REGION Network 30: CLOSEED 1 ALARM
   RUNG wire#powerrail
      I_Contact( #CYL.CLOSE_COMMAND )
      I_Contact( #CLOSE )
      Not()
      Contact( #CLOSED_1_I )
      Contact( #OPENED_1_I )
      Contact( #CYL.SIMULTANEITY_ALARM )
      wire#w1
      Contact( #O_BYTE_0.OPENED_INPUT_1 )
      Contact( "DB1401_PNEUMATIC_SYSTEM".IN_SERVICE )
      Coil( #OPENED_1_ALARM )
   END_RUNG
   RUNG wire#powerrail
      I_Contact( #CYL.OPEN_COMMAND )
      I_Contact( #OPEN )
      Not()
      Contact( #CYL.TIME_EXCEEDED_ALARM )
      I_Contact( #OPENED_1_I )
   END_RUNG wire#w1
   RUNG wire#powerrail
      Contact( #OPENED_1_ALARM )
      I_Contact( "DB2120_MPP_ITC_IPC".RESET_FAULTS )
   END_RUNG wire#w1
   // the same network as SCL:
   #OPENED_1_ALARM := ((NOT (NOT #CYL.CLOSE_COMMAND AND NOT #CLOSE) AND #CLOSED_1_I AND #OPENED_1_I AND #CYL.SIMULTANEITY_ALARM) OR (NOT (NOT #CYL.OPEN_COMMAND AND NOT #OPEN) AND #CYL.TIME_EXCEEDED_ALARM AND NOT #OPENED_1_I) OR (#OPENED_1_ALARM AND NOT "DB2120_MPP_ITC_IPC".RESET_FAULTS)) AND #O_BYTE_0.OPENED_INPUT_1 AND "DB1401_PNEUMATIC_SYSTEM".IN_SERVICE;
END_REGION

REGION Network 31: CLOSEED 2 ALARM
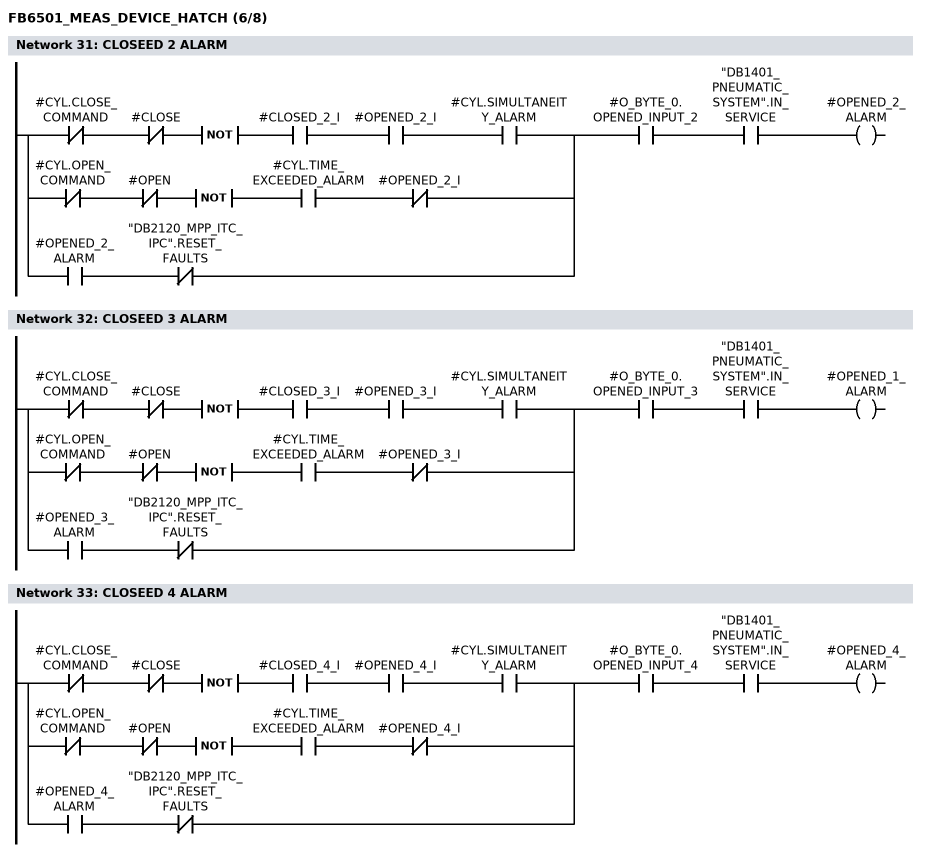
   RUNG wire#powerrail
      I_Contact( #CYL.CLOSE_COMMAND )
      I_Contact( #CLOSE )
      Not()
      Contact( #CLOSED_2_I )
      Contact( #OPENED_2_I )
      Contact( #CYL.SIMULTANEITY_ALARM )
      wire#w1
      Contact( #O_BYTE_0.OPENED_INPUT_2 )
      Contact( "DB1401_PNEUMATIC_SYSTEM".IN_SERVICE )
      Coil( #OPENED_2_ALARM )
   END_RUNG
   RUNG wire#powerrail
      I_Contact( #CYL.OPEN_COMMAND )
      I_Contact( #OPEN )
      Not()
      Contact( #CYL.TIME_EXCEEDED_ALARM )
      I_Contact( #OPENED_2_I )
   END_RUNG wire#w1
   RUNG wire#powerrail
      Contact( #OPENED_2_ALARM )
      I_Contact( "DB2120_MPP_ITC_IPC".RESET_FAULTS )
   END_RUNG wire#w1
   // the same network as SCL:
   #OPENED_2_ALARM := ((NOT (NOT #CYL.CLOSE_COMMAND AND NOT #CLOSE) AND #CLOSED_2_I AND #OPENED_2_I AND #CYL.SIMULTANEITY_ALARM) OR (NOT (NOT #CYL.OPEN_COMMAND AND NOT #OPEN) AND #CYL.TIME_EXCEEDED_ALARM AND NOT #OPENED_2_I) OR (#OPENED_2_ALARM AND NOT "DB2120_MPP_ITC_IPC".RESET_FAULTS)) AND #O_BYTE_0.OPENED_INPUT_2 AND "DB1401_PNEUMATIC_SYSTEM".IN_SERVICE;
END_REGION

REGION Network 32: CLOSEED 3 ALARM
   RUNG wire#powerrail
      I_Contact( #CYL.CLOSE_COMMAND )
      I_Contact( #CLOSE )
      Not()
      Contact( #CLOSED_3_I )
      Contact( #OPENED_3_I )
      Contact( #CYL.SIMULTANEITY_ALARM )
      wire#w1
      Contact( #O_BYTE_0.OPENED_INPUT_3 )
      Contact( "DB1401_PNEUMATIC_SYSTEM".IN_SERVICE )
      Coil( #OPENED_1_ALARM )
   END_RUNG
   RUNG wire#powerrail
      I_Contact( #CYL.OPEN_COMMAND )
      I_Contact( #OPEN )
      Not()
      Contact( #CYL.TIME_EXCEEDED_ALARM )
      I_Contact( #OPENED_3_I )
   END_RUNG wire#w1
   RUNG wire#powerrail
      Contact( #OPENED_3_ALARM )
      I_Contact( "DB2120_MPP_ITC_IPC".RESET_FAULTS )
   END_RUNG wire#w1
   // the same network as SCL:
   #OPENED_1_ALARM := ((NOT (NOT #CYL.CLOSE_COMMAND AND NOT #CLOSE) AND #CLOSED_3_I AND #OPENED_3_I AND #CYL.SIMULTANEITY_ALARM) OR (NOT (NOT #CYL.OPEN_COMMAND AND NOT #OPEN) AND #CYL.TIME_EXCEEDED_ALARM AND NOT #OPENED_3_I) OR (#OPENED_3_ALARM AND NOT "DB2120_MPP_ITC_IPC".RESET_FAULTS)) AND #O_BYTE_0.OPENED_INPUT_3 AND "DB1401_PNEUMATIC_SYSTEM".IN_SERVICE;
END_REGION

REGION Network 33: CLOSEED 4 ALARM
   RUNG wire#powerrail
      I_Contact( #CYL.CLOSE_COMMAND )
      I_Contact( #CLOSE )
      Not()
      Contact( #CLOSED_4_I )
      Contact( #OPENED_4_I )
      Contact( #CYL.SIMULTANEITY_ALARM )
      wire#w1
      Contact( #O_BYTE_0.OPENED_INPUT_4 )
      Contact( "DB1401_PNEUMATIC_SYSTEM".IN_SERVICE )
      Coil( #OPENED_4_ALARM )
   END_RUNG
   RUNG wire#powerrail
      I_Contact( #CYL.OPEN_COMMAND )
      I_Contact( #OPEN )
      Not()
      Contact( #CYL.TIME_EXCEEDED_ALARM )
      I_Contact( #OPENED_4_I )
   END_RUNG wire#w1
   RUNG wire#powerrail
      Contact( #OPENED_4_ALARM )
      I_Contact( "DB2120_MPP_ITC_IPC".RESET_FAULTS )
   END_RUNG wire#w1
   // the same network as SCL:
   #OPENED_4_ALARM := ((NOT (NOT #CYL.CLOSE_COMMAND AND NOT #CLOSE) AND #CLOSED_4_I AND #OPENED_4_I AND #CYL.SIMULTANEITY_ALARM) OR (NOT (NOT #CYL.OPEN_COMMAND AND NOT #OPEN) AND #CYL.TIME_EXCEEDED_ALARM AND NOT #OPENED_4_I) OR (#OPENED_4_ALARM AND NOT "DB2120_MPP_ITC_IPC".RESET_FAULTS)) AND #O_BYTE_0.OPENED_INPUT_4 AND "DB1401_PNEUMATIC_SYSTEM".IN_SERVICE;
END_REGION

REGION Network 34: IMMEDIATE STOP AND STOP END OF CYCLE ALARMS
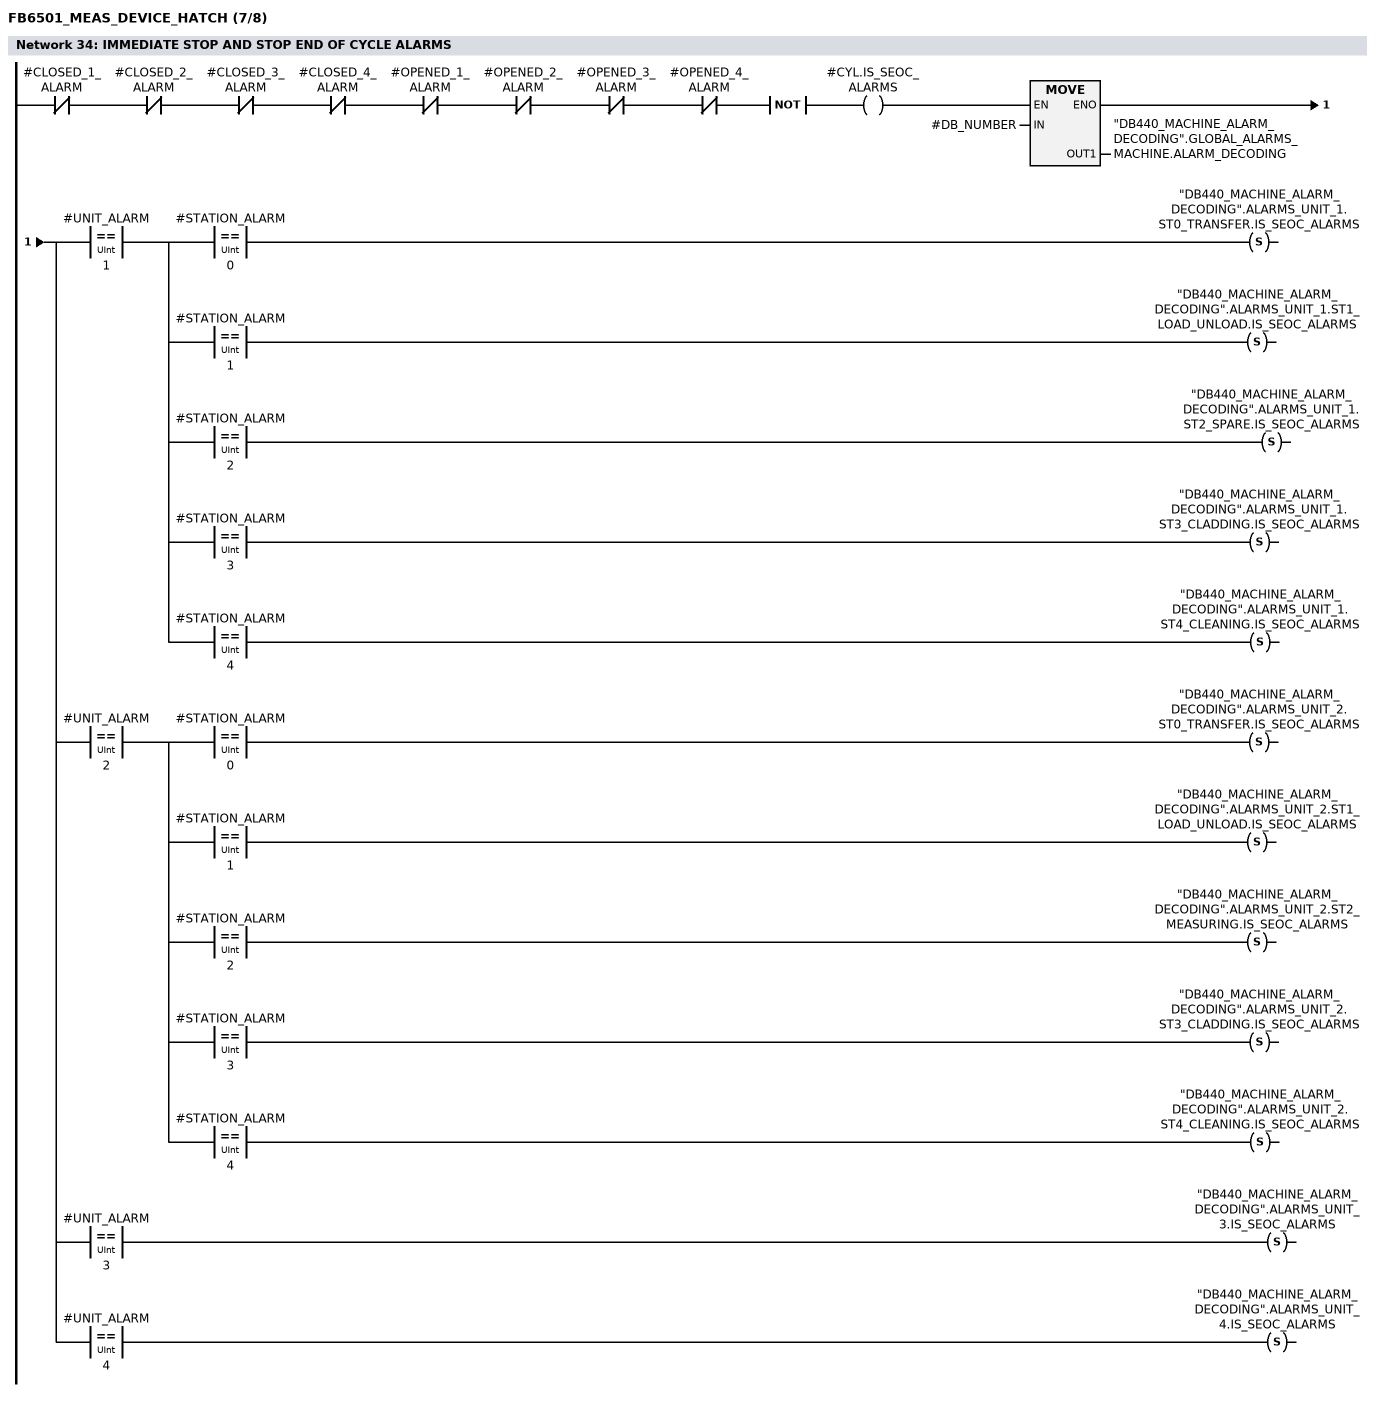
   RUNG wire#powerrail
      I_Contact( #CLOSED_1_ALARM )
      I_Contact( #CLOSED_2_ALARM )
      I_Contact( #CLOSED_3_ALARM )
      I_Contact( #CLOSED_4_ALARM )
      I_Contact( #OPENED_1_ALARM )
      I_Contact( #OPENED_2_ALARM )
      I_Contact( #OPENED_3_ALARM )
      I_Contact( #OPENED_4_ALARM )
      Not()
      Coil( #CYL.IS_SEOC_ALARMS )
      { S7_GenerateENO := "TRUE" } Move(in := #DB_NUMBER, out1 => "DB440_MACHINE_ALARM_DECODING".GLOBAL_ALARMS_MACHINE.ALARM_DECODING)
      wire#w1
      { S7_Templates := "SrcType := UInt" } EQ_Contact(in1 := #UNIT_ALARM, in2 := 1)
      wire#w2
      { S7_Templates := "SrcType := UInt" } EQ_Contact(in1 := #STATION_ALARM, in2 := 0)
      S_Coil( "DB440_MACHINE_ALARM_DECODING".ALARMS_UNIT_1.ST0_TRANSFER.IS_SEOC_ALARMS )
   END_RUNG
   RUNG wire#w2
      { S7_Templates := "SrcType := UInt" } EQ_Contact(in1 := #STATION_ALARM, in2 := 1)
      S_Coil( "DB440_MACHINE_ALARM_DECODING".ALARMS_UNIT_1.ST1_LOAD_UNLOAD.IS_SEOC_ALARMS )
   END_RUNG
   RUNG wire#w2
      { S7_Templates := "SrcType := UInt" } EQ_Contact(in1 := #STATION_ALARM, in2 := 2)
      S_Coil( "DB440_MACHINE_ALARM_DECODING".ALARMS_UNIT_1.ST2_SPARE.IS_SEOC_ALARMS )
   END_RUNG
   RUNG wire#w2
      { S7_Templates := "SrcType := UInt" } EQ_Contact(in1 := #STATION_ALARM, in2 := 3)
      S_Coil( "DB440_MACHINE_ALARM_DECODING".ALARMS_UNIT_1.ST3_CLADDING.IS_SEOC_ALARMS )
   END_RUNG
   RUNG wire#w2
      { S7_Templates := "SrcType := UInt" } EQ_Contact(in1 := #STATION_ALARM, in2 := 4)
      S_Coil( "DB440_MACHINE_ALARM_DECODING".ALARMS_UNIT_1.ST4_CLEANING.IS_SEOC_ALARMS )
   END_RUNG
   RUNG wire#w1
      { S7_Templates := "SrcType := UInt" } EQ_Contact(in1 := #UNIT_ALARM, in2 := 2)
      wire#w3
      { S7_Templates := "SrcType := UInt" } EQ_Contact(in1 := #STATION_ALARM, in2 := 0)
      S_Coil( "DB440_MACHINE_ALARM_DECODING".ALARMS_UNIT_2.ST0_TRANSFER.IS_SEOC_ALARMS )
   END_RUNG
   RUNG wire#w3
      { S7_Templates := "SrcType := UInt" } EQ_Contact(in1 := #STATION_ALARM, in2 := 1)
      S_Coil( "DB440_MACHINE_ALARM_DECODING".ALARMS_UNIT_2.ST1_LOAD_UNLOAD.IS_SEOC_ALARMS )
   END_RUNG
   RUNG wire#w3
      { S7_Templates := "SrcType := UInt" } EQ_Contact(in1 := #STATION_ALARM, in2 := 2)
      S_Coil( "DB440_MACHINE_ALARM_DECODING".ALARMS_UNIT_2.ST2_MEASURING.IS_SEOC_ALARMS )
   END_RUNG
   RUNG wire#w3
      { S7_Templates := "SrcType := UInt" } EQ_Contact(in1 := #STATION_ALARM, in2 := 3)
      S_Coil( "DB440_MACHINE_ALARM_DECODING".ALARMS_UNIT_2.ST3_CLADDING.IS_SEOC_ALARMS )
   END_RUNG
   RUNG wire#w3
      { S7_Templates := "SrcType := UInt" } EQ_Contact(in1 := #STATION_ALARM, in2 := 4)
      S_Coil( "DB440_MACHINE_ALARM_DECODING".ALARMS_UNIT_2.ST4_CLEANING.IS_SEOC_ALARMS )
   END_RUNG
   RUNG wire#w1
      { S7_Templates := "SrcType := UInt" } EQ_Contact(in1 := #UNIT_ALARM, in2 := 3)
      S_Coil( "DB440_MACHINE_ALARM_DECODING".ALARMS_UNIT_3.IS_SEOC_ALARMS )
   END_RUNG
   RUNG wire#w1
      { S7_Templates := "SrcType := UInt" } EQ_Contact(in1 := #UNIT_ALARM, in2 := 4)
      S_Coil( "DB440_MACHINE_ALARM_DECODING".ALARMS_UNIT_4.IS_SEOC_ALARMS )
   END_RUNG
   // the same network as SCL:
   // ENO of a box is taken as its EN; it also drops when the box reports an error
   #CYL.IS_SEOC_ALARMS := NOT (NOT #CLOSED_1_ALARM AND NOT #CLOSED_2_ALARM AND NOT #CLOSED_3_ALARM AND NOT #CLOSED_4_ALARM AND NOT #OPENED_1_ALARM AND NOT #OPENED_2_ALARM AND NOT #OPENED_3_ALARM AND NOT #OPENED_4_ALARM);
   IF #CYL.IS_SEOC_ALARMS THEN
       "DB440_MACHINE_ALARM_DECODING".GLOBAL_ALARMS_MACHINE.ALARM_DECODING := #DB_NUMBER;
   END_IF;
   #_w1 := #CYL.IS_SEOC_ALARMS AND (#UNIT_ALARM = 1);
   IF #_w1 AND (#STATION_ALARM = 0) THEN
       "DB440_MACHINE_ALARM_DECODING".ALARMS_UNIT_1.ST0_TRANSFER.IS_SEOC_ALARMS := TRUE;
   END_IF;
   IF #_w1 AND (#STATION_ALARM = 1) THEN
       "DB440_MACHINE_ALARM_DECODING".ALARMS_UNIT_1.ST1_LOAD_UNLOAD.IS_SEOC_ALARMS := TRUE;
   END_IF;
   IF #_w1 AND (#STATION_ALARM = 2) THEN
       "DB440_MACHINE_ALARM_DECODING".ALARMS_UNIT_1.ST2_SPARE.IS_SEOC_ALARMS := TRUE;
   END_IF;
   IF #_w1 AND (#STATION_ALARM = 3) THEN
       "DB440_MACHINE_ALARM_DECODING".ALARMS_UNIT_1.ST3_CLADDING.IS_SEOC_ALARMS := TRUE;
   END_IF;
   IF #_w1 AND (#STATION_ALARM = 4) THEN
       "DB440_MACHINE_ALARM_DECODING".ALARMS_UNIT_1.ST4_CLEANING.IS_SEOC_ALARMS := TRUE;
   END_IF;
   #_w2 := #CYL.IS_SEOC_ALARMS AND (#UNIT_ALARM = 2);
   IF #_w2 AND (#STATION_ALARM = 0) THEN
       "DB440_MACHINE_ALARM_DECODING".ALARMS_UNIT_2.ST0_TRANSFER.IS_SEOC_ALARMS := TRUE;
   END_IF;
   IF #_w2 AND (#STATION_ALARM = 1) THEN
       "DB440_MACHINE_ALARM_DECODING".ALARMS_UNIT_2.ST1_LOAD_UNLOAD.IS_SEOC_ALARMS := TRUE;
   END_IF;
   IF #_w2 AND (#STATION_ALARM = 2) THEN
       "DB440_MACHINE_ALARM_DECODING".ALARMS_UNIT_2.ST2_MEASURING.IS_SEOC_ALARMS := TRUE;
   END_IF;
   IF #_w2 AND (#STATION_ALARM = 3) THEN
       "DB440_MACHINE_ALARM_DECODING".ALARMS_UNIT_2.ST3_CLADDING.IS_SEOC_ALARMS := TRUE;
   END_IF;
   IF #_w2 AND (#STATION_ALARM = 4) THEN
       "DB440_MACHINE_ALARM_DECODING".ALARMS_UNIT_2.ST4_CLEANING.IS_SEOC_ALARMS := TRUE;
   END_IF;
   IF #CYL.IS_SEOC_ALARMS AND (#UNIT_ALARM = 3) THEN
       "DB440_MACHINE_ALARM_DECODING".ALARMS_UNIT_3.IS_SEOC_ALARMS := TRUE;
   END_IF;
   IF #CYL.IS_SEOC_ALARMS AND (#UNIT_ALARM = 4) THEN
       "DB440_MACHINE_ALARM_DECODING".ALARMS_UNIT_4.IS_SEOC_ALARMS := TRUE;
   END_IF;
END_REGION

REGION Network 35: ANY ACTIVE ALARM
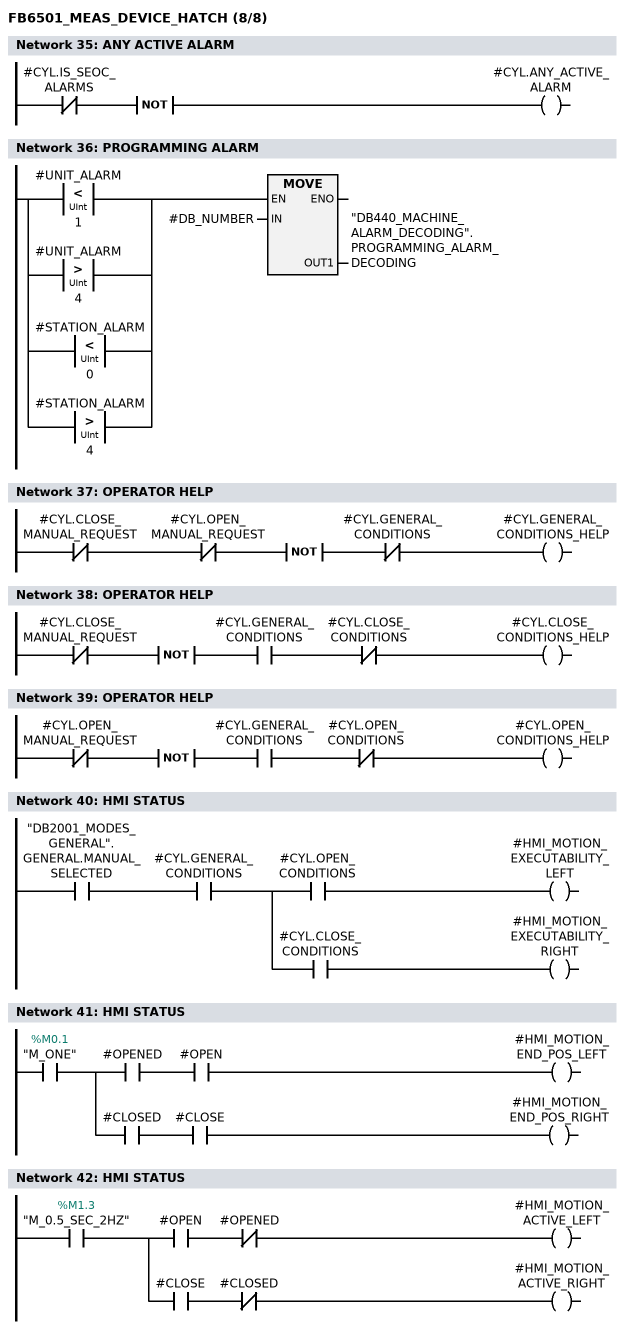
   RUNG wire#powerrail
      I_Contact( #CYL.IS_SEOC_ALARMS )
      Not()
      Coil( #CYL.ANY_ACTIVE_ALARM )
   END_RUNG
   // the same network as SCL:
   #CYL.ANY_ACTIVE_ALARM := NOT (NOT #CYL.IS_SEOC_ALARMS);
END_REGION

REGION Network 36: PROGRAMMING ALARM
   RUNG wire#powerrail
      { S7_Templates := "SrcType := UInt" } LT_Contact(in1 := #UNIT_ALARM, in2 := 1)
      wire#w1
      Move(in := #DB_NUMBER, out1 => "DB440_MACHINE_ALARM_DECODING".PROGRAMMING_ALARM_DECODING)
   END_RUNG
   RUNG wire#powerrail
      { S7_Templates := "SrcType := UInt" } GT_Contact(in1 := #UNIT_ALARM, in2 := 4)
   END_RUNG wire#w1
   RUNG wire#powerrail
      { S7_Templates := "SrcType := UInt" } LT_Contact(in1 := #STATION_ALARM, in2 := 0)
   END_RUNG wire#w1
   RUNG wire#powerrail
      { S7_Templates := "SrcType := UInt" } GT_Contact(in1 := #STATION_ALARM, in2 := 4)
   END_RUNG wire#w1
   // the same network as SCL:
   IF (#UNIT_ALARM < 1) OR (#UNIT_ALARM > 4) OR (#STATION_ALARM < 0) OR (#STATION_ALARM > 4) THEN
       "DB440_MACHINE_ALARM_DECODING".PROGRAMMING_ALARM_DECODING := #DB_NUMBER;
   END_IF;
END_REGION

REGION Network 37: OPERATOR HELP
   RUNG wire#powerrail
      I_Contact( #CYL.CLOSE_MANUAL_REQUEST )
      I_Contact( #CYL.OPEN_MANUAL_REQUEST )
      Not()
      I_Contact( #CYL.GENERAL_CONDITIONS )
      Coil( #CYL.GENERAL_CONDITIONS_HELP )
   END_RUNG
   // the same network as SCL:
   #CYL.GENERAL_CONDITIONS_HELP := NOT (NOT #CYL.CLOSE_MANUAL_REQUEST AND NOT #CYL.OPEN_MANUAL_REQUEST) AND NOT #CYL.GENERAL_CONDITIONS;
END_REGION

REGION Network 38: OPERATOR HELP
   RUNG wire#powerrail
      I_Contact( #CYL.CLOSE_MANUAL_REQUEST )
      Not()
      Contact( #CYL.GENERAL_CONDITIONS )
      I_Contact( #CYL.CLOSE_CONDITIONS )
      Coil( #CYL.CLOSE_CONDITIONS_HELP )
   END_RUNG
   // the same network as SCL:
   #CYL.CLOSE_CONDITIONS_HELP := NOT (NOT #CYL.CLOSE_MANUAL_REQUEST) AND #CYL.GENERAL_CONDITIONS AND NOT #CYL.CLOSE_CONDITIONS;
END_REGION

REGION Network 39: OPERATOR HELP
   RUNG wire#powerrail
      I_Contact( #CYL.OPEN_MANUAL_REQUEST )
      Not()
      Contact( #CYL.GENERAL_CONDITIONS )
      I_Contact( #CYL.OPEN_CONDITIONS )
      Coil( #CYL.OPEN_CONDITIONS_HELP )
   END_RUNG
   // the same network as SCL:
   #CYL.OPEN_CONDITIONS_HELP := NOT (NOT #CYL.OPEN_MANUAL_REQUEST) AND #CYL.GENERAL_CONDITIONS AND NOT #CYL.OPEN_CONDITIONS;
END_REGION

REGION Network 40: HMI STATUS
   RUNG wire#powerrail
      Contact( "DB2001_MODES_GENERAL".GENERAL.MANUAL_SELECTED )
      Contact( #CYL.GENERAL_CONDITIONS )
      wire#w1
      Contact( #CYL.OPEN_CONDITIONS )
      Coil( #HMI_MOTION_EXECUTABILITY_LEFT )
   END_RUNG
   RUNG wire#w1
      Contact( #CYL.CLOSE_CONDITIONS )
      Coil( #HMI_MOTION_EXECUTABILITY_RIGHT )
   END_RUNG
   // the same network as SCL:
   #_w1 := "DB2001_MODES_GENERAL".GENERAL.MANUAL_SELECTED AND #CYL.GENERAL_CONDITIONS;
   #HMI_MOTION_EXECUTABILITY_LEFT := #_w1 AND #CYL.OPEN_CONDITIONS;
   #HMI_MOTION_EXECUTABILITY_RIGHT := #_w1 AND #CYL.CLOSE_CONDITIONS;
END_REGION

REGION Network 41: HMI STATUS
   RUNG wire#powerrail
      Contact( "M_ONE" )
      wire#w1
      Contact( #OPENED )
      Contact( #OPEN )
      Coil( #HMI_MOTION_END_POS_LEFT )
   END_RUNG
   RUNG wire#w1
      Contact( #CLOSED )
      Contact( #CLOSE )
      Coil( #HMI_MOTION_END_POS_RIGHT )
   END_RUNG
   // the same network as SCL:
   #HMI_MOTION_END_POS_LEFT := "M_ONE" AND #OPENED AND #OPEN;
   #HMI_MOTION_END_POS_RIGHT := "M_ONE" AND #CLOSED AND #CLOSE;
END_REGION

REGION Network 42: HMI STATUS
   RUNG wire#powerrail
      Contact( "M_0.5_SEC_2HZ" )
      wire#w1
      Contact( #OPEN )
      I_Contact( #OPENED )
      Coil( #HMI_MOTION_ACTIVE_LEFT )
   END_RUNG
   RUNG wire#w1
      Contact( #CLOSE )
      I_Contact( #CLOSED )
      Coil( #HMI_MOTION_ACTIVE_RIGHT )
   END_RUNG
   // the same network as SCL:
   #HMI_MOTION_ACTIVE_LEFT := "M_0.5_SEC_2HZ" AND #OPEN AND NOT #OPENED;
   #HMI_MOTION_ACTIVE_RIGHT := "M_0.5_SEC_2HZ" AND #CLOSE AND NOT #CLOSED;
END_REGION
END_FUNCTION_BLOCK

FUNCTION_BLOCK "FB6502_SEALING_STRUCTURES"   // FB6502, LAD
{ S7_Optimized_Access := 'FALSE' }
AUTHOR : ETXETAR
VERSION : 1.0
// stored: AutoNumber false, IsIECCheckEnabled false, SetENOAutomatically false, UDAEnableTagReadback false
   VAR_INPUT
      OPTIONS_0 : Byte := 2#0000_0000;   // OPTIONS 0
      CLOSED_1_I : Bool;   // CLOSED 1 INPUT
      CLOSED_2_I : Bool;   // CLOSED 2 INPUT
      CLOSED_3_I : Bool;   // CLOSED 3 INPUT
      CLOSED_4_I : Bool;   // CLOSED 4 INPUT
      OPENED_1_I : Bool;   // OPENED 1 INPUT
      OPENED_2_I : Bool;   // OPENED 2 INPUT
      OPENED_3_I : Bool;   // OPENED 3 INPUT
      OPENED_4_I : Bool;   // OPENED 4 INPUT
      CLOSE_CONDITIONS : Bool;   // CLOSE CONDITIONS
      OPEN_CONDITIONS : Bool;   // OPEN CONDITIONS
      HMI_LINE_REQUEST : Bool;   // HMI LINE REQUEST
      CLOSE_AUTO_REQUEST : Bool;   // AUTO CLOSE REQUEST
      OPEN_AUTO_REQUEST_1 : Bool;   // AUTO OPEN REQUEST
      UNIT_ALARM : UInt;   // UNIT NUMBER MIN. NUMBER=1 MAX. NUMBER=4
      STATION_ALARM : UInt;   // STATION NUMBER MIN. NUMBER=0 MAX. NUMBER=4
   END_VAR
   VAR_OUTPUT
      CLOSED : Bool;   // CLOSED STATUS
      OPENED : Bool;   // OPENED STATUS
      CLOSED_1_ALARM : Bool;   // CLOSED 1 ALARM
      CLOSED_2_ALARM : Bool;   // CLOSED 2 ALARM
      CLOSED_3_ALARM : Bool;   // CLOSED 3 ALARM
      CLOSED_4_ALARM : Bool;   // CLOSED 4 ALARM
      OPENED_1_ALARM : Bool;   // OPENED 1 ALARM
      OPENED_2_ALARM : Bool;   // OPENED 2 ALARM
      OPENED_3_ALARM : Bool;   // OPENED 3 ALARM
      OPENED_4_ALARM : Bool;   // OPENED 4 ALARM
      HMI_MOTION_EXECUTABILITY_LEFT : Bool;   // HMI MOTION EXECUTABILITY LEFT
      HMI_MOTION_EXECUTABILITY_RIGHT : Bool;   // HMI MOTION EXECUTABILITY RIGHT
      HMI_MOTION_END_POS_LEFT : Bool;   // HMI MOTION END POSITION LEFT
      HMI_MOTION_END_POS_RIGHT : Bool;   // HMI MOTION END POSITION RIGHT
      HMI_MOTION_ACTIVE_LEFT : Bool;   // HMI MOTION ACTIVE LEFT
      HMI_MOTION_ACTIVE_RIGHT : Bool;   // HMI MOTION ACTIVE RIGHT
      CLOSE : Bool;   // CLOSE OUTPUT
      OPEN : Bool;   // OPEN OUTPUT
   END_VAR
   VAR DB_SPECIFIC
      CYL { S7_SetPoint := 'True'} : "OPEN_CLOSE_HATCH_CLADDING";
      TIMER_CLOSED { S7_SetPoint := 'True'} : TON_TIME;   // CLOSED TIMER
      TIMER_OPENED { S7_SetPoint := 'True'} : TON_TIME;   // OPENED TIMER
      TIMER_SIMULTANEITY { S7_SetPoint := 'True'} : TON_TIME;   // SIMULTANEITY TIMER
      TIMER_TIME_EXCEEDED { S7_SetPoint := 'True'} : TON_TIME;   // TIME EXCEEDED TIMER
   END_VAR
   VAR_TEMP
      INPUTS_MASK : Byte;   // INPUTS_MASK
      O_BYTE_0 : Struct   // OPTIONS BYTE 0
         CLOSED_INPUT_1 : Bool;   // CLOSED INPUT 1 OPTION
         CLOSED_INPUT_2 : Bool;   // CLOSED INPUT 2 OPTION
         CLOSED_INPUT_3 : Bool;   // CLOSED
         CLOSED_INPUT_4 : Bool;   // CLOSED INPUT 4 OPTION
         OPENED_INPUT_1 : Bool;   // OPENED INPUT 1 OPTION
         OPENED_INPUT_2 : Bool;   // OPENED INPUT 2 OPTION
         OPENED_INPUT_3 : Bool;   // OPENED INPUT 3 OPTION
         OPENED_INPUT_4 : Bool;   // OPENED INPUT 4 OPTION
      END_STRUCT;
      DB_NUMBER : DInt;   // DB NUMBER FOR ALARM AND HELP DECODING
   END_VAR
   // TIMER_CLOSED.PT := T#100MS;
   // TIMER_OPENED.PT := T#300MS;
   // TIMER_SIMULTANEITY.PT := T#100MS;
   // TIMER_TIME_EXCEEDED.PT := T#8S;
   VAR_TEMP   // added for the SCL form of the ladder/FBD networks
      _w1 : Bool;
      _w2 : Bool;
   END_VAR
BEGIN

NETWORK
TITLE = READ INSTANCE DB
      L     DINO;
      +     10#800000;
      T     #DB_NUMBER;


REGION Network 2: OPTIONS
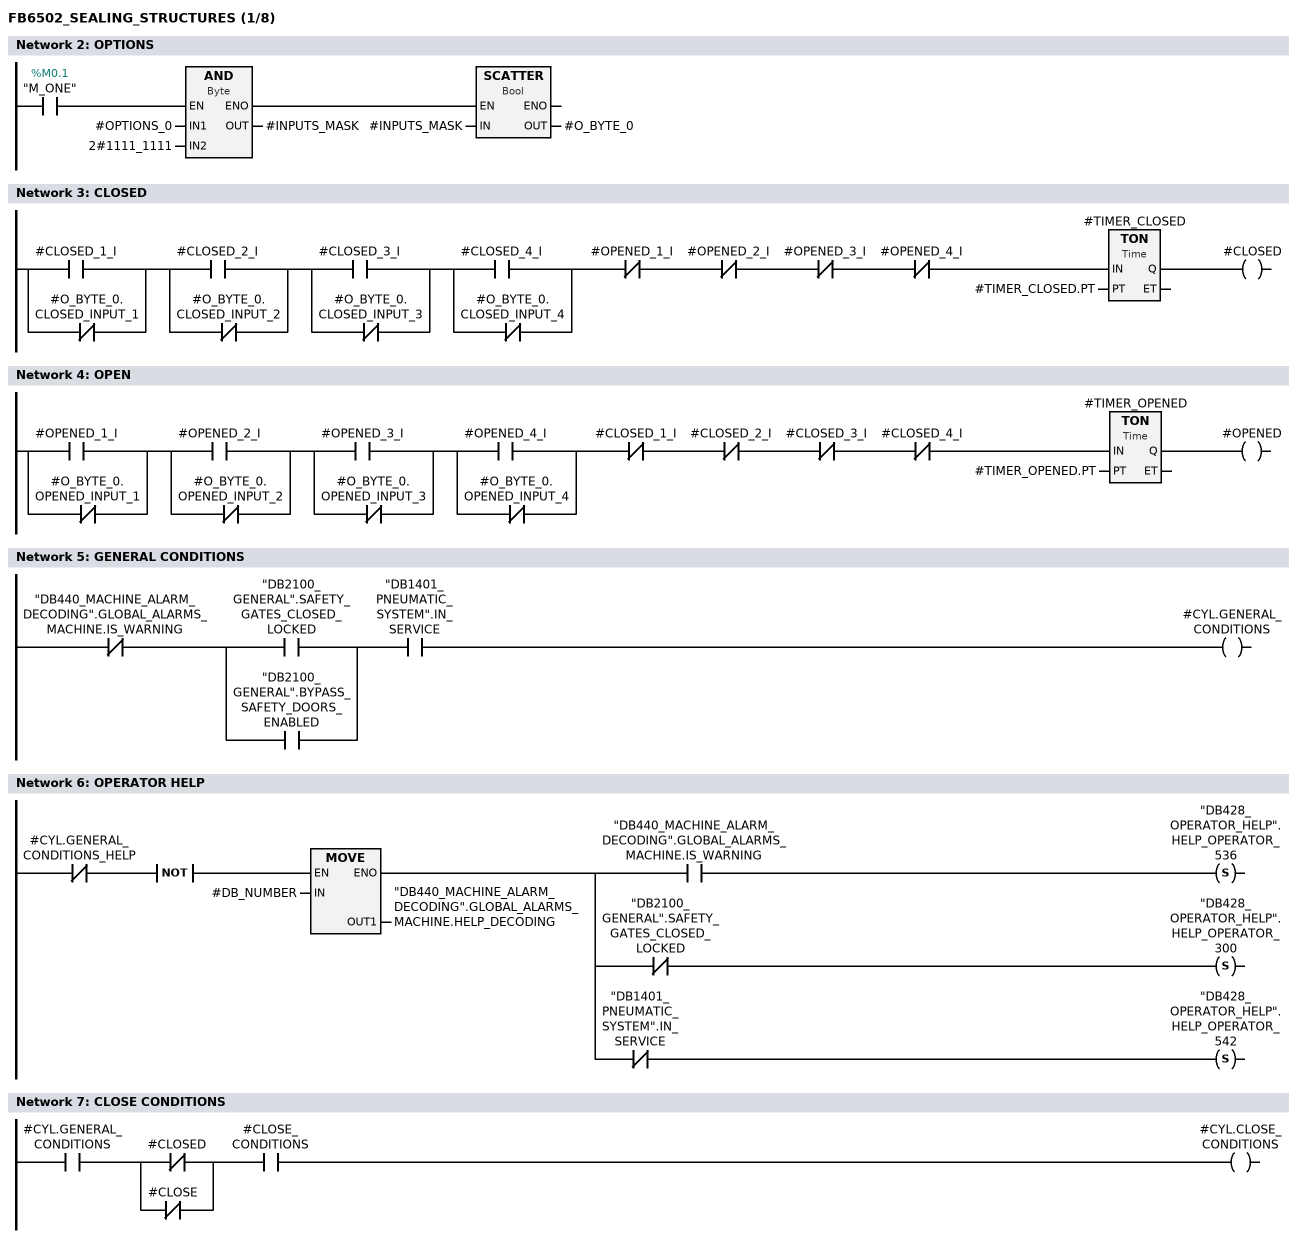
   RUNG wire#powerrail
      Contact( "M_ONE" )
      { S7_Templates := "SrcType := Byte"; S7_GenerateENO := "TRUE" } And(in1 := #OPTIONS_0, in2 := 2#1111_1111, out => #INPUTS_MASK)
      { S7_Templates := "[dest_type := Bool, src_type := Byte]" } SCATTER(IN := #INPUTS_MASK, OUT => #O_BYTE_0)
   END_RUNG
   // the same network as SCL:
   IF "M_ONE" THEN
       #INPUTS_MASK := #OPTIONS_0 AND 2#1111_1111;
       SCATTER(IN := #INPUTS_MASK, OUT => #O_BYTE_0);
   END_IF;
END_REGION

REGION Network 3: CLOSED
   RUNG wire#powerrail
      Contact( #CLOSED_1_I )
      wire#w1
      Contact( #CLOSED_2_I )
      wire#w2
      Contact( #CLOSED_3_I )
      wire#w3
      Contact( #CLOSED_4_I )
      wire#w4
      I_Contact( #OPENED_1_I )
      I_Contact( #OPENED_2_I )
      I_Contact( #OPENED_3_I )
      I_Contact( #OPENED_4_I )
      { S7_Templates := "time_type := Time" } #TIMER_CLOSED.TON(pt := #TIMER_CLOSED.PT, et =>)
      Coil( #CLOSED )
   END_RUNG
   RUNG wire#powerrail
      I_Contact( #O_BYTE_0.CLOSED_INPUT_1 )
   END_RUNG wire#w1
   RUNG wire#w1
      I_Contact( #O_BYTE_0.CLOSED_INPUT_2 )
   END_RUNG wire#w2
   RUNG wire#w2
      I_Contact( #O_BYTE_0.CLOSED_INPUT_3 )
   END_RUNG wire#w3
   RUNG wire#w3
      I_Contact( #O_BYTE_0.CLOSED_INPUT_4 )
   END_RUNG wire#w4
   // the same network as SCL:
   #TIMER_CLOSED(IN := (#CLOSED_1_I OR NOT #O_BYTE_0.CLOSED_INPUT_1) AND (#CLOSED_2_I OR NOT #O_BYTE_0.CLOSED_INPUT_2) AND (#CLOSED_3_I OR NOT #O_BYTE_0.CLOSED_INPUT_3) AND (#CLOSED_4_I OR NOT #O_BYTE_0.CLOSED_INPUT_4) AND NOT #OPENED_1_I AND NOT #OPENED_2_I AND NOT #OPENED_3_I AND NOT #OPENED_4_I,   // TON
                 PT := #TIMER_CLOSED.PT);
   #CLOSED := #TIMER_CLOSED.Q;
END_REGION

REGION Network 4: OPEN
   RUNG wire#powerrail
      Contact( #OPENED_1_I )
      wire#w1
      Contact( #OPENED_2_I )
      wire#w2
      Contact( #OPENED_3_I )
      wire#w3
      Contact( #OPENED_4_I )
      wire#w4
      I_Contact( #CLOSED_1_I )
      I_Contact( #CLOSED_2_I )
      I_Contact( #CLOSED_3_I )
      I_Contact( #CLOSED_4_I )
      { S7_Templates := "time_type := Time" } #TIMER_OPENED.TON(pt := #TIMER_OPENED.PT, et =>)
      Coil( #OPENED )
   END_RUNG
   RUNG wire#powerrail
      I_Contact( #O_BYTE_0.OPENED_INPUT_1 )
   END_RUNG wire#w1
   RUNG wire#w1
      I_Contact( #O_BYTE_0.OPENED_INPUT_2 )
   END_RUNG wire#w2
   RUNG wire#w2
      I_Contact( #O_BYTE_0.OPENED_INPUT_3 )
   END_RUNG wire#w3
   RUNG wire#w3
      I_Contact( #O_BYTE_0.OPENED_INPUT_4 )
   END_RUNG wire#w4
   // the same network as SCL:
   #TIMER_OPENED(IN := (#OPENED_1_I OR NOT #O_BYTE_0.OPENED_INPUT_1) AND (#OPENED_2_I OR NOT #O_BYTE_0.OPENED_INPUT_2) AND (#OPENED_3_I OR NOT #O_BYTE_0.OPENED_INPUT_3) AND (#OPENED_4_I OR NOT #O_BYTE_0.OPENED_INPUT_4) AND NOT #CLOSED_1_I AND NOT #CLOSED_2_I AND NOT #CLOSED_3_I AND NOT #CLOSED_4_I,   // TON
                 PT := #TIMER_OPENED.PT);
   #OPENED := #TIMER_OPENED.Q;
END_REGION

REGION Network 5: GENERAL CONDITIONS
   RUNG wire#powerrail
      I_Contact( "DB440_MACHINE_ALARM_DECODING".GLOBAL_ALARMS_MACHINE.IS_WARNING )
      wire#w1
      Contact( "DB2100_GENERAL".SAFETY_GATES_CLOSED_LOCKED )
      wire#w2
      Contact( "DB1401_PNEUMATIC_SYSTEM".IN_SERVICE )
      Coil( #CYL.GENERAL_CONDITIONS )
   END_RUNG
   RUNG wire#w1
      Contact( "DB2100_GENERAL".BYPASS_SAFETY_DOORS_ENABLED )
   END_RUNG wire#w2
   // the same network as SCL:
   #CYL.GENERAL_CONDITIONS := NOT "DB440_MACHINE_ALARM_DECODING".GLOBAL_ALARMS_MACHINE.IS_WARNING AND ("DB2100_GENERAL".SAFETY_GATES_CLOSED_LOCKED OR "DB2100_GENERAL".BYPASS_SAFETY_DOORS_ENABLED) AND "DB1401_PNEUMATIC_SYSTEM".IN_SERVICE;
END_REGION

REGION Network 6: OPERATOR HELP
   RUNG wire#powerrail
      I_Contact( #CYL.GENERAL_CONDITIONS_HELP )
      Not()
      { S7_GenerateENO := "TRUE" } Move(in := #DB_NUMBER, out1 => "DB440_MACHINE_ALARM_DECODING".GLOBAL_ALARMS_MACHINE.HELP_DECODING)
      wire#w1
      Contact( "DB440_MACHINE_ALARM_DECODING".GLOBAL_ALARMS_MACHINE.IS_WARNING )
      S_Coil( "DB428_OPERATOR_HELP".HELP_OPERATOR_536 )
   END_RUNG
   RUNG wire#w1
      I_Contact( "DB2100_GENERAL".SAFETY_GATES_CLOSED_LOCKED )
      S_Coil( "DB428_OPERATOR_HELP".HELP_OPERATOR_300 )
   END_RUNG
   RUNG wire#w1
      I_Contact( "DB1401_PNEUMATIC_SYSTEM".IN_SERVICE )
      S_Coil( "DB428_OPERATOR_HELP".HELP_OPERATOR_542 )
   END_RUNG
   // the same network as SCL:
   // ENO of a box is taken as its EN; it also drops when the box reports an error
   #_w1 := NOT (NOT #CYL.GENERAL_CONDITIONS_HELP);
   IF #_w1 THEN "DB440_MACHINE_ALARM_DECODING".GLOBAL_ALARMS_MACHINE.HELP_DECODING := #DB_NUMBER; END_IF;
   IF #_w1 AND "DB440_MACHINE_ALARM_DECODING".GLOBAL_ALARMS_MACHINE.IS_WARNING THEN
       "DB428_OPERATOR_HELP".HELP_OPERATOR_536 := TRUE;
   END_IF;
   IF #_w1 AND NOT "DB2100_GENERAL".SAFETY_GATES_CLOSED_LOCKED THEN
       "DB428_OPERATOR_HELP".HELP_OPERATOR_300 := TRUE;
   END_IF;
   IF #_w1 AND NOT "DB1401_PNEUMATIC_SYSTEM".IN_SERVICE THEN
       "DB428_OPERATOR_HELP".HELP_OPERATOR_542 := TRUE;
   END_IF;
END_REGION

REGION Network 7: CLOSE CONDITIONS
   RUNG wire#powerrail
      Contact( #CYL.GENERAL_CONDITIONS )
      wire#w1
      I_Contact( #CLOSED )
      wire#w2
      Contact( #CLOSE_CONDITIONS )
      Coil( #CYL.CLOSE_CONDITIONS )
   END_RUNG
   RUNG wire#w1
      I_Contact( #CLOSE )
   END_RUNG wire#w2
   // the same network as SCL:
   #CYL.CLOSE_CONDITIONS := #CYL.GENERAL_CONDITIONS AND (NOT #CLOSED OR NOT #CLOSE) AND #CLOSE_CONDITIONS;
END_REGION

REGION Network 8: OPERATOR HELP
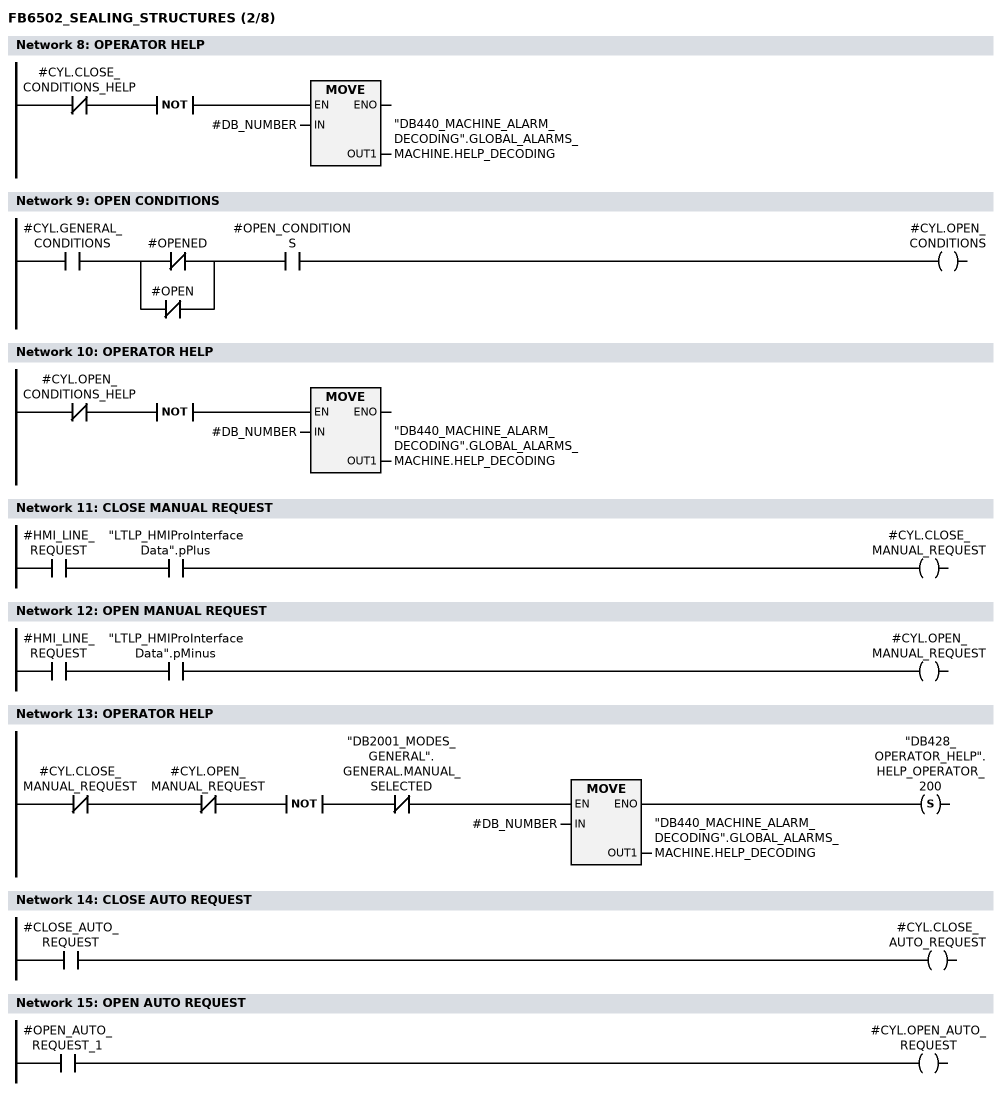
   RUNG wire#powerrail
      I_Contact( #CYL.CLOSE_CONDITIONS_HELP )
      Not()
      { S7_GenerateENO := "TRUE" } Move(in := #DB_NUMBER, out1 => "DB440_MACHINE_ALARM_DECODING".GLOBAL_ALARMS_MACHINE.HELP_DECODING)
   END_RUNG
   // the same network as SCL:
   IF NOT (NOT #CYL.CLOSE_CONDITIONS_HELP) THEN
       "DB440_MACHINE_ALARM_DECODING".GLOBAL_ALARMS_MACHINE.HELP_DECODING := #DB_NUMBER;
   END_IF;
END_REGION

REGION Network 9: OPEN CONDITIONS
   RUNG wire#powerrail
      Contact( #CYL.GENERAL_CONDITIONS )
      wire#w1
      I_Contact( #OPENED )
      wire#w2
      Contact( #OPEN_CONDITIONS )
      Coil( #CYL.OPEN_CONDITIONS )
   END_RUNG
   RUNG wire#w1
      I_Contact( #OPEN )
   END_RUNG wire#w2
   // the same network as SCL:
   #CYL.OPEN_CONDITIONS := #CYL.GENERAL_CONDITIONS AND (NOT #OPENED OR NOT #OPEN) AND #OPEN_CONDITIONS;
END_REGION

REGION Network 10: OPERATOR HELP
   RUNG wire#powerrail
      I_Contact( #CYL.OPEN_CONDITIONS_HELP )
      Not()
      { S7_GenerateENO := "TRUE" } Move(in := #DB_NUMBER, out1 => "DB440_MACHINE_ALARM_DECODING".GLOBAL_ALARMS_MACHINE.HELP_DECODING)
   END_RUNG
   // the same network as SCL:
   IF NOT (NOT #CYL.OPEN_CONDITIONS_HELP) THEN
       "DB440_MACHINE_ALARM_DECODING".GLOBAL_ALARMS_MACHINE.HELP_DECODING := #DB_NUMBER;
   END_IF;
END_REGION

REGION Network 11: CLOSE MANUAL REQUEST
   RUNG wire#powerrail
      Contact( #HMI_LINE_REQUEST )
      Contact( "LTLP_HMIProInterfaceData".pPlus )
      Coil( #CYL.CLOSE_MANUAL_REQUEST )
   END_RUNG
   // the same network as SCL:
   #CYL.CLOSE_MANUAL_REQUEST := #HMI_LINE_REQUEST AND "LTLP_HMIProInterfaceData".pPlus;
END_REGION

REGION Network 12: OPEN MANUAL REQUEST
   RUNG wire#powerrail
      Contact( #HMI_LINE_REQUEST )
      Contact( "LTLP_HMIProInterfaceData".pMinus )
      Coil( #CYL.OPEN_MANUAL_REQUEST )
   END_RUNG
   // the same network as SCL:
   #CYL.OPEN_MANUAL_REQUEST := #HMI_LINE_REQUEST AND "LTLP_HMIProInterfaceData".pMinus;
END_REGION

REGION Network 13: OPERATOR HELP
   RUNG wire#powerrail
      I_Contact( #CYL.CLOSE_MANUAL_REQUEST )
      I_Contact( #CYL.OPEN_MANUAL_REQUEST )
      Not()
      I_Contact( "DB2001_MODES_GENERAL".GENERAL.MANUAL_SELECTED )
      { S7_GenerateENO := "TRUE" } Move(in := #DB_NUMBER, out1 => "DB440_MACHINE_ALARM_DECODING".GLOBAL_ALARMS_MACHINE.HELP_DECODING)
      S_Coil( "DB428_OPERATOR_HELP".HELP_OPERATOR_200 )
   END_RUNG
   // the same network as SCL:
   // ENO of a box is taken as its EN; it also drops when the box reports an error
   IF NOT (NOT #CYL.CLOSE_MANUAL_REQUEST AND NOT #CYL.OPEN_MANUAL_REQUEST) AND NOT "DB2001_MODES_GENERAL".GENERAL.MANUAL_SELECTED THEN
       "DB440_MACHINE_ALARM_DECODING".GLOBAL_ALARMS_MACHINE.HELP_DECODING := #DB_NUMBER;
       "DB428_OPERATOR_HELP".HELP_OPERATOR_200 := TRUE;
   END_IF;
END_REGION

REGION Network 14: CLOSE AUTO REQUEST
   RUNG wire#powerrail
      Contact( #CLOSE_AUTO_REQUEST )
      Coil( #CYL.CLOSE_AUTO_REQUEST )
   END_RUNG
   // the same network as SCL:
   #CYL.CLOSE_AUTO_REQUEST := #CLOSE_AUTO_REQUEST;
END_REGION

REGION Network 15: OPEN AUTO REQUEST
   RUNG wire#powerrail
      Contact( #OPEN_AUTO_REQUEST_1 )
      Coil( #CYL.OPEN_AUTO_REQUEST )
   END_RUNG
   // the same network as SCL:
   #CYL.OPEN_AUTO_REQUEST := #OPEN_AUTO_REQUEST_1;
END_REGION

REGION Network 16: CLOSE GLOBAL REQUEST
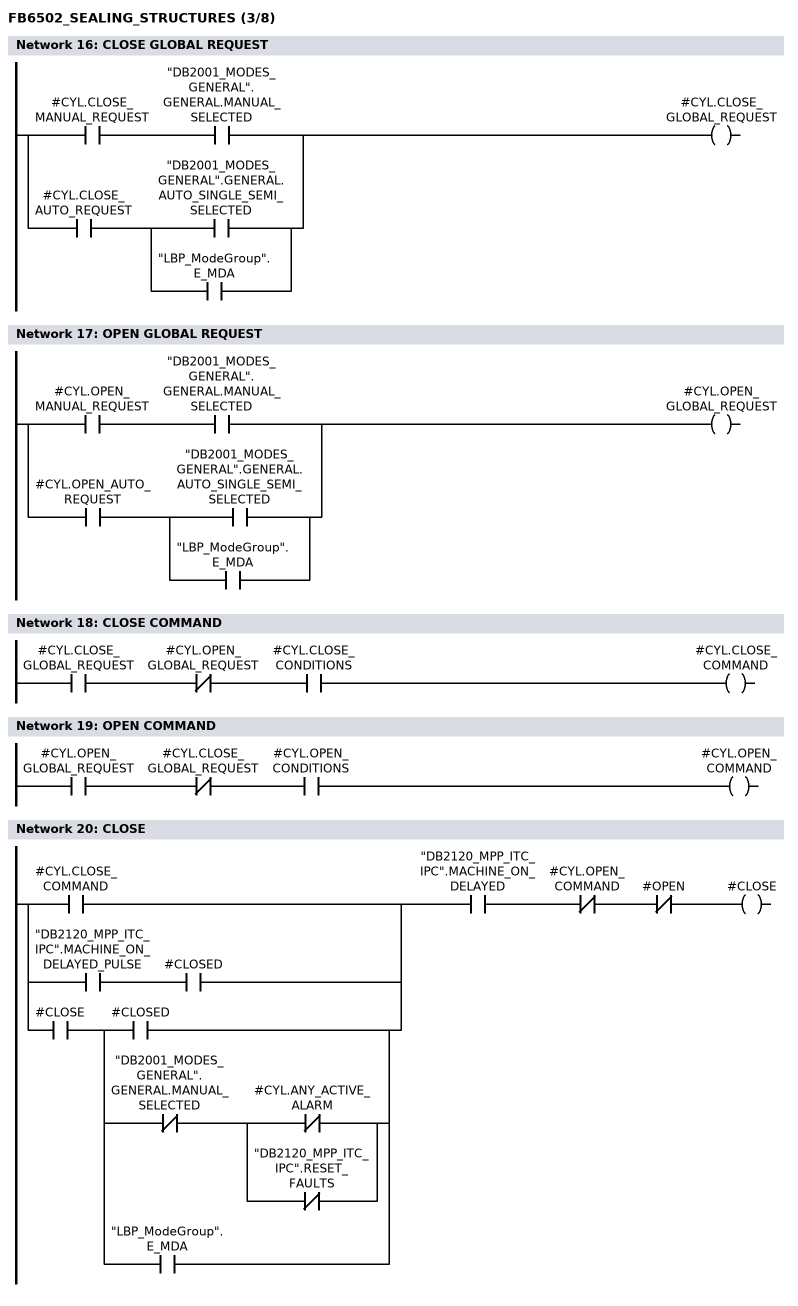
   RUNG wire#powerrail
      Contact( #CYL.CLOSE_MANUAL_REQUEST )
      Contact( "DB2001_MODES_GENERAL".GENERAL.MANUAL_SELECTED )
      wire#w1
      Coil( #CYL.CLOSE_GLOBAL_REQUEST )
   END_RUNG
   RUNG wire#powerrail
      Contact( #CYL.CLOSE_AUTO_REQUEST )
      wire#w2
      Contact( "DB2001_MODES_GENERAL".GENERAL.AUTO_SINGLE_SEMI_SELECTED )
   END_RUNG wire#w1
   RUNG wire#w2
      Contact( "LBP_ModeGroup".E_MDA )
   END_RUNG wire#w1
   // the same network as SCL:
   #CYL.CLOSE_GLOBAL_REQUEST := (#CYL.CLOSE_MANUAL_REQUEST AND "DB2001_MODES_GENERAL".GENERAL.MANUAL_SELECTED) OR (#CYL.CLOSE_AUTO_REQUEST AND ("DB2001_MODES_GENERAL".GENERAL.AUTO_SINGLE_SEMI_SELECTED OR "LBP_ModeGroup".E_MDA));
END_REGION

REGION Network 17: OPEN GLOBAL REQUEST
   RUNG wire#powerrail
      Contact( #CYL.OPEN_MANUAL_REQUEST )
      Contact( "DB2001_MODES_GENERAL".GENERAL.MANUAL_SELECTED )
      wire#w1
      Coil( #CYL.OPEN_GLOBAL_REQUEST )
   END_RUNG
   RUNG wire#powerrail
      Contact( #CYL.OPEN_AUTO_REQUEST )
      wire#w2
      Contact( "DB2001_MODES_GENERAL".GENERAL.AUTO_SINGLE_SEMI_SELECTED )
   END_RUNG wire#w1
   RUNG wire#w2
      Contact( "LBP_ModeGroup".E_MDA )
   END_RUNG wire#w1
   // the same network as SCL:
   #CYL.OPEN_GLOBAL_REQUEST := (#CYL.OPEN_MANUAL_REQUEST AND "DB2001_MODES_GENERAL".GENERAL.MANUAL_SELECTED) OR (#CYL.OPEN_AUTO_REQUEST AND ("DB2001_MODES_GENERAL".GENERAL.AUTO_SINGLE_SEMI_SELECTED OR "LBP_ModeGroup".E_MDA));
END_REGION

REGION Network 18: CLOSE COMMAND
   RUNG wire#powerrail
      Contact( #CYL.CLOSE_GLOBAL_REQUEST )
      I_Contact( #CYL.OPEN_GLOBAL_REQUEST )
      Contact( #CYL.CLOSE_CONDITIONS )
      Coil( #CYL.CLOSE_COMMAND )
   END_RUNG
   // the same network as SCL:
   #CYL.CLOSE_COMMAND := #CYL.CLOSE_GLOBAL_REQUEST AND NOT #CYL.OPEN_GLOBAL_REQUEST AND #CYL.CLOSE_CONDITIONS;
END_REGION

REGION Network 19: OPEN COMMAND
   RUNG wire#powerrail
      Contact( #CYL.OPEN_GLOBAL_REQUEST )
      I_Contact( #CYL.CLOSE_GLOBAL_REQUEST )
      Contact( #CYL.OPEN_CONDITIONS )
      Coil( #CYL.OPEN_COMMAND )
   END_RUNG
   // the same network as SCL:
   #CYL.OPEN_COMMAND := #CYL.OPEN_GLOBAL_REQUEST AND NOT #CYL.CLOSE_GLOBAL_REQUEST AND #CYL.OPEN_CONDITIONS;
END_REGION

REGION Network 20: CLOSE
   RUNG wire#powerrail
      Contact( #CYL.CLOSE_COMMAND )
      wire#w1
      Contact( "DB2120_MPP_ITC_IPC".MACHINE_ON_DELAYED )
      I_Contact( #CYL.OPEN_COMMAND )
      I_Contact( #OPEN )
      Coil( #CLOSE )
   END_RUNG
   RUNG wire#powerrail
      Contact( "DB2120_MPP_ITC_IPC".MACHINE_ON_DELAYED_PULSE )
      Contact( #CLOSED )
   END_RUNG wire#w1
   RUNG wire#powerrail
      Contact( #CLOSE )
      wire#w2
      Contact( #CLOSED )
   END_RUNG wire#w1
   RUNG wire#w2
      I_Contact( "DB2001_MODES_GENERAL".GENERAL.MANUAL_SELECTED )
      wire#w3
      I_Contact( #CYL.ANY_ACTIVE_ALARM )
   END_RUNG wire#w1
   RUNG wire#w3
      I_Contact( "DB2120_MPP_ITC_IPC".RESET_FAULTS )
   END_RUNG wire#w1
   RUNG wire#w2
      Contact( "LBP_ModeGroup".E_MDA )
   END_RUNG wire#w1
   // the same network as SCL:
   #CLOSE := (#CYL.CLOSE_COMMAND OR ("DB2120_MPP_ITC_IPC".MACHINE_ON_DELAYED_PULSE AND #CLOSED) OR (#CLOSE AND (#CLOSED OR (NOT "DB2001_MODES_GENERAL".GENERAL.MANUAL_SELECTED AND (NOT #CYL.ANY_ACTIVE_ALARM OR NOT "DB2120_MPP_ITC_IPC".RESET_FAULTS)) OR "LBP_ModeGroup".E_MDA))) AND "DB2120_MPP_ITC_IPC".MACHINE_ON_DELAYED AND NOT #CYL.OPEN_COMMAND AND NOT #OPEN;
END_REGION

REGION Network 21: OPEN
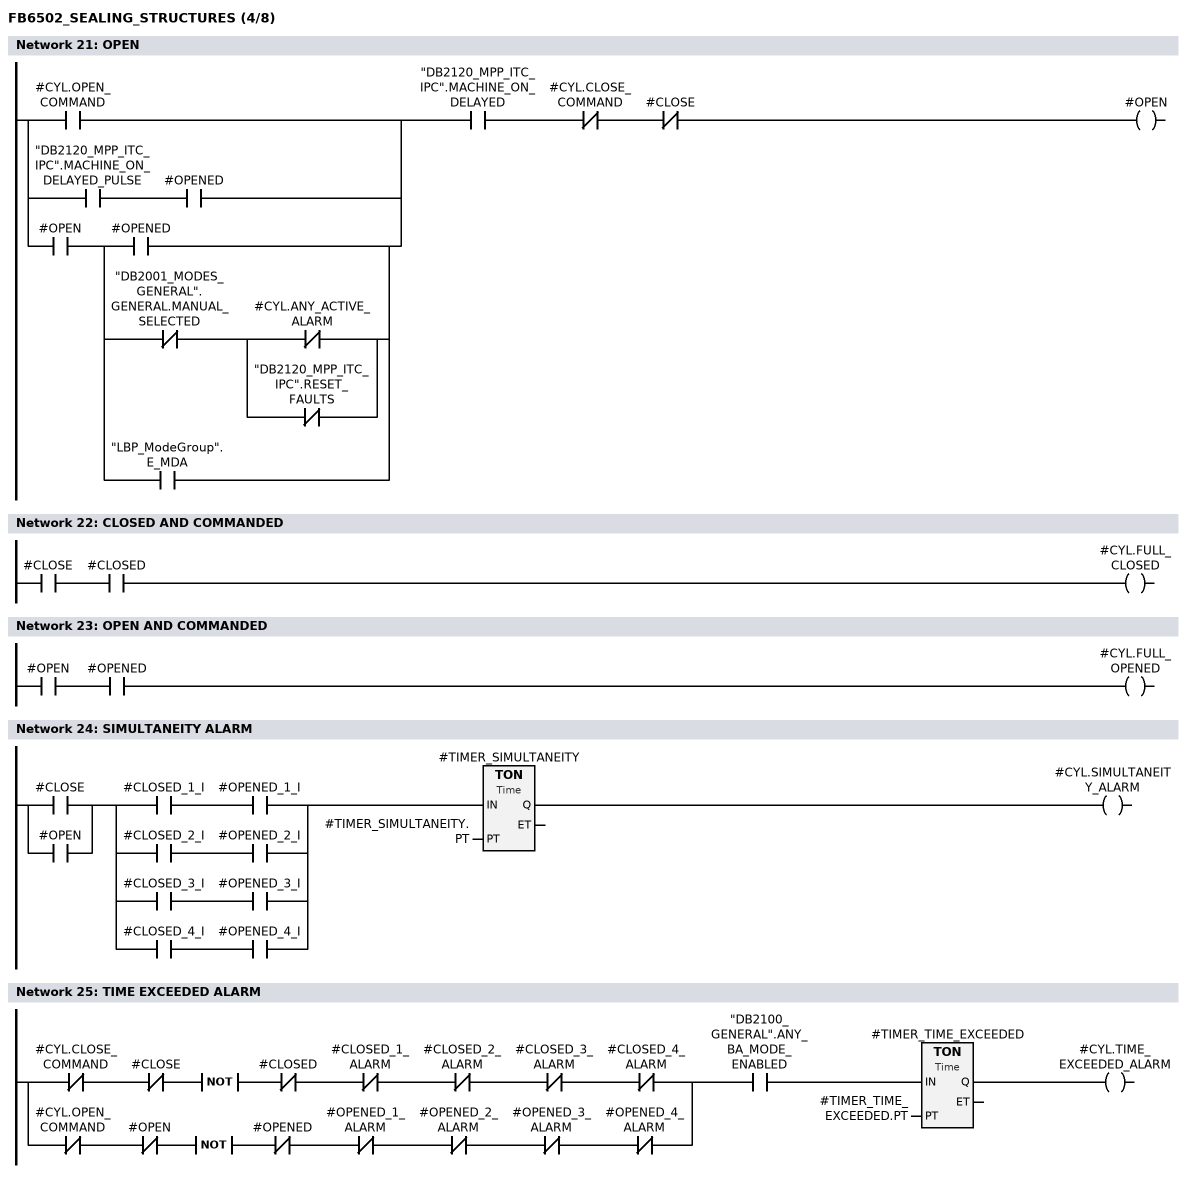
   RUNG wire#powerrail
      Contact( #CYL.OPEN_COMMAND )
      wire#w1
      Contact( "DB2120_MPP_ITC_IPC".MACHINE_ON_DELAYED )
      I_Contact( #CYL.CLOSE_COMMAND )
      I_Contact( #CLOSE )
      Coil( #OPEN )
   END_RUNG
   RUNG wire#powerrail
      Contact( "DB2120_MPP_ITC_IPC".MACHINE_ON_DELAYED_PULSE )
      Contact( #OPENED )
   END_RUNG wire#w1
   RUNG wire#powerrail
      Contact( #OPEN )
      wire#w2
      Contact( #OPENED )
   END_RUNG wire#w1
   RUNG wire#w2
      I_Contact( "DB2001_MODES_GENERAL".GENERAL.MANUAL_SELECTED )
      wire#w3
      I_Contact( #CYL.ANY_ACTIVE_ALARM )
   END_RUNG wire#w1
   RUNG wire#w3
      I_Contact( "DB2120_MPP_ITC_IPC".RESET_FAULTS )
   END_RUNG wire#w1
   RUNG wire#w2
      Contact( "LBP_ModeGroup".E_MDA )
   END_RUNG wire#w1
   // the same network as SCL:
   #OPEN := (#CYL.OPEN_COMMAND OR ("DB2120_MPP_ITC_IPC".MACHINE_ON_DELAYED_PULSE AND #OPENED) OR (#OPEN AND (#OPENED OR (NOT "DB2001_MODES_GENERAL".GENERAL.MANUAL_SELECTED AND (NOT #CYL.ANY_ACTIVE_ALARM OR NOT "DB2120_MPP_ITC_IPC".RESET_FAULTS)) OR "LBP_ModeGroup".E_MDA))) AND "DB2120_MPP_ITC_IPC".MACHINE_ON_DELAYED AND NOT #CYL.CLOSE_COMMAND AND NOT #CLOSE;
END_REGION

REGION Network 22: CLOSED AND COMMANDED
   RUNG wire#powerrail
      Contact( #CLOSE )
      Contact( #CLOSED )
      Coil( #CYL.FULL_CLOSED )
   END_RUNG
   // the same network as SCL:
   #CYL.FULL_CLOSED := #CLOSE AND #CLOSED;
END_REGION

REGION Network 23: OPEN AND COMMANDED
   RUNG wire#powerrail
      Contact( #OPEN )
      Contact( #OPENED )
      Coil( #CYL.FULL_OPENED )
   END_RUNG
   // the same network as SCL:
   #CYL.FULL_OPENED := #OPEN AND #OPENED;
END_REGION

REGION Network 24: SIMULTANEITY ALARM
   RUNG wire#powerrail
      Contact( #CLOSE )
      wire#w1
      Contact( #CLOSED_1_I )
      Contact( #OPENED_1_I )
      wire#w2
      { S7_Templates := "time_type := Time" } #TIMER_SIMULTANEITY.TON(pt := #TIMER_SIMULTANEITY.PT, et =>)
      Coil( #CYL.SIMULTANEITY_ALARM )
   END_RUNG
   RUNG wire#powerrail
      Contact( #OPEN )
   END_RUNG wire#w1
   RUNG wire#w1
      Contact( #CLOSED_2_I )
      Contact( #OPENED_2_I )
   END_RUNG wire#w2
   RUNG wire#w1
      Contact( #CLOSED_3_I )
      Contact( #OPENED_3_I )
   END_RUNG wire#w2
   RUNG wire#w1
      Contact( #CLOSED_4_I )
      Contact( #OPENED_4_I )
   END_RUNG wire#w2
   // the same network as SCL:
   #TIMER_SIMULTANEITY(IN := (#CLOSE OR #OPEN) AND ((#CLOSED_1_I AND #OPENED_1_I) OR (#CLOSED_2_I AND #OPENED_2_I) OR (#CLOSED_3_I AND #OPENED_3_I) OR (#CLOSED_4_I AND #OPENED_4_I)),   // TON
                       PT := #TIMER_SIMULTANEITY.PT);
   #CYL.SIMULTANEITY_ALARM := #TIMER_SIMULTANEITY.Q;
END_REGION

REGION Network 25: TIME EXCEEDED ALARM
   RUNG wire#powerrail
      I_Contact( #CYL.CLOSE_COMMAND )
      I_Contact( #CLOSE )
      Not()
      I_Contact( #CLOSED )
      I_Contact( #CLOSED_1_ALARM )
      I_Contact( #CLOSED_2_ALARM )
      I_Contact( #CLOSED_3_ALARM )
      I_Contact( #CLOSED_4_ALARM )
      wire#w1
      Contact( "DB2100_GENERAL".ANY_BA_MODE_ENABLED )
      { S7_Templates := "time_type := Time" } #TIMER_TIME_EXCEEDED.TON(pt := #TIMER_TIME_EXCEEDED.PT, et =>)
      Coil( #CYL.TIME_EXCEEDED_ALARM )
   END_RUNG
   RUNG wire#powerrail
      I_Contact( #CYL.OPEN_COMMAND )
      I_Contact( #OPEN )
      Not()
      I_Contact( #OPENED )
      I_Contact( #OPENED_1_ALARM )
      I_Contact( #OPENED_2_ALARM )
      I_Contact( #OPENED_3_ALARM )
      I_Contact( #OPENED_4_ALARM )
   END_RUNG wire#w1
   // the same network as SCL:
   #TIMER_TIME_EXCEEDED(IN := ((NOT (NOT #CYL.CLOSE_COMMAND AND NOT #CLOSE) AND NOT #CLOSED AND NOT #CLOSED_1_ALARM AND NOT #CLOSED_2_ALARM AND NOT #CLOSED_3_ALARM AND NOT #CLOSED_4_ALARM) OR (NOT (NOT #CYL.OPEN_COMMAND AND NOT #OPEN) AND NOT #OPENED AND NOT #OPENED_1_ALARM AND NOT #OPENED_2_ALARM AND NOT #OPENED_3_ALARM AND NOT #OPENED_4_ALARM)) AND "DB2100_GENERAL".ANY_BA_MODE_ENABLED,   // TON
                        PT := #TIMER_TIME_EXCEEDED.PT);
   #CYL.TIME_EXCEEDED_ALARM := #TIMER_TIME_EXCEEDED.Q;
END_REGION

REGION Network 26: CLOSED 1 ALARM
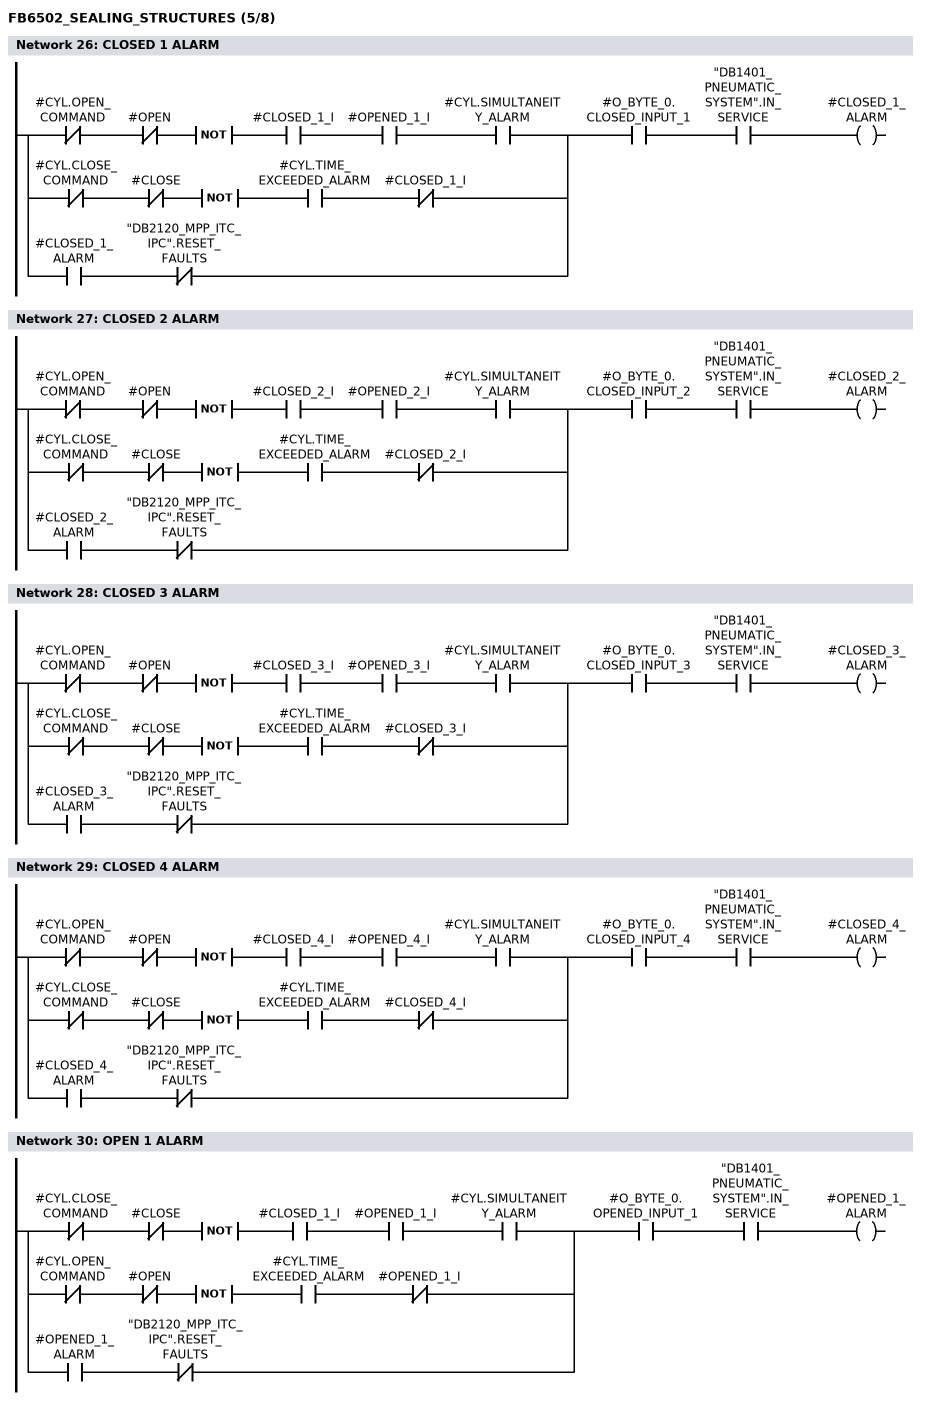
   RUNG wire#powerrail
      I_Contact( #CYL.OPEN_COMMAND )
      I_Contact( #OPEN )
      Not()
      Contact( #CLOSED_1_I )
      Contact( #OPENED_1_I )
      Contact( #CYL.SIMULTANEITY_ALARM )
      wire#w1
      Contact( #O_BYTE_0.CLOSED_INPUT_1 )
      Contact( "DB1401_PNEUMATIC_SYSTEM".IN_SERVICE )
      Coil( #CLOSED_1_ALARM )
   END_RUNG
   RUNG wire#powerrail
      I_Contact( #CYL.CLOSE_COMMAND )
      I_Contact( #CLOSE )
      Not()
      Contact( #CYL.TIME_EXCEEDED_ALARM )
      I_Contact( #CLOSED_1_I )
   END_RUNG wire#w1
   RUNG wire#powerrail
      Contact( #CLOSED_1_ALARM )
      I_Contact( "DB2120_MPP_ITC_IPC".RESET_FAULTS )
   END_RUNG wire#w1
   // the same network as SCL:
   #CLOSED_1_ALARM := ((NOT (NOT #CYL.OPEN_COMMAND AND NOT #OPEN) AND #CLOSED_1_I AND #OPENED_1_I AND #CYL.SIMULTANEITY_ALARM) OR (NOT (NOT #CYL.CLOSE_COMMAND AND NOT #CLOSE) AND #CYL.TIME_EXCEEDED_ALARM AND NOT #CLOSED_1_I) OR (#CLOSED_1_ALARM AND NOT "DB2120_MPP_ITC_IPC".RESET_FAULTS)) AND #O_BYTE_0.CLOSED_INPUT_1 AND "DB1401_PNEUMATIC_SYSTEM".IN_SERVICE;
END_REGION

REGION Network 27: CLOSED 2 ALARM
   RUNG wire#powerrail
      I_Contact( #CYL.OPEN_COMMAND )
      I_Contact( #OPEN )
      Not()
      Contact( #CLOSED_2_I )
      Contact( #OPENED_2_I )
      Contact( #CYL.SIMULTANEITY_ALARM )
      wire#w1
      Contact( #O_BYTE_0.CLOSED_INPUT_2 )
      Contact( "DB1401_PNEUMATIC_SYSTEM".IN_SERVICE )
      Coil( #CLOSED_2_ALARM )
   END_RUNG
   RUNG wire#powerrail
      I_Contact( #CYL.CLOSE_COMMAND )
      I_Contact( #CLOSE )
      Not()
      Contact( #CYL.TIME_EXCEEDED_ALARM )
      I_Contact( #CLOSED_2_I )
   END_RUNG wire#w1
   RUNG wire#powerrail
      Contact( #CLOSED_2_ALARM )
      I_Contact( "DB2120_MPP_ITC_IPC".RESET_FAULTS )
   END_RUNG wire#w1
   // the same network as SCL:
   #CLOSED_2_ALARM := ((NOT (NOT #CYL.OPEN_COMMAND AND NOT #OPEN) AND #CLOSED_2_I AND #OPENED_2_I AND #CYL.SIMULTANEITY_ALARM) OR (NOT (NOT #CYL.CLOSE_COMMAND AND NOT #CLOSE) AND #CYL.TIME_EXCEEDED_ALARM AND NOT #CLOSED_2_I) OR (#CLOSED_2_ALARM AND NOT "DB2120_MPP_ITC_IPC".RESET_FAULTS)) AND #O_BYTE_0.CLOSED_INPUT_2 AND "DB1401_PNEUMATIC_SYSTEM".IN_SERVICE;
END_REGION

REGION Network 28: CLOSED 3 ALARM
   RUNG wire#powerrail
      I_Contact( #CYL.OPEN_COMMAND )
      I_Contact( #OPEN )
      Not()
      Contact( #CLOSED_3_I )
      Contact( #OPENED_3_I )
      Contact( #CYL.SIMULTANEITY_ALARM )
      wire#w1
      Contact( #O_BYTE_0.CLOSED_INPUT_3 )
      Contact( "DB1401_PNEUMATIC_SYSTEM".IN_SERVICE )
      Coil( #CLOSED_3_ALARM )
   END_RUNG
   RUNG wire#powerrail
      I_Contact( #CYL.CLOSE_COMMAND )
      I_Contact( #CLOSE )
      Not()
      Contact( #CYL.TIME_EXCEEDED_ALARM )
      I_Contact( #CLOSED_3_I )
   END_RUNG wire#w1
   RUNG wire#powerrail
      Contact( #CLOSED_3_ALARM )
      I_Contact( "DB2120_MPP_ITC_IPC".RESET_FAULTS )
   END_RUNG wire#w1
   // the same network as SCL:
   #CLOSED_3_ALARM := ((NOT (NOT #CYL.OPEN_COMMAND AND NOT #OPEN) AND #CLOSED_3_I AND #OPENED_3_I AND #CYL.SIMULTANEITY_ALARM) OR (NOT (NOT #CYL.CLOSE_COMMAND AND NOT #CLOSE) AND #CYL.TIME_EXCEEDED_ALARM AND NOT #CLOSED_3_I) OR (#CLOSED_3_ALARM AND NOT "DB2120_MPP_ITC_IPC".RESET_FAULTS)) AND #O_BYTE_0.CLOSED_INPUT_3 AND "DB1401_PNEUMATIC_SYSTEM".IN_SERVICE;
END_REGION

REGION Network 29: CLOSED 4 ALARM
   RUNG wire#powerrail
      I_Contact( #CYL.OPEN_COMMAND )
      I_Contact( #OPEN )
      Not()
      Contact( #CLOSED_4_I )
      Contact( #OPENED_4_I )
      Contact( #CYL.SIMULTANEITY_ALARM )
      wire#w1
      Contact( #O_BYTE_0.CLOSED_INPUT_4 )
      Contact( "DB1401_PNEUMATIC_SYSTEM".IN_SERVICE )
      Coil( #CLOSED_4_ALARM )
   END_RUNG
   RUNG wire#powerrail
      I_Contact( #CYL.CLOSE_COMMAND )
      I_Contact( #CLOSE )
      Not()
      Contact( #CYL.TIME_EXCEEDED_ALARM )
      I_Contact( #CLOSED_4_I )
   END_RUNG wire#w1
   RUNG wire#powerrail
      Contact( #CLOSED_4_ALARM )
      I_Contact( "DB2120_MPP_ITC_IPC".RESET_FAULTS )
   END_RUNG wire#w1
   // the same network as SCL:
   #CLOSED_4_ALARM := ((NOT (NOT #CYL.OPEN_COMMAND AND NOT #OPEN) AND #CLOSED_4_I AND #OPENED_4_I AND #CYL.SIMULTANEITY_ALARM) OR (NOT (NOT #CYL.CLOSE_COMMAND AND NOT #CLOSE) AND #CYL.TIME_EXCEEDED_ALARM AND NOT #CLOSED_4_I) OR (#CLOSED_4_ALARM AND NOT "DB2120_MPP_ITC_IPC".RESET_FAULTS)) AND #O_BYTE_0.CLOSED_INPUT_4 AND "DB1401_PNEUMATIC_SYSTEM".IN_SERVICE;
END_REGION

REGION Network 30: OPEN 1 ALARM
   RUNG wire#powerrail
      I_Contact( #CYL.CLOSE_COMMAND )
      I_Contact( #CLOSE )
      Not()
      Contact( #CLOSED_1_I )
      Contact( #OPENED_1_I )
      Contact( #CYL.SIMULTANEITY_ALARM )
      wire#w1
      Contact( #O_BYTE_0.OPENED_INPUT_1 )
      Contact( "DB1401_PNEUMATIC_SYSTEM".IN_SERVICE )
      Coil( #OPENED_1_ALARM )
   END_RUNG
   RUNG wire#powerrail
      I_Contact( #CYL.OPEN_COMMAND )
      I_Contact( #OPEN )
      Not()
      Contact( #CYL.TIME_EXCEEDED_ALARM )
      I_Contact( #OPENED_1_I )
   END_RUNG wire#w1
   RUNG wire#powerrail
      Contact( #OPENED_1_ALARM )
      I_Contact( "DB2120_MPP_ITC_IPC".RESET_FAULTS )
   END_RUNG wire#w1
   // the same network as SCL:
   #OPENED_1_ALARM := ((NOT (NOT #CYL.CLOSE_COMMAND AND NOT #CLOSE) AND #CLOSED_1_I AND #OPENED_1_I AND #CYL.SIMULTANEITY_ALARM) OR (NOT (NOT #CYL.OPEN_COMMAND AND NOT #OPEN) AND #CYL.TIME_EXCEEDED_ALARM AND NOT #OPENED_1_I) OR (#OPENED_1_ALARM AND NOT "DB2120_MPP_ITC_IPC".RESET_FAULTS)) AND #O_BYTE_0.OPENED_INPUT_1 AND "DB1401_PNEUMATIC_SYSTEM".IN_SERVICE;
END_REGION

REGION Network 31: OPEN 2 ALARM
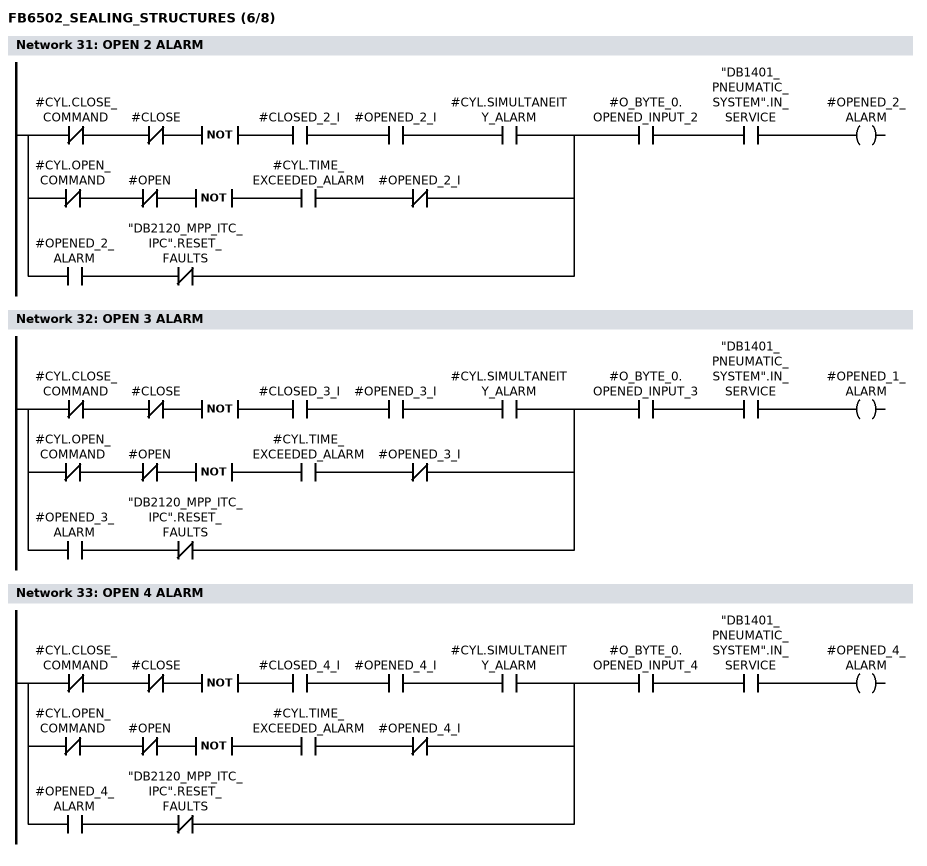
   RUNG wire#powerrail
      I_Contact( #CYL.CLOSE_COMMAND )
      I_Contact( #CLOSE )
      Not()
      Contact( #CLOSED_2_I )
      Contact( #OPENED_2_I )
      Contact( #CYL.SIMULTANEITY_ALARM )
      wire#w1
      Contact( #O_BYTE_0.OPENED_INPUT_2 )
      Contact( "DB1401_PNEUMATIC_SYSTEM".IN_SERVICE )
      Coil( #OPENED_2_ALARM )
   END_RUNG
   RUNG wire#powerrail
      I_Contact( #CYL.OPEN_COMMAND )
      I_Contact( #OPEN )
      Not()
      Contact( #CYL.TIME_EXCEEDED_ALARM )
      I_Contact( #OPENED_2_I )
   END_RUNG wire#w1
   RUNG wire#powerrail
      Contact( #OPENED_2_ALARM )
      I_Contact( "DB2120_MPP_ITC_IPC".RESET_FAULTS )
   END_RUNG wire#w1
   // the same network as SCL:
   #OPENED_2_ALARM := ((NOT (NOT #CYL.CLOSE_COMMAND AND NOT #CLOSE) AND #CLOSED_2_I AND #OPENED_2_I AND #CYL.SIMULTANEITY_ALARM) OR (NOT (NOT #CYL.OPEN_COMMAND AND NOT #OPEN) AND #CYL.TIME_EXCEEDED_ALARM AND NOT #OPENED_2_I) OR (#OPENED_2_ALARM AND NOT "DB2120_MPP_ITC_IPC".RESET_FAULTS)) AND #O_BYTE_0.OPENED_INPUT_2 AND "DB1401_PNEUMATIC_SYSTEM".IN_SERVICE;
END_REGION

REGION Network 32: OPEN 3 ALARM
   RUNG wire#powerrail
      I_Contact( #CYL.CLOSE_COMMAND )
      I_Contact( #CLOSE )
      Not()
      Contact( #CLOSED_3_I )
      Contact( #OPENED_3_I )
      Contact( #CYL.SIMULTANEITY_ALARM )
      wire#w1
      Contact( #O_BYTE_0.OPENED_INPUT_3 )
      Contact( "DB1401_PNEUMATIC_SYSTEM".IN_SERVICE )
      Coil( #OPENED_1_ALARM )
   END_RUNG
   RUNG wire#powerrail
      I_Contact( #CYL.OPEN_COMMAND )
      I_Contact( #OPEN )
      Not()
      Contact( #CYL.TIME_EXCEEDED_ALARM )
      I_Contact( #OPENED_3_I )
   END_RUNG wire#w1
   RUNG wire#powerrail
      Contact( #OPENED_3_ALARM )
      I_Contact( "DB2120_MPP_ITC_IPC".RESET_FAULTS )
   END_RUNG wire#w1
   // the same network as SCL:
   #OPENED_1_ALARM := ((NOT (NOT #CYL.CLOSE_COMMAND AND NOT #CLOSE) AND #CLOSED_3_I AND #OPENED_3_I AND #CYL.SIMULTANEITY_ALARM) OR (NOT (NOT #CYL.OPEN_COMMAND AND NOT #OPEN) AND #CYL.TIME_EXCEEDED_ALARM AND NOT #OPENED_3_I) OR (#OPENED_3_ALARM AND NOT "DB2120_MPP_ITC_IPC".RESET_FAULTS)) AND #O_BYTE_0.OPENED_INPUT_3 AND "DB1401_PNEUMATIC_SYSTEM".IN_SERVICE;
END_REGION

REGION Network 33: OPEN 4 ALARM
   RUNG wire#powerrail
      I_Contact( #CYL.CLOSE_COMMAND )
      I_Contact( #CLOSE )
      Not()
      Contact( #CLOSED_4_I )
      Contact( #OPENED_4_I )
      Contact( #CYL.SIMULTANEITY_ALARM )
      wire#w1
      Contact( #O_BYTE_0.OPENED_INPUT_4 )
      Contact( "DB1401_PNEUMATIC_SYSTEM".IN_SERVICE )
      Coil( #OPENED_4_ALARM )
   END_RUNG
   RUNG wire#powerrail
      I_Contact( #CYL.OPEN_COMMAND )
      I_Contact( #OPEN )
      Not()
      Contact( #CYL.TIME_EXCEEDED_ALARM )
      I_Contact( #OPENED_4_I )
   END_RUNG wire#w1
   RUNG wire#powerrail
      Contact( #OPENED_4_ALARM )
      I_Contact( "DB2120_MPP_ITC_IPC".RESET_FAULTS )
   END_RUNG wire#w1
   // the same network as SCL:
   #OPENED_4_ALARM := ((NOT (NOT #CYL.CLOSE_COMMAND AND NOT #CLOSE) AND #CLOSED_4_I AND #OPENED_4_I AND #CYL.SIMULTANEITY_ALARM) OR (NOT (NOT #CYL.OPEN_COMMAND AND NOT #OPEN) AND #CYL.TIME_EXCEEDED_ALARM AND NOT #OPENED_4_I) OR (#OPENED_4_ALARM AND NOT "DB2120_MPP_ITC_IPC".RESET_FAULTS)) AND #O_BYTE_0.OPENED_INPUT_4 AND "DB1401_PNEUMATIC_SYSTEM".IN_SERVICE;
END_REGION

REGION Network 34: IMMEDIATE STOP AND STOP END OF CYCLE ALARMS
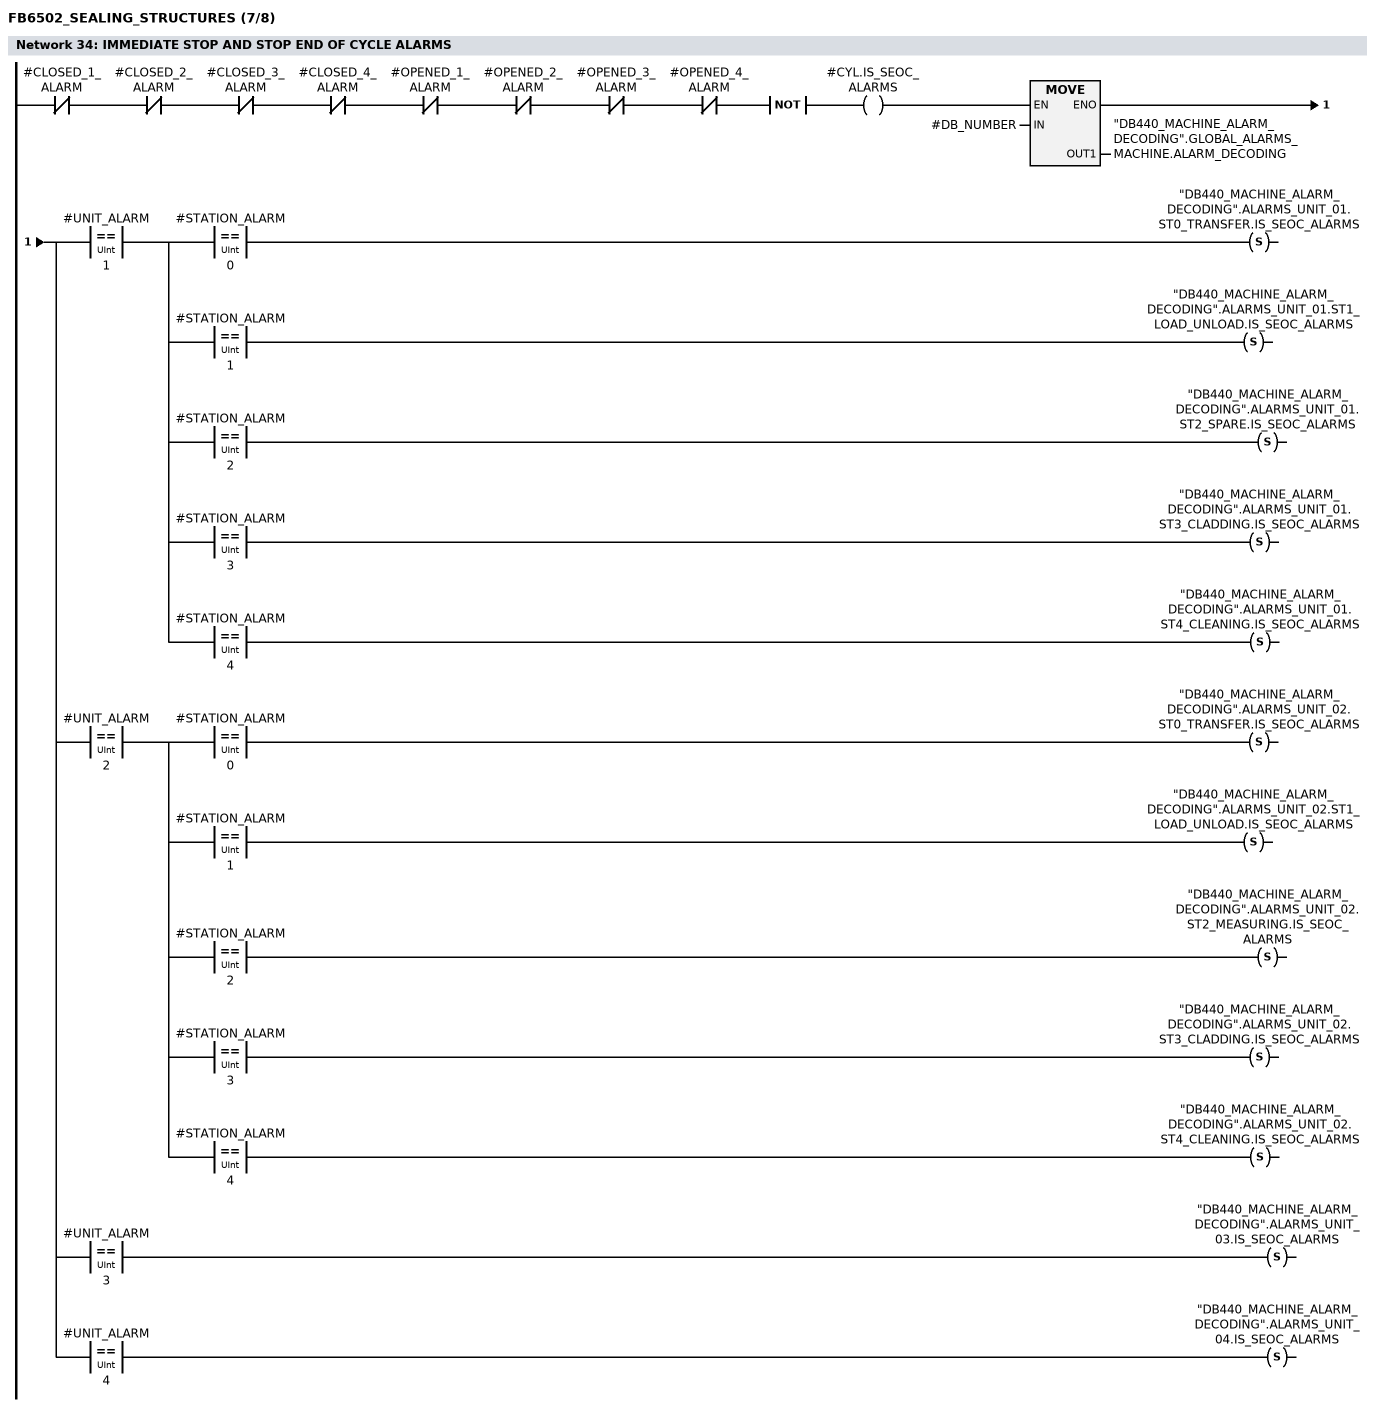
   RUNG wire#powerrail
      I_Contact( #CLOSED_1_ALARM )
      I_Contact( #CLOSED_2_ALARM )
      I_Contact( #CLOSED_3_ALARM )
      I_Contact( #CLOSED_4_ALARM )
      I_Contact( #OPENED_1_ALARM )
      I_Contact( #OPENED_2_ALARM )
      I_Contact( #OPENED_3_ALARM )
      I_Contact( #OPENED_4_ALARM )
      Not()
      Coil( #CYL.IS_SEOC_ALARMS )
      { S7_GenerateENO := "TRUE" } Move(in := #DB_NUMBER, out1 => "DB440_MACHINE_ALARM_DECODING".GLOBAL_ALARMS_MACHINE.ALARM_DECODING)
      wire#w1
      { S7_Templates := "SrcType := UInt" } EQ_Contact(in1 := #UNIT_ALARM, in2 := 1)
      wire#w2
      { S7_Templates := "SrcType := UInt" } EQ_Contact(in1 := #STATION_ALARM, in2 := 0)
      S_Coil( "DB440_MACHINE_ALARM_DECODING".ALARMS_UNIT_01.ST0_TRANSFER.IS_SEOC_ALARMS )
   END_RUNG
   RUNG wire#w2
      { S7_Templates := "SrcType := UInt" } EQ_Contact(in1 := #STATION_ALARM, in2 := 1)
      S_Coil( "DB440_MACHINE_ALARM_DECODING".ALARMS_UNIT_01.ST1_LOAD_UNLOAD.IS_SEOC_ALARMS )
   END_RUNG
   RUNG wire#w2
      { S7_Templates := "SrcType := UInt" } EQ_Contact(in1 := #STATION_ALARM, in2 := 2)
      S_Coil( "DB440_MACHINE_ALARM_DECODING".ALARMS_UNIT_01.ST2_SPARE.IS_SEOC_ALARMS )
   END_RUNG
   RUNG wire#w2
      { S7_Templates := "SrcType := UInt" } EQ_Contact(in1 := #STATION_ALARM, in2 := 3)
      S_Coil( "DB440_MACHINE_ALARM_DECODING".ALARMS_UNIT_01.ST3_CLADDING.IS_SEOC_ALARMS )
   END_RUNG
   RUNG wire#w2
      { S7_Templates := "SrcType := UInt" } EQ_Contact(in1 := #STATION_ALARM, in2 := 4)
      S_Coil( "DB440_MACHINE_ALARM_DECODING".ALARMS_UNIT_01.ST4_CLEANING.IS_SEOC_ALARMS )
   END_RUNG
   RUNG wire#w1
      { S7_Templates := "SrcType := UInt" } EQ_Contact(in1 := #UNIT_ALARM, in2 := 2)
      wire#w3
      { S7_Templates := "SrcType := UInt" } EQ_Contact(in1 := #STATION_ALARM, in2 := 0)
      S_Coil( "DB440_MACHINE_ALARM_DECODING".ALARMS_UNIT_02.ST0_TRANSFER.IS_SEOC_ALARMS )
   END_RUNG
   RUNG wire#w3
      { S7_Templates := "SrcType := UInt" } EQ_Contact(in1 := #STATION_ALARM, in2 := 1)
      S_Coil( "DB440_MACHINE_ALARM_DECODING".ALARMS_UNIT_02.ST1_LOAD_UNLOAD.IS_SEOC_ALARMS )
   END_RUNG
   RUNG wire#w3
      { S7_Templates := "SrcType := UInt" } EQ_Contact(in1 := #STATION_ALARM, in2 := 2)
      S_Coil( "DB440_MACHINE_ALARM_DECODING".ALARMS_UNIT_02.ST2_MEASURING.IS_SEOC_ALARMS )
   END_RUNG
   RUNG wire#w3
      { S7_Templates := "SrcType := UInt" } EQ_Contact(in1 := #STATION_ALARM, in2 := 3)
      S_Coil( "DB440_MACHINE_ALARM_DECODING".ALARMS_UNIT_02.ST3_CLADDING.IS_SEOC_ALARMS )
   END_RUNG
   RUNG wire#w3
      { S7_Templates := "SrcType := UInt" } EQ_Contact(in1 := #STATION_ALARM, in2 := 4)
      S_Coil( "DB440_MACHINE_ALARM_DECODING".ALARMS_UNIT_02.ST4_CLEANING.IS_SEOC_ALARMS )
   END_RUNG
   RUNG wire#w1
      { S7_Templates := "SrcType := UInt" } EQ_Contact(in1 := #UNIT_ALARM, in2 := 3)
      S_Coil( "DB440_MACHINE_ALARM_DECODING".ALARMS_UNIT_03.IS_SEOC_ALARMS )
   END_RUNG
   RUNG wire#w1
      { S7_Templates := "SrcType := UInt" } EQ_Contact(in1 := #UNIT_ALARM, in2 := 4)
      S_Coil( "DB440_MACHINE_ALARM_DECODING".ALARMS_UNIT_04.IS_SEOC_ALARMS )
   END_RUNG
   // the same network as SCL:
   // ENO of a box is taken as its EN; it also drops when the box reports an error
   #CYL.IS_SEOC_ALARMS := NOT (NOT #CLOSED_1_ALARM AND NOT #CLOSED_2_ALARM AND NOT #CLOSED_3_ALARM AND NOT #CLOSED_4_ALARM AND NOT #OPENED_1_ALARM AND NOT #OPENED_2_ALARM AND NOT #OPENED_3_ALARM AND NOT #OPENED_4_ALARM);
   IF #CYL.IS_SEOC_ALARMS THEN
       "DB440_MACHINE_ALARM_DECODING".GLOBAL_ALARMS_MACHINE.ALARM_DECODING := #DB_NUMBER;
   END_IF;
   #_w1 := #CYL.IS_SEOC_ALARMS AND (#UNIT_ALARM = 1);
   IF #_w1 AND (#STATION_ALARM = 0) THEN
       "DB440_MACHINE_ALARM_DECODING".ALARMS_UNIT_01.ST0_TRANSFER.IS_SEOC_ALARMS := TRUE;
   END_IF;
   IF #_w1 AND (#STATION_ALARM = 1) THEN
       "DB440_MACHINE_ALARM_DECODING".ALARMS_UNIT_01.ST1_LOAD_UNLOAD.IS_SEOC_ALARMS := TRUE;
   END_IF;
   IF #_w1 AND (#STATION_ALARM = 2) THEN
       "DB440_MACHINE_ALARM_DECODING".ALARMS_UNIT_01.ST2_SPARE.IS_SEOC_ALARMS := TRUE;
   END_IF;
   IF #_w1 AND (#STATION_ALARM = 3) THEN
       "DB440_MACHINE_ALARM_DECODING".ALARMS_UNIT_01.ST3_CLADDING.IS_SEOC_ALARMS := TRUE;
   END_IF;
   IF #_w1 AND (#STATION_ALARM = 4) THEN
       "DB440_MACHINE_ALARM_DECODING".ALARMS_UNIT_01.ST4_CLEANING.IS_SEOC_ALARMS := TRUE;
   END_IF;
   #_w2 := #CYL.IS_SEOC_ALARMS AND (#UNIT_ALARM = 2);
   IF #_w2 AND (#STATION_ALARM = 0) THEN
       "DB440_MACHINE_ALARM_DECODING".ALARMS_UNIT_02.ST0_TRANSFER.IS_SEOC_ALARMS := TRUE;
   END_IF;
   IF #_w2 AND (#STATION_ALARM = 1) THEN
       "DB440_MACHINE_ALARM_DECODING".ALARMS_UNIT_02.ST1_LOAD_UNLOAD.IS_SEOC_ALARMS := TRUE;
   END_IF;
   IF #_w2 AND (#STATION_ALARM = 2) THEN
       "DB440_MACHINE_ALARM_DECODING".ALARMS_UNIT_02.ST2_MEASURING.IS_SEOC_ALARMS := TRUE;
   END_IF;
   IF #_w2 AND (#STATION_ALARM = 3) THEN
       "DB440_MACHINE_ALARM_DECODING".ALARMS_UNIT_02.ST3_CLADDING.IS_SEOC_ALARMS := TRUE;
   END_IF;
   IF #_w2 AND (#STATION_ALARM = 4) THEN
       "DB440_MACHINE_ALARM_DECODING".ALARMS_UNIT_02.ST4_CLEANING.IS_SEOC_ALARMS := TRUE;
   END_IF;
   IF #CYL.IS_SEOC_ALARMS AND (#UNIT_ALARM = 3) THEN
       "DB440_MACHINE_ALARM_DECODING".ALARMS_UNIT_03.IS_SEOC_ALARMS := TRUE;
   END_IF;
   IF #CYL.IS_SEOC_ALARMS AND (#UNIT_ALARM = 4) THEN
       "DB440_MACHINE_ALARM_DECODING".ALARMS_UNIT_04.IS_SEOC_ALARMS := TRUE;
   END_IF;
END_REGION

REGION Network 35: ANY ACTIVE ALARM
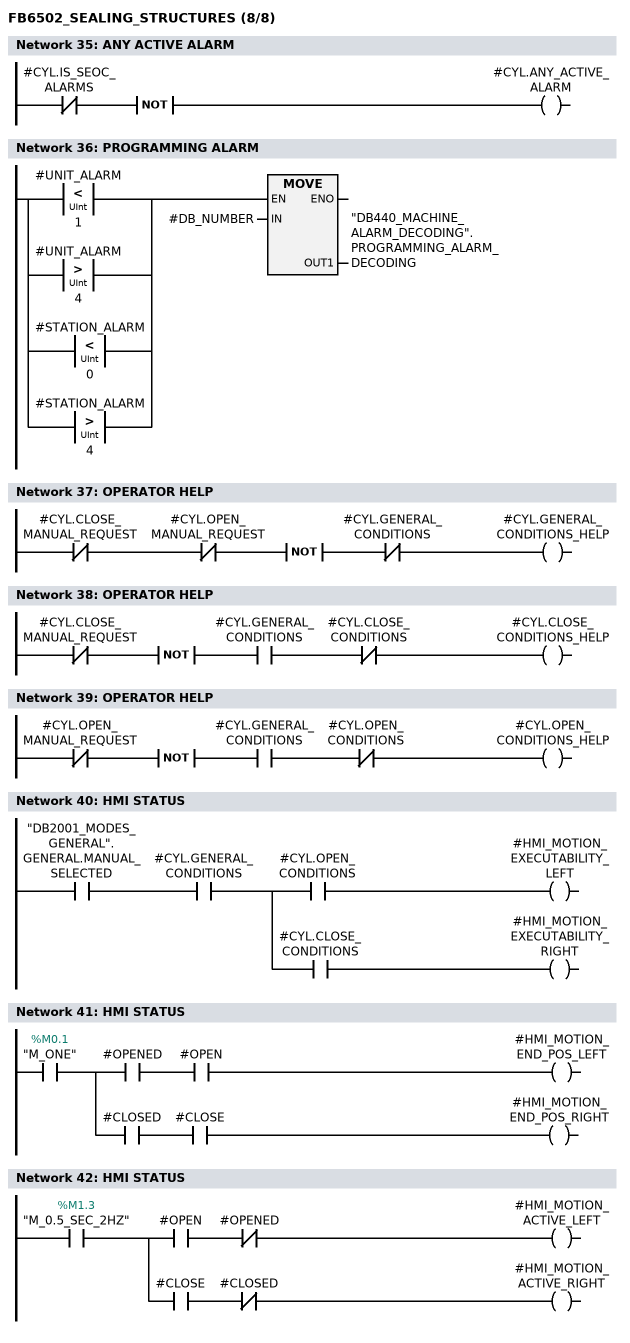
   RUNG wire#powerrail
      I_Contact( #CYL.IS_SEOC_ALARMS )
      Not()
      Coil( #CYL.ANY_ACTIVE_ALARM )
   END_RUNG
   // the same network as SCL:
   #CYL.ANY_ACTIVE_ALARM := NOT (NOT #CYL.IS_SEOC_ALARMS);
END_REGION

REGION Network 36: PROGRAMMING ALARM
   RUNG wire#powerrail
      { S7_Templates := "SrcType := UInt" } LT_Contact(in1 := #UNIT_ALARM, in2 := 1)
      wire#w1
      Move(in := #DB_NUMBER, out1 => "DB440_MACHINE_ALARM_DECODING".PROGRAMMING_ALARM_DECODING)
   END_RUNG
   RUNG wire#powerrail
      { S7_Templates := "SrcType := UInt" } GT_Contact(in1 := #UNIT_ALARM, in2 := 4)
   END_RUNG wire#w1
   RUNG wire#powerrail
      { S7_Templates := "SrcType := UInt" } LT_Contact(in1 := #STATION_ALARM, in2 := 0)
   END_RUNG wire#w1
   RUNG wire#powerrail
      { S7_Templates := "SrcType := UInt" } GT_Contact(in1 := #STATION_ALARM, in2 := 4)
   END_RUNG wire#w1
   // the same network as SCL:
   IF (#UNIT_ALARM < 1) OR (#UNIT_ALARM > 4) OR (#STATION_ALARM < 0) OR (#STATION_ALARM > 4) THEN
       "DB440_MACHINE_ALARM_DECODING".PROGRAMMING_ALARM_DECODING := #DB_NUMBER;
   END_IF;
END_REGION

REGION Network 37: OPERATOR HELP
   RUNG wire#powerrail
      I_Contact( #CYL.CLOSE_MANUAL_REQUEST )
      I_Contact( #CYL.OPEN_MANUAL_REQUEST )
      Not()
      I_Contact( #CYL.GENERAL_CONDITIONS )
      Coil( #CYL.GENERAL_CONDITIONS_HELP )
   END_RUNG
   // the same network as SCL:
   #CYL.GENERAL_CONDITIONS_HELP := NOT (NOT #CYL.CLOSE_MANUAL_REQUEST AND NOT #CYL.OPEN_MANUAL_REQUEST) AND NOT #CYL.GENERAL_CONDITIONS;
END_REGION

REGION Network 38: OPERATOR HELP
   RUNG wire#powerrail
      I_Contact( #CYL.CLOSE_MANUAL_REQUEST )
      Not()
      Contact( #CYL.GENERAL_CONDITIONS )
      I_Contact( #CYL.CLOSE_CONDITIONS )
      Coil( #CYL.CLOSE_CONDITIONS_HELP )
   END_RUNG
   // the same network as SCL:
   #CYL.CLOSE_CONDITIONS_HELP := NOT (NOT #CYL.CLOSE_MANUAL_REQUEST) AND #CYL.GENERAL_CONDITIONS AND NOT #CYL.CLOSE_CONDITIONS;
END_REGION

REGION Network 39: OPERATOR HELP
   RUNG wire#powerrail
      I_Contact( #CYL.OPEN_MANUAL_REQUEST )
      Not()
      Contact( #CYL.GENERAL_CONDITIONS )
      I_Contact( #CYL.OPEN_CONDITIONS )
      Coil( #CYL.OPEN_CONDITIONS_HELP )
   END_RUNG
   // the same network as SCL:
   #CYL.OPEN_CONDITIONS_HELP := NOT (NOT #CYL.OPEN_MANUAL_REQUEST) AND #CYL.GENERAL_CONDITIONS AND NOT #CYL.OPEN_CONDITIONS;
END_REGION

REGION Network 40: HMI STATUS
   RUNG wire#powerrail
      Contact( "DB2001_MODES_GENERAL".GENERAL.MANUAL_SELECTED )
      Contact( #CYL.GENERAL_CONDITIONS )
      wire#w1
      Contact( #CYL.OPEN_CONDITIONS )
      Coil( #HMI_MOTION_EXECUTABILITY_LEFT )
   END_RUNG
   RUNG wire#w1
      Contact( #CYL.CLOSE_CONDITIONS )
      Coil( #HMI_MOTION_EXECUTABILITY_RIGHT )
   END_RUNG
   // the same network as SCL:
   #_w1 := "DB2001_MODES_GENERAL".GENERAL.MANUAL_SELECTED AND #CYL.GENERAL_CONDITIONS;
   #HMI_MOTION_EXECUTABILITY_LEFT := #_w1 AND #CYL.OPEN_CONDITIONS;
   #HMI_MOTION_EXECUTABILITY_RIGHT := #_w1 AND #CYL.CLOSE_CONDITIONS;
END_REGION

REGION Network 41: HMI STATUS
   RUNG wire#powerrail
      Contact( "M_ONE" )
      wire#w1
      Contact( #OPENED )
      Contact( #OPEN )
      Coil( #HMI_MOTION_END_POS_LEFT )
   END_RUNG
   RUNG wire#w1
      Contact( #CLOSED )
      Contact( #CLOSE )
      Coil( #HMI_MOTION_END_POS_RIGHT )
   END_RUNG
   // the same network as SCL:
   #HMI_MOTION_END_POS_LEFT := "M_ONE" AND #OPENED AND #OPEN;
   #HMI_MOTION_END_POS_RIGHT := "M_ONE" AND #CLOSED AND #CLOSE;
END_REGION

REGION Network 42: HMI STATUS
   RUNG wire#powerrail
      Contact( "M_0.5_SEC_2HZ" )
      wire#w1
      Contact( #OPEN )
      I_Contact( #OPENED )
      Coil( #HMI_MOTION_ACTIVE_LEFT )
   END_RUNG
   RUNG wire#w1
      Contact( #CLOSE )
      I_Contact( #CLOSED )
      Coil( #HMI_MOTION_ACTIVE_RIGHT )
   END_RUNG
   // the same network as SCL:
   #HMI_MOTION_ACTIVE_LEFT := "M_0.5_SEC_2HZ" AND #OPEN AND NOT #OPENED;
   #HMI_MOTION_ACTIVE_RIGHT := "M_0.5_SEC_2HZ" AND #CLOSE AND NOT #CLOSED;
END_REGION
END_FUNCTION_BLOCK

FUNCTION_BLOCK "FB6600_SAFETY_BRAKE_Z_AXIS"   // FB6600, LAD
{ S7_Optimized_Access := 'FALSE' }
AUTHOR : ETXETAR
VERSION : 1.0
// stored: AutoNumber false, IsIECCheckEnabled false, SetENOAutomatically false, UDAEnableTagReadback false
   VAR_INPUT
      OPTIONS_0 : Byte := 2#0000_0000;   // OPTION
      BLOCKED_1 : Bool;   // BLOCKED INPUT
      UNBLOCKED_1 : Bool;   // UNBLOCKED INPUT
      MAINT_BLOCKED : Bool;   // MAINTENANCE BLOCKED INPUT
      MAINT_UNBLOCKED : Bool;   // MAINTENANCE UNBLOCKED INPUT
      BLOCK_CONDITIONS : Bool;   // BLOCK CONDITIONS INPUT
      UNBLOCK_CONDITIONS : Bool;   // UNBLOCK CONDITIONS INPUT
      AXIS_SELECTED : Bool;   // AXES SCREEN AXIS SELECTED
      TRAVERSE_COMMAND : Bool;   // TRAVERSE COMMAND FOR THE AXIS
      UNBLOCK_MAN_REQUEST : Bool;   // UNBLOCK MANUAL REQUEST
      BLOCK_AUTO_REQUEST : Bool;   // BLOCK AUTO REQUEST
      UNBLOCK_AUTO_REQUEST : Bool;   // UNBLOCK AUTO REQUEST
      BRAKE_TEST : Bool;   // BRAKE TEST SIGNAL OF THE AXIS
      UNIT_ALARM : UInt;   // UNIT NUMBER MAX. NUMBER=10
      STATION_ALARM : UInt;   // UNIT NUMBER MAX. NUMBER=10
   END_VAR
   VAR_OUTPUT
      BLOCKED : Bool;   // BLOCKED
      UNBLOCKED : Bool;   // UNBLOCKED
      BLOCKED_ALARM : Bool;   // BLOCKED ALARM
      UNBLOCKED_ALARM : Bool;   // UNBLOCKED ALARM
      MAINTENANCE_UNBLOCKED_ALARM : Bool;   // MAINTENANCE UNBLOCKED ALARM
      BLOCK : Bool;   // BLOCK
      UNBLOCK : Bool;   // UNBLOCK
   END_VAR
   VAR DB_SPECIFIC
      BRAKE { S7_SetPoint := 'True'} : "SAFETY_BRAKE";
      TIMER_BLOCKED { S7_SetPoint := 'True'} : TON_TIME;   // BLOCKED TIMER
      TIMER_UNBLOCKED { S7_SetPoint := 'True'} : TON_TIME;   // UNBLOCKED TIMER
      TIMER_SIMULTANEITY { S7_SetPoint := 'True'} : TON_TIME;   // SIMULTANEITY TIMER
      TIMER_TIME_EXCEEDED { S7_SetPoint := 'True'} : TON_TIME;   // TIME EXCEEDED TIMER
   END_VAR
   VAR_TEMP
      INPUTS_MASK : Byte;   // INPUT MASK
      O_BYTE_0 : Struct   // OPTIONS BYTE 0
         MAINTENANCE_SENSORS : Bool;   // MAINTENANCE SENSORS OPTION
         SPARE_1 : Bool;   // SPARE OPTION
         SPARE_2 : Bool;   // SPARE OPTION
         SPARE_3 : Bool;   // SPARE OPTION
         SPARE_4 : Bool;   // SPARE OPTION
         SPARE_5 : Bool;   // SPARE OPTION
         SPARE_6 : Bool;   // SPARE OPTION
         SPARE_7 : Bool;   // SPARE OPTION
      END_STRUCT;
      DB_NUMBER : DInt;   // DB NUMBER FOR ALARM AND HELP DECODING
   END_VAR
   // TIMER_BLOCKED.PT := T#200ms;
   // TIMER_UNBLOCKED.PT := T#150ms;
   // TIMER_SIMULTANEITY.PT := T#20ms;
   // TIMER_TIME_EXCEEDED.PT := T#2S;
   VAR_TEMP   // added for the SCL form of the ladder/FBD networks
      _w1 : Bool;
      _w2 : Bool;
   END_VAR
BEGIN

NETWORK
TITLE = READ INSTANCE DB
      L     DINO;
      +     10#800000;
      T     #DB_NUMBER;


REGION Network 2: OPTIONS
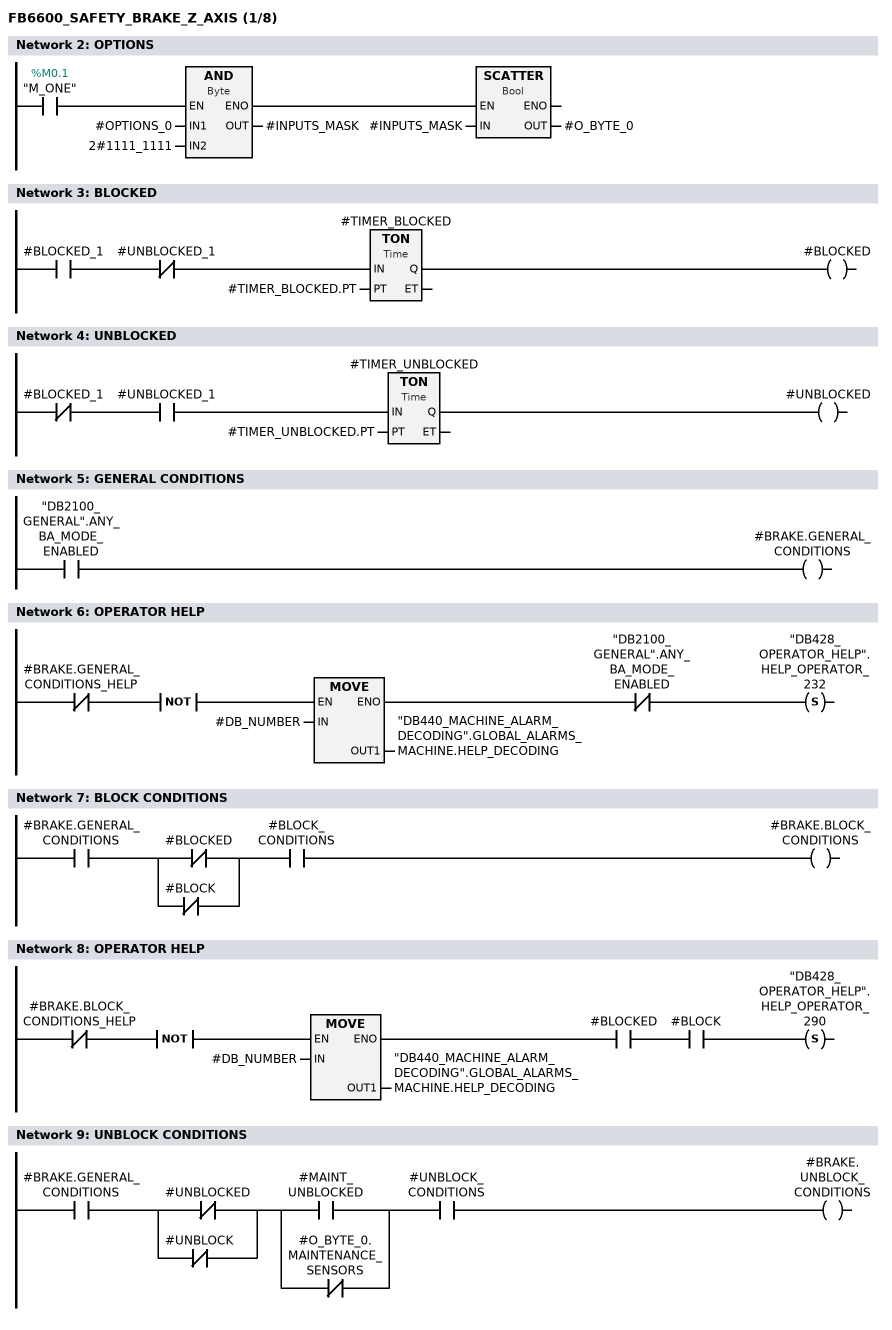
   RUNG wire#powerrail
      Contact( "M_ONE" )
      { S7_Templates := "SrcType := Byte"; S7_GenerateENO := "TRUE" } And(in1 := #OPTIONS_0, in2 := 2#1111_1111, out => #INPUTS_MASK)
      { S7_Templates := "[dest_type := Bool, src_type := Byte]" } SCATTER(IN := #INPUTS_MASK, OUT => #O_BYTE_0)
   END_RUNG
   // the same network as SCL:
   IF "M_ONE" THEN
       #INPUTS_MASK := #OPTIONS_0 AND 2#1111_1111;
       SCATTER(IN := #INPUTS_MASK, OUT => #O_BYTE_0);
   END_IF;
END_REGION

REGION Network 3: BLOCKED
   RUNG wire#powerrail
      Contact( #BLOCKED_1 )
      I_Contact( #UNBLOCKED_1 )
      { S7_Templates := "time_type := Time" } #TIMER_BLOCKED.TON(pt := #TIMER_BLOCKED.PT, et =>)
      Coil( #BLOCKED )
   END_RUNG
   // the same network as SCL:
   #TIMER_BLOCKED(IN := #BLOCKED_1 AND NOT #UNBLOCKED_1, PT := #TIMER_BLOCKED.PT);   // TON
   #BLOCKED := #TIMER_BLOCKED.Q;
END_REGION

REGION Network 4: UNBLOCKED
   RUNG wire#powerrail
      I_Contact( #BLOCKED_1 )
      Contact( #UNBLOCKED_1 )
      { S7_Templates := "time_type := Time" } #TIMER_UNBLOCKED.TON(pt := #TIMER_UNBLOCKED.PT, et =>)
      Coil( #UNBLOCKED )
   END_RUNG
   // the same network as SCL:
   #TIMER_UNBLOCKED(IN := NOT #BLOCKED_1 AND #UNBLOCKED_1, PT := #TIMER_UNBLOCKED.PT);   // TON
   #UNBLOCKED := #TIMER_UNBLOCKED.Q;
END_REGION

REGION Network 5: GENERAL CONDITIONS
   RUNG wire#powerrail
      Contact( "DB2100_GENERAL".ANY_BA_MODE_ENABLED )
      Coil( #BRAKE.GENERAL_CONDITIONS )
   END_RUNG
   // the same network as SCL:
   #BRAKE.GENERAL_CONDITIONS := "DB2100_GENERAL".ANY_BA_MODE_ENABLED;
END_REGION

REGION Network 6: OPERATOR HELP
   RUNG wire#powerrail
      I_Contact( #BRAKE.GENERAL_CONDITIONS_HELP )
      Not()
      { S7_GenerateENO := "TRUE" } Move(in := #DB_NUMBER, out1 => "DB440_MACHINE_ALARM_DECODING".GLOBAL_ALARMS_MACHINE.HELP_DECODING)
      I_Contact( "DB2100_GENERAL".ANY_BA_MODE_ENABLED )
      S_Coil( "DB428_OPERATOR_HELP".HELP_OPERATOR_232 )
   END_RUNG
   // the same network as SCL:
   // ENO of a box is taken as its EN; it also drops when the box reports an error
   #_w1 := NOT (NOT #BRAKE.GENERAL_CONDITIONS_HELP);
   IF #_w1 THEN "DB440_MACHINE_ALARM_DECODING".GLOBAL_ALARMS_MACHINE.HELP_DECODING := #DB_NUMBER; END_IF;
   IF #_w1 AND NOT "DB2100_GENERAL".ANY_BA_MODE_ENABLED THEN
       "DB428_OPERATOR_HELP".HELP_OPERATOR_232 := TRUE;
   END_IF;
END_REGION

REGION Network 7: BLOCK CONDITIONS
   RUNG wire#powerrail
      Contact( #BRAKE.GENERAL_CONDITIONS )
      wire#w1
      I_Contact( #BLOCKED )
      wire#w2
      Contact( #BLOCK_CONDITIONS )
      Coil( #BRAKE.BLOCK_CONDITIONS )
   END_RUNG
   RUNG wire#w1
      I_Contact( #BLOCK )
   END_RUNG wire#w2
   // the same network as SCL:
   #BRAKE.BLOCK_CONDITIONS := #BRAKE.GENERAL_CONDITIONS AND (NOT #BLOCKED OR NOT #BLOCK) AND #BLOCK_CONDITIONS;
END_REGION

REGION Network 8: OPERATOR HELP
   RUNG wire#powerrail
      I_Contact( #BRAKE.BLOCK_CONDITIONS_HELP )
      Not()
      { S7_GenerateENO := "TRUE" } Move(in := #DB_NUMBER, out1 => "DB440_MACHINE_ALARM_DECODING".GLOBAL_ALARMS_MACHINE.HELP_DECODING)
      Contact( #BLOCKED )
      Contact( #BLOCK )
      S_Coil( "DB428_OPERATOR_HELP".HELP_OPERATOR_290 )
   END_RUNG
   // the same network as SCL:
   // ENO of a box is taken as its EN; it also drops when the box reports an error
   #_w1 := NOT (NOT #BRAKE.BLOCK_CONDITIONS_HELP);
   IF #_w1 THEN "DB440_MACHINE_ALARM_DECODING".GLOBAL_ALARMS_MACHINE.HELP_DECODING := #DB_NUMBER; END_IF;
   IF #_w1 AND #BLOCKED AND #BLOCK THEN "DB428_OPERATOR_HELP".HELP_OPERATOR_290 := TRUE; END_IF;
END_REGION

REGION Network 9: UNBLOCK CONDITIONS
   RUNG wire#powerrail
      Contact( #BRAKE.GENERAL_CONDITIONS )
      wire#w1
      I_Contact( #UNBLOCKED )
      wire#w2
      Contact( #MAINT_UNBLOCKED )
      wire#w3
      Contact( #UNBLOCK_CONDITIONS )
      Coil( #BRAKE.UNBLOCK_CONDITIONS )
   END_RUNG
   RUNG wire#w1
      I_Contact( #UNBLOCK )
   END_RUNG wire#w2
   RUNG wire#w2
      I_Contact( #O_BYTE_0.MAINTENANCE_SENSORS )
   END_RUNG wire#w3
   // the same network as SCL:
   #BRAKE.UNBLOCK_CONDITIONS := #BRAKE.GENERAL_CONDITIONS AND (NOT #UNBLOCKED OR NOT #UNBLOCK) AND (#MAINT_UNBLOCKED OR NOT #O_BYTE_0.MAINTENANCE_SENSORS) AND #UNBLOCK_CONDITIONS;
END_REGION

REGION Network 10: OPERATOR HELP
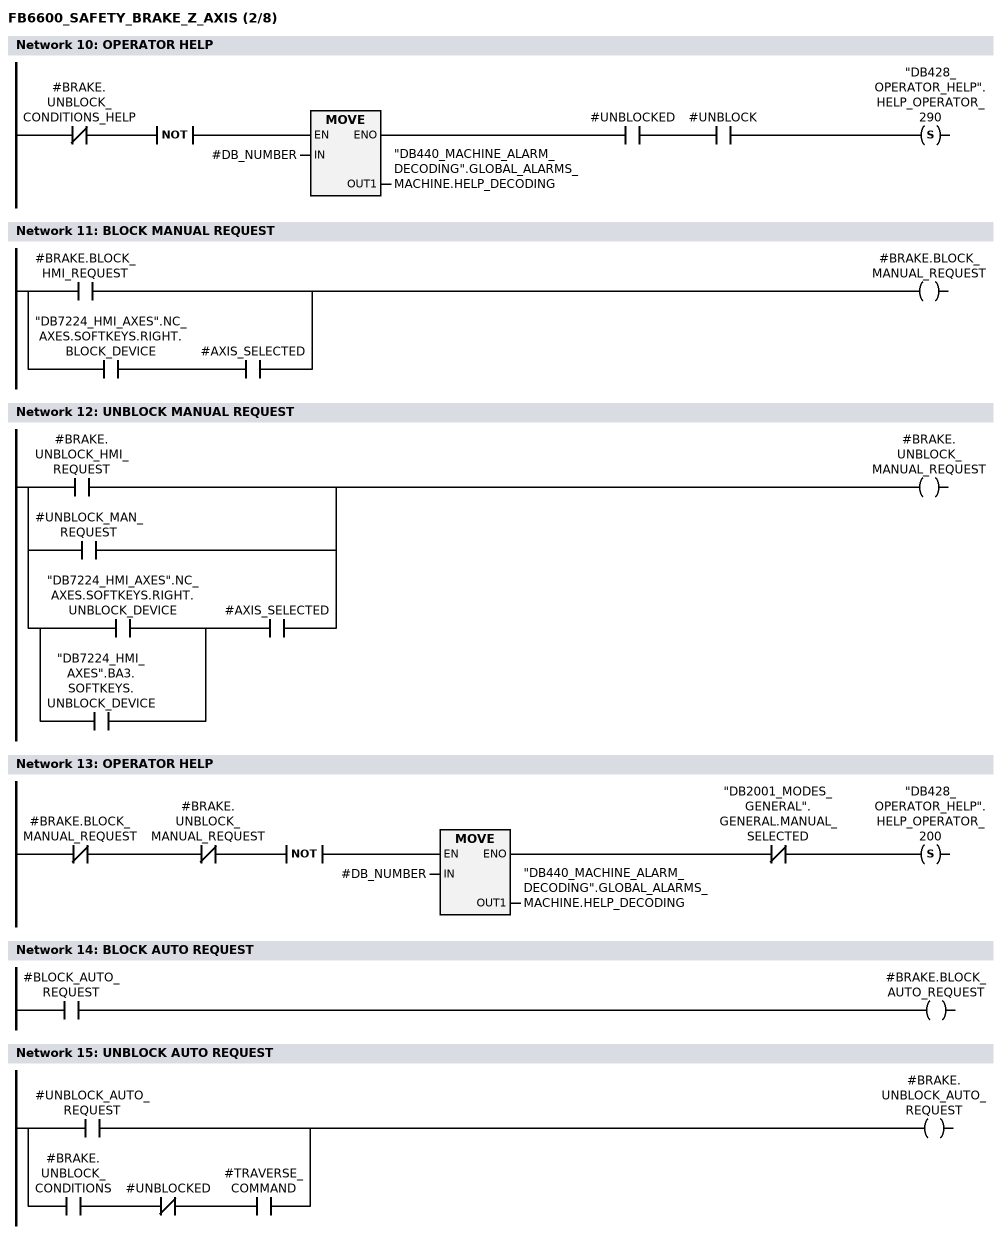
   RUNG wire#powerrail
      I_Contact( #BRAKE.UNBLOCK_CONDITIONS_HELP )
      Not()
      { S7_GenerateENO := "TRUE" } Move(in := #DB_NUMBER, out1 => "DB440_MACHINE_ALARM_DECODING".GLOBAL_ALARMS_MACHINE.HELP_DECODING)
      Contact( #UNBLOCKED )
      Contact( #UNBLOCK )
      S_Coil( "DB428_OPERATOR_HELP".HELP_OPERATOR_290 )
   END_RUNG
   // the same network as SCL:
   // ENO of a box is taken as its EN; it also drops when the box reports an error
   #_w1 := NOT (NOT #BRAKE.UNBLOCK_CONDITIONS_HELP);
   IF #_w1 THEN "DB440_MACHINE_ALARM_DECODING".GLOBAL_ALARMS_MACHINE.HELP_DECODING := #DB_NUMBER; END_IF;
   IF #_w1 AND #UNBLOCKED AND #UNBLOCK THEN "DB428_OPERATOR_HELP".HELP_OPERATOR_290 := TRUE; END_IF;
END_REGION

REGION Network 11: BLOCK MANUAL REQUEST
   RUNG wire#powerrail
      Contact( #BRAKE.BLOCK_HMI_REQUEST )
      wire#w1
      Coil( #BRAKE.BLOCK_MANUAL_REQUEST )
   END_RUNG
   RUNG wire#powerrail
      Contact( "DB7224_HMI_AXES".NC_AXES.SOFTKEYS.RIGHT.BLOCK_DEVICE )
      Contact( #AXIS_SELECTED )
   END_RUNG wire#w1
   // the same network as SCL:
   #BRAKE.BLOCK_MANUAL_REQUEST := #BRAKE.BLOCK_HMI_REQUEST OR ("DB7224_HMI_AXES".NC_AXES.SOFTKEYS.RIGHT.BLOCK_DEVICE AND #AXIS_SELECTED);
END_REGION

REGION Network 12: UNBLOCK MANUAL REQUEST
   RUNG wire#powerrail
      Contact( #BRAKE.UNBLOCK_HMI_REQUEST )
      wire#w1
      Coil( #BRAKE.UNBLOCK_MANUAL_REQUEST )
   END_RUNG
   RUNG wire#powerrail
      Contact( #UNBLOCK_MAN_REQUEST )
   END_RUNG wire#w1
   RUNG wire#powerrail
      Contact( "DB7224_HMI_AXES".NC_AXES.SOFTKEYS.RIGHT.UNBLOCK_DEVICE )
      wire#w2
      Contact( #AXIS_SELECTED )
   END_RUNG wire#w1
   RUNG wire#powerrail
      Contact( "DB7224_HMI_AXES".BA3.SOFTKEYS.UNBLOCK_DEVICE )
   END_RUNG wire#w2
   // the same network as SCL:
   #BRAKE.UNBLOCK_MANUAL_REQUEST := #BRAKE.UNBLOCK_HMI_REQUEST OR #UNBLOCK_MAN_REQUEST OR (("DB7224_HMI_AXES".NC_AXES.SOFTKEYS.RIGHT.UNBLOCK_DEVICE OR "DB7224_HMI_AXES".BA3.SOFTKEYS.UNBLOCK_DEVICE) AND #AXIS_SELECTED);
END_REGION

REGION Network 13: OPERATOR HELP
   RUNG wire#powerrail
      I_Contact( #BRAKE.BLOCK_MANUAL_REQUEST )
      I_Contact( #BRAKE.UNBLOCK_MANUAL_REQUEST )
      Not()
      { S7_GenerateENO := "TRUE" } Move(in := #DB_NUMBER, out1 => "DB440_MACHINE_ALARM_DECODING".GLOBAL_ALARMS_MACHINE.HELP_DECODING)
      I_Contact( "DB2001_MODES_GENERAL".GENERAL.MANUAL_SELECTED )
      S_Coil( "DB428_OPERATOR_HELP".HELP_OPERATOR_200 )
   END_RUNG
   // the same network as SCL:
   // ENO of a box is taken as its EN; it also drops when the box reports an error
   #_w1 := NOT (NOT #BRAKE.BLOCK_MANUAL_REQUEST AND NOT #BRAKE.UNBLOCK_MANUAL_REQUEST);
   IF #_w1 THEN "DB440_MACHINE_ALARM_DECODING".GLOBAL_ALARMS_MACHINE.HELP_DECODING := #DB_NUMBER; END_IF;
   IF #_w1 AND NOT "DB2001_MODES_GENERAL".GENERAL.MANUAL_SELECTED THEN
       "DB428_OPERATOR_HELP".HELP_OPERATOR_200 := TRUE;
   END_IF;
END_REGION

REGION Network 14: BLOCK AUTO REQUEST
   RUNG wire#powerrail
      Contact( #BLOCK_AUTO_REQUEST )
      Coil( #BRAKE.BLOCK_AUTO_REQUEST )
   END_RUNG
   // the same network as SCL:
   #BRAKE.BLOCK_AUTO_REQUEST := #BLOCK_AUTO_REQUEST;
END_REGION

REGION Network 15: UNBLOCK AUTO REQUEST
   RUNG wire#powerrail
      Contact( #UNBLOCK_AUTO_REQUEST )
      wire#w1
      Coil( #BRAKE.UNBLOCK_AUTO_REQUEST )
   END_RUNG
   RUNG wire#powerrail
      Contact( #BRAKE.UNBLOCK_CONDITIONS )
      I_Contact( #UNBLOCKED )
      Contact( #TRAVERSE_COMMAND )
   END_RUNG wire#w1
   // the same network as SCL:
   #BRAKE.UNBLOCK_AUTO_REQUEST := #UNBLOCK_AUTO_REQUEST OR (#BRAKE.UNBLOCK_CONDITIONS AND NOT #UNBLOCKED AND #TRAVERSE_COMMAND);
END_REGION

REGION Network 16: BLOCK GLOBAL REQUEST
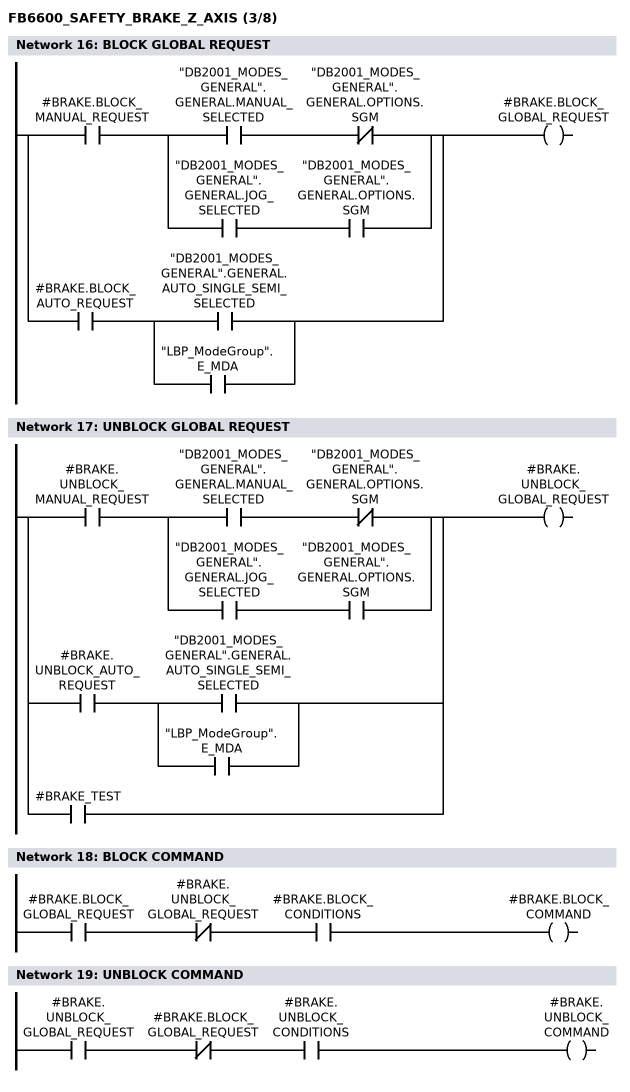
   RUNG wire#powerrail
      Contact( #BRAKE.BLOCK_MANUAL_REQUEST )
      wire#w1
      Contact( "DB2001_MODES_GENERAL".GENERAL.MANUAL_SELECTED )
      I_Contact( "DB2001_MODES_GENERAL".GENERAL.OPTIONS.SGM )
      wire#w2
      Coil( #BRAKE.BLOCK_GLOBAL_REQUEST )
   END_RUNG
   RUNG wire#w1
      Contact( "DB2001_MODES_GENERAL".GENERAL.JOG_SELECTED )
      Contact( "DB2001_MODES_GENERAL".GENERAL.OPTIONS.SGM )
   END_RUNG wire#w2
   RUNG wire#powerrail
      Contact( #BRAKE.BLOCK_AUTO_REQUEST )
      wire#w3
      Contact( "DB2001_MODES_GENERAL".GENERAL.AUTO_SINGLE_SEMI_SELECTED )
   END_RUNG wire#w2
   RUNG wire#w3
      Contact( "LBP_ModeGroup".E_MDA )
   END_RUNG wire#w2
   // the same network as SCL:
   #BRAKE.BLOCK_GLOBAL_REQUEST := (#BRAKE.BLOCK_MANUAL_REQUEST AND (("DB2001_MODES_GENERAL".GENERAL.MANUAL_SELECTED AND NOT "DB2001_MODES_GENERAL".GENERAL.OPTIONS.SGM) OR ("DB2001_MODES_GENERAL".GENERAL.JOG_SELECTED AND "DB2001_MODES_GENERAL".GENERAL.OPTIONS.SGM))) OR (#BRAKE.BLOCK_AUTO_REQUEST AND ("DB2001_MODES_GENERAL".GENERAL.AUTO_SINGLE_SEMI_SELECTED OR "LBP_ModeGroup".E_MDA));
END_REGION

REGION Network 17: UNBLOCK GLOBAL REQUEST
   RUNG wire#powerrail
      Contact( #BRAKE.UNBLOCK_MANUAL_REQUEST )
      wire#w1
      Contact( "DB2001_MODES_GENERAL".GENERAL.MANUAL_SELECTED )
      I_Contact( "DB2001_MODES_GENERAL".GENERAL.OPTIONS.SGM )
      wire#w2
      Coil( #BRAKE.UNBLOCK_GLOBAL_REQUEST )
   END_RUNG
   RUNG wire#w1
      Contact( "DB2001_MODES_GENERAL".GENERAL.JOG_SELECTED )
      Contact( "DB2001_MODES_GENERAL".GENERAL.OPTIONS.SGM )
   END_RUNG wire#w2
   RUNG wire#powerrail
      Contact( #BRAKE.UNBLOCK_AUTO_REQUEST )
      wire#w3
      Contact( "DB2001_MODES_GENERAL".GENERAL.AUTO_SINGLE_SEMI_SELECTED )
   END_RUNG wire#w2
   RUNG wire#w3
      Contact( "LBP_ModeGroup".E_MDA )
   END_RUNG wire#w2
   RUNG wire#powerrail
      Contact( #BRAKE_TEST )
   END_RUNG wire#w2
   // the same network as SCL:
   #BRAKE.UNBLOCK_GLOBAL_REQUEST := (#BRAKE.UNBLOCK_MANUAL_REQUEST AND (("DB2001_MODES_GENERAL".GENERAL.MANUAL_SELECTED AND NOT "DB2001_MODES_GENERAL".GENERAL.OPTIONS.SGM) OR ("DB2001_MODES_GENERAL".GENERAL.JOG_SELECTED AND "DB2001_MODES_GENERAL".GENERAL.OPTIONS.SGM))) OR (#BRAKE.UNBLOCK_AUTO_REQUEST AND ("DB2001_MODES_GENERAL".GENERAL.AUTO_SINGLE_SEMI_SELECTED OR "LBP_ModeGroup".E_MDA)) OR #BRAKE_TEST;
END_REGION

REGION Network 18: BLOCK COMMAND
   RUNG wire#powerrail
      Contact( #BRAKE.BLOCK_GLOBAL_REQUEST )
      I_Contact( #BRAKE.UNBLOCK_GLOBAL_REQUEST )
      Contact( #BRAKE.BLOCK_CONDITIONS )
      Coil( #BRAKE.BLOCK_COMMAND )
   END_RUNG
   // the same network as SCL:
   #BRAKE.BLOCK_COMMAND := #BRAKE.BLOCK_GLOBAL_REQUEST AND NOT #BRAKE.UNBLOCK_GLOBAL_REQUEST AND #BRAKE.BLOCK_CONDITIONS;
END_REGION

REGION Network 19: UNBLOCK COMMAND
   RUNG wire#powerrail
      Contact( #BRAKE.UNBLOCK_GLOBAL_REQUEST )
      I_Contact( #BRAKE.BLOCK_GLOBAL_REQUEST )
      Contact( #BRAKE.UNBLOCK_CONDITIONS )
      Coil( #BRAKE.UNBLOCK_COMMAND )
   END_RUNG
   // the same network as SCL:
   #BRAKE.UNBLOCK_COMMAND := #BRAKE.UNBLOCK_GLOBAL_REQUEST AND NOT #BRAKE.BLOCK_GLOBAL_REQUEST AND #BRAKE.UNBLOCK_CONDITIONS;
END_REGION

REGION Network 20: BLOCK
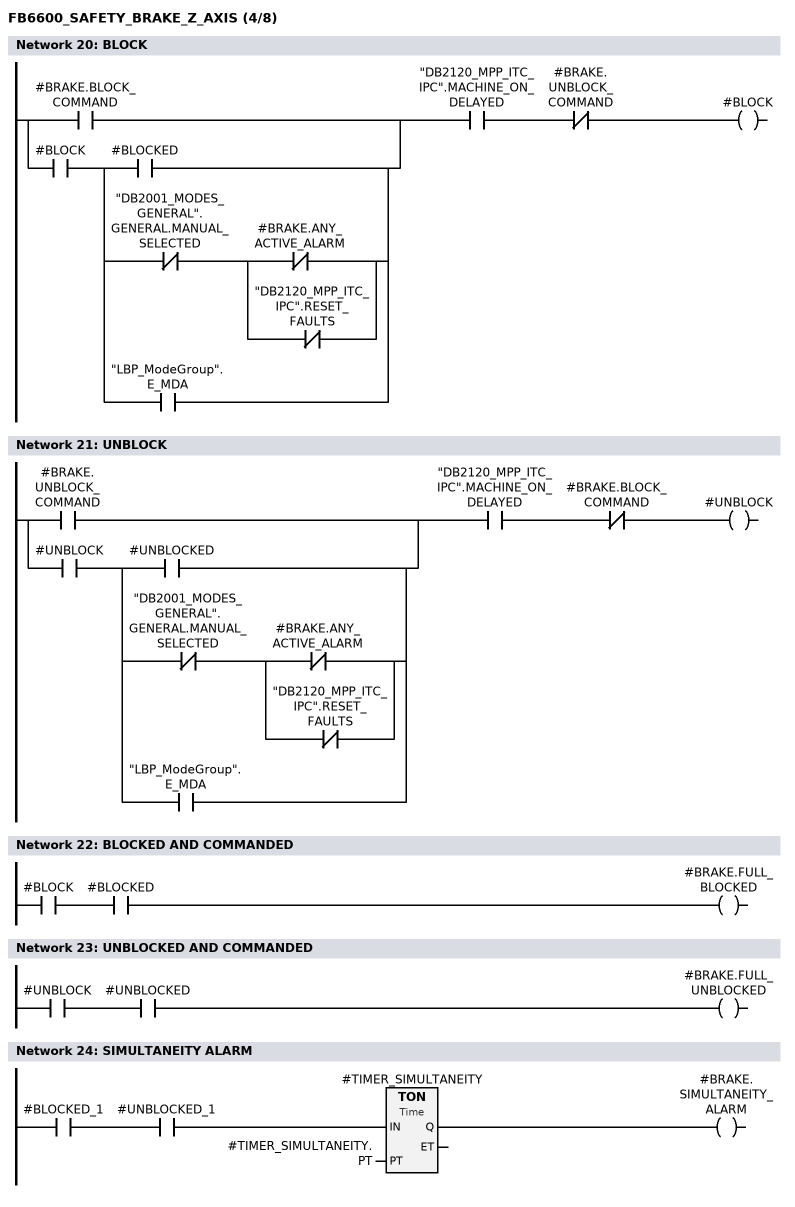
   RUNG wire#powerrail
      Contact( #BRAKE.BLOCK_COMMAND )
      wire#w1
      Contact( "DB2120_MPP_ITC_IPC".MACHINE_ON_DELAYED )
      I_Contact( #BRAKE.UNBLOCK_COMMAND )
      Coil( #BLOCK )
   END_RUNG
   RUNG wire#powerrail
      Contact( #BLOCK )
      wire#w2
      Contact( #BLOCKED )
   END_RUNG wire#w1
   RUNG wire#w2
      I_Contact( "DB2001_MODES_GENERAL".GENERAL.MANUAL_SELECTED )
      wire#w3
      I_Contact( #BRAKE.ANY_ACTIVE_ALARM )
   END_RUNG wire#w1
   RUNG wire#w3
      I_Contact( "DB2120_MPP_ITC_IPC".RESET_FAULTS )
   END_RUNG wire#w1
   RUNG wire#w2
      Contact( "LBP_ModeGroup".E_MDA )
   END_RUNG wire#w1
   // the same network as SCL:
   #BLOCK := (#BRAKE.BLOCK_COMMAND OR (#BLOCK AND (#BLOCKED OR (NOT "DB2001_MODES_GENERAL".GENERAL.MANUAL_SELECTED AND (NOT #BRAKE.ANY_ACTIVE_ALARM OR NOT "DB2120_MPP_ITC_IPC".RESET_FAULTS)) OR "LBP_ModeGroup".E_MDA))) AND "DB2120_MPP_ITC_IPC".MACHINE_ON_DELAYED AND NOT #BRAKE.UNBLOCK_COMMAND;
END_REGION

REGION Network 21: UNBLOCK
   RUNG wire#powerrail
      Contact( #BRAKE.UNBLOCK_COMMAND )
      wire#w1
      Contact( "DB2120_MPP_ITC_IPC".MACHINE_ON_DELAYED )
      I_Contact( #BRAKE.BLOCK_COMMAND )
      Coil( #UNBLOCK )
   END_RUNG
   RUNG wire#powerrail
      Contact( #UNBLOCK )
      wire#w2
      Contact( #UNBLOCKED )
   END_RUNG wire#w1
   RUNG wire#w2
      I_Contact( "DB2001_MODES_GENERAL".GENERAL.MANUAL_SELECTED )
      wire#w3
      I_Contact( #BRAKE.ANY_ACTIVE_ALARM )
   END_RUNG wire#w1
   RUNG wire#w3
      I_Contact( "DB2120_MPP_ITC_IPC".RESET_FAULTS )
   END_RUNG wire#w1
   RUNG wire#w2
      Contact( "LBP_ModeGroup".E_MDA )
   END_RUNG wire#w1
   // the same network as SCL:
   #UNBLOCK := (#BRAKE.UNBLOCK_COMMAND OR (#UNBLOCK AND (#UNBLOCKED OR (NOT "DB2001_MODES_GENERAL".GENERAL.MANUAL_SELECTED AND (NOT #BRAKE.ANY_ACTIVE_ALARM OR NOT "DB2120_MPP_ITC_IPC".RESET_FAULTS)) OR "LBP_ModeGroup".E_MDA))) AND "DB2120_MPP_ITC_IPC".MACHINE_ON_DELAYED AND NOT #BRAKE.BLOCK_COMMAND;
END_REGION

REGION Network 22: BLOCKED AND COMMANDED
   RUNG wire#powerrail
      Contact( #BLOCK )
      Contact( #BLOCKED )
      Coil( #BRAKE.FULL_BLOCKED )
   END_RUNG
   // the same network as SCL:
   #BRAKE.FULL_BLOCKED := #BLOCK AND #BLOCKED;
END_REGION

REGION Network 23: UNBLOCKED AND COMMANDED
   RUNG wire#powerrail
      Contact( #UNBLOCK )
      Contact( #UNBLOCKED )
      Coil( #BRAKE.FULL_UNBLOCKED )
   END_RUNG
   // the same network as SCL:
   #BRAKE.FULL_UNBLOCKED := #UNBLOCK AND #UNBLOCKED;
END_REGION

REGION Network 24: SIMULTANEITY ALARM
   RUNG wire#powerrail
      Contact( #BLOCKED_1 )
      Contact( #UNBLOCKED_1 )
      { S7_Templates := "time_type := Time" } #TIMER_SIMULTANEITY.TON(pt := #TIMER_SIMULTANEITY.PT, et =>)
      Coil( #BRAKE.SIMULTANEITY_ALARM )
   END_RUNG
   // the same network as SCL:
   #TIMER_SIMULTANEITY(IN := #BLOCKED_1 AND #UNBLOCKED_1, PT := #TIMER_SIMULTANEITY.PT);   // TON
   #BRAKE.SIMULTANEITY_ALARM := #TIMER_SIMULTANEITY.Q;
END_REGION

REGION Network 25: TIME EXCEEDED ALARM
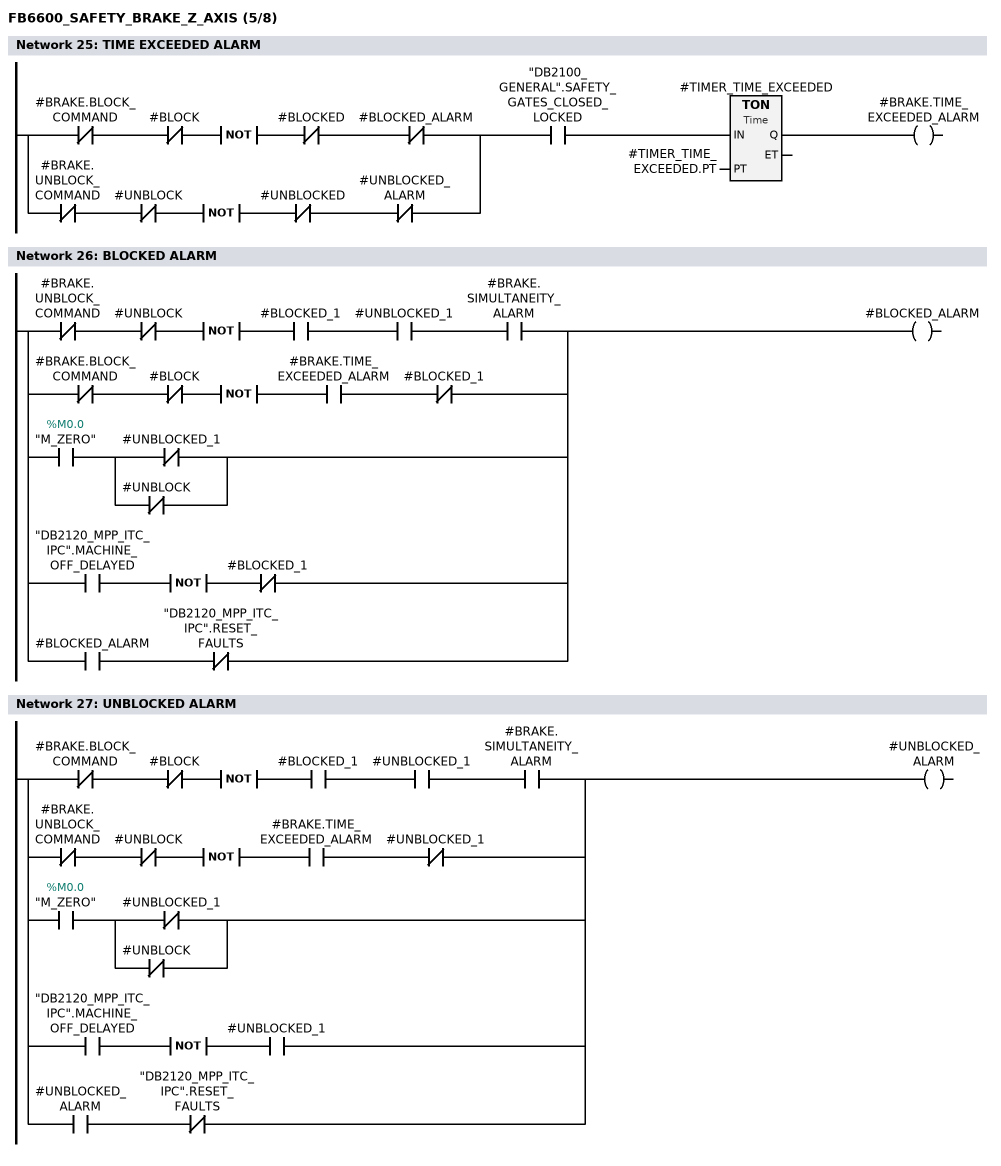
   RUNG wire#powerrail
      I_Contact( #BRAKE.BLOCK_COMMAND )
      I_Contact( #BLOCK )
      Not()
      I_Contact( #BLOCKED )
      I_Contact( #BLOCKED_ALARM )
      wire#w1
      Contact( "DB2100_GENERAL".SAFETY_GATES_CLOSED_LOCKED )
      { S7_Templates := "time_type := Time" } #TIMER_TIME_EXCEEDED.TON(pt := #TIMER_TIME_EXCEEDED.PT, et =>)
      Coil( #BRAKE.TIME_EXCEEDED_ALARM )
   END_RUNG
   RUNG wire#powerrail
      I_Contact( #BRAKE.UNBLOCK_COMMAND )
      I_Contact( #UNBLOCK )
      Not()
      I_Contact( #UNBLOCKED )
      I_Contact( #UNBLOCKED_ALARM )
   END_RUNG wire#w1
   // the same network as SCL:
   #TIMER_TIME_EXCEEDED(IN := ((NOT (NOT #BRAKE.BLOCK_COMMAND AND NOT #BLOCK) AND NOT #BLOCKED AND NOT #BLOCKED_ALARM) OR (NOT (NOT #BRAKE.UNBLOCK_COMMAND AND NOT #UNBLOCK) AND NOT #UNBLOCKED AND NOT #UNBLOCKED_ALARM)) AND "DB2100_GENERAL".SAFETY_GATES_CLOSED_LOCKED,   // TON
                        PT := #TIMER_TIME_EXCEEDED.PT);
   #BRAKE.TIME_EXCEEDED_ALARM := #TIMER_TIME_EXCEEDED.Q;
END_REGION

REGION Network 26: BLOCKED ALARM
   RUNG wire#powerrail
      I_Contact( #BRAKE.UNBLOCK_COMMAND )
      I_Contact( #UNBLOCK )
      Not()
      Contact( #BLOCKED_1 )
      Contact( #UNBLOCKED_1 )
      Contact( #BRAKE.SIMULTANEITY_ALARM )
      wire#w1
      Coil( #BLOCKED_ALARM )
   END_RUNG
   RUNG wire#powerrail
      I_Contact( #BRAKE.BLOCK_COMMAND )
      I_Contact( #BLOCK )
      Not()
      Contact( #BRAKE.TIME_EXCEEDED_ALARM )
      I_Contact( #BLOCKED_1 )
   END_RUNG wire#w1
   RUNG wire#powerrail
      Contact( "M_ZERO" )
      wire#w2
      I_Contact( #UNBLOCKED_1 )
   END_RUNG wire#w1
   RUNG wire#w2
      I_Contact( #UNBLOCK )
   END_RUNG wire#w1
   RUNG wire#powerrail
      Contact( "DB2120_MPP_ITC_IPC".MACHINE_OFF_DELAYED )
      Not()
      I_Contact( #BLOCKED_1 )
   END_RUNG wire#w1
   RUNG wire#powerrail
      Contact( #BLOCKED_ALARM )
      I_Contact( "DB2120_MPP_ITC_IPC".RESET_FAULTS )
   END_RUNG wire#w1
   // the same network as SCL:
   #BLOCKED_ALARM := (NOT (NOT #BRAKE.UNBLOCK_COMMAND AND NOT #UNBLOCK) AND #BLOCKED_1 AND #UNBLOCKED_1 AND #BRAKE.SIMULTANEITY_ALARM) OR (NOT (NOT #BRAKE.BLOCK_COMMAND AND NOT #BLOCK) AND #BRAKE.TIME_EXCEEDED_ALARM AND NOT #BLOCKED_1) OR ("M_ZERO" AND (NOT #UNBLOCKED_1 OR NOT #UNBLOCK)) OR (NOT "DB2120_MPP_ITC_IPC".MACHINE_OFF_DELAYED AND NOT #BLOCKED_1) OR (#BLOCKED_ALARM AND NOT "DB2120_MPP_ITC_IPC".RESET_FAULTS);
END_REGION

REGION Network 27: UNBLOCKED ALARM
   RUNG wire#powerrail
      I_Contact( #BRAKE.BLOCK_COMMAND )
      I_Contact( #BLOCK )
      Not()
      Contact( #BLOCKED_1 )
      Contact( #UNBLOCKED_1 )
      Contact( #BRAKE.SIMULTANEITY_ALARM )
      wire#w1
      Coil( #UNBLOCKED_ALARM )
   END_RUNG
   RUNG wire#powerrail
      I_Contact( #BRAKE.UNBLOCK_COMMAND )
      I_Contact( #UNBLOCK )
      Not()
      Contact( #BRAKE.TIME_EXCEEDED_ALARM )
      I_Contact( #UNBLOCKED_1 )
   END_RUNG wire#w1
   RUNG wire#powerrail
      Contact( "M_ZERO" )
      wire#w2
      I_Contact( #UNBLOCKED_1 )
   END_RUNG wire#w1
   RUNG wire#w2
      I_Contact( #UNBLOCK )
   END_RUNG wire#w1
   RUNG wire#powerrail
      Contact( "DB2120_MPP_ITC_IPC".MACHINE_OFF_DELAYED )
      Not()
      Contact( #UNBLOCKED_1 )
   END_RUNG wire#w1
   RUNG wire#powerrail
      Contact( #UNBLOCKED_ALARM )
      I_Contact( "DB2120_MPP_ITC_IPC".RESET_FAULTS )
   END_RUNG wire#w1
   // the same network as SCL:
   #UNBLOCKED_ALARM := (NOT (NOT #BRAKE.BLOCK_COMMAND AND NOT #BLOCK) AND #BLOCKED_1 AND #UNBLOCKED_1 AND #BRAKE.SIMULTANEITY_ALARM) OR (NOT (NOT #BRAKE.UNBLOCK_COMMAND AND NOT #UNBLOCK) AND #BRAKE.TIME_EXCEEDED_ALARM AND NOT #UNBLOCKED_1) OR ("M_ZERO" AND (NOT #UNBLOCKED_1 OR NOT #UNBLOCK)) OR (NOT "DB2120_MPP_ITC_IPC".MACHINE_OFF_DELAYED AND #UNBLOCKED_1) OR (#UNBLOCKED_ALARM AND NOT "DB2120_MPP_ITC_IPC".RESET_FAULTS);
END_REGION

REGION Network 28: MAINTENANCE UNBLOCKED ALARM
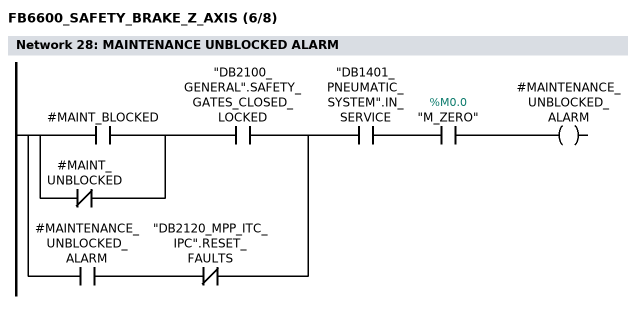
   RUNG wire#powerrail
      Contact( #MAINT_BLOCKED )
      wire#w1
      Contact( "DB2100_GENERAL".SAFETY_GATES_CLOSED_LOCKED )
      wire#w2
      Contact( "DB1401_PNEUMATIC_SYSTEM".IN_SERVICE )
      Contact( "M_ZERO" )
      Coil( #MAINTENANCE_UNBLOCKED_ALARM )
   END_RUNG
   RUNG wire#powerrail
      I_Contact( #MAINT_UNBLOCKED )
   END_RUNG wire#w1
   RUNG wire#powerrail
      Contact( #MAINTENANCE_UNBLOCKED_ALARM )
      I_Contact( "DB2120_MPP_ITC_IPC".RESET_FAULTS )
   END_RUNG wire#w2
   // the same network as SCL:
   #MAINTENANCE_UNBLOCKED_ALARM := (((#MAINT_BLOCKED OR NOT #MAINT_UNBLOCKED) AND "DB2100_GENERAL".SAFETY_GATES_CLOSED_LOCKED) OR (#MAINTENANCE_UNBLOCKED_ALARM AND NOT "DB2120_MPP_ITC_IPC".RESET_FAULTS)) AND "DB1401_PNEUMATIC_SYSTEM".IN_SERVICE AND "M_ZERO";
END_REGION

REGION Network 29: IMMEDIATE STOP AND STOP END OF CYCLE ALARMS
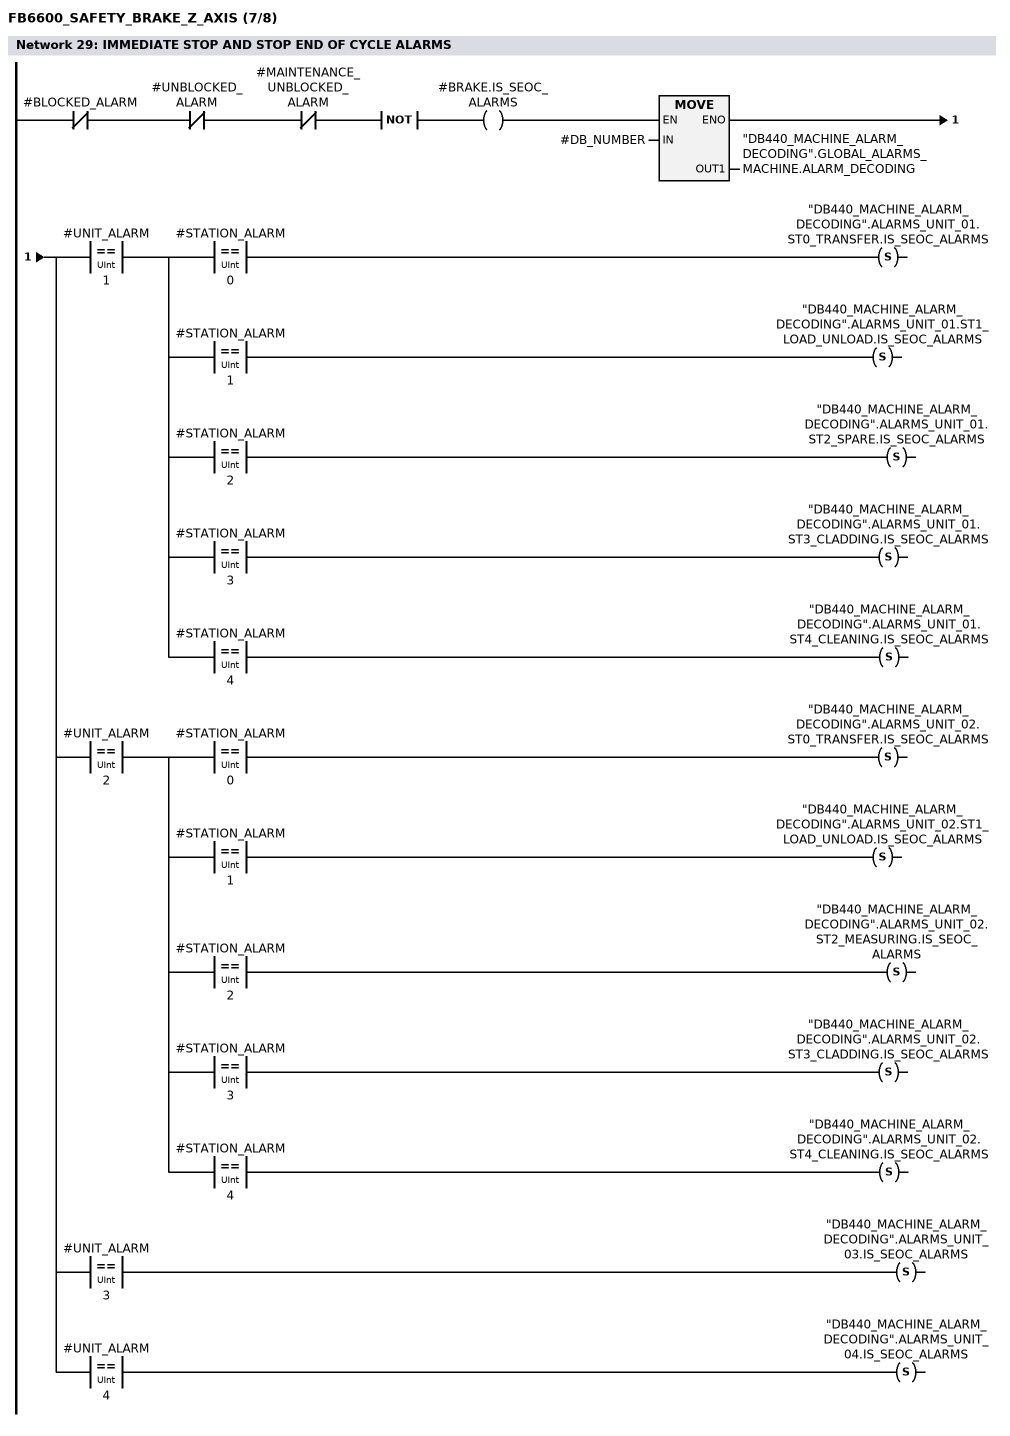
   RUNG wire#powerrail
      I_Contact( #BLOCKED_ALARM )
      I_Contact( #UNBLOCKED_ALARM )
      I_Contact( #MAINTENANCE_UNBLOCKED_ALARM )
      Not()
      Coil( #BRAKE.IS_SEOC_ALARMS )
      { S7_GenerateENO := "TRUE" } Move(in := #DB_NUMBER, out1 => "DB440_MACHINE_ALARM_DECODING".GLOBAL_ALARMS_MACHINE.ALARM_DECODING)
      wire#w1
      { S7_Templates := "SrcType := UInt" } EQ_Contact(in1 := #UNIT_ALARM, in2 := 1)
      wire#w2
      { S7_Templates := "SrcType := UInt" } EQ_Contact(in1 := #STATION_ALARM, in2 := 0)
      S_Coil( "DB440_MACHINE_ALARM_DECODING".ALARMS_UNIT_01.ST0_TRANSFER.IS_SEOC_ALARMS )
   END_RUNG
   RUNG wire#w2
      { S7_Templates := "SrcType := UInt" } EQ_Contact(in1 := #STATION_ALARM, in2 := 1)
      S_Coil( "DB440_MACHINE_ALARM_DECODING".ALARMS_UNIT_01.ST1_LOAD_UNLOAD.IS_SEOC_ALARMS )
   END_RUNG
   RUNG wire#w2
      { S7_Templates := "SrcType := UInt" } EQ_Contact(in1 := #STATION_ALARM, in2 := 2)
      S_Coil( "DB440_MACHINE_ALARM_DECODING".ALARMS_UNIT_01.ST2_SPARE.IS_SEOC_ALARMS )
   END_RUNG
   RUNG wire#w2
      { S7_Templates := "SrcType := UInt" } EQ_Contact(in1 := #STATION_ALARM, in2 := 3)
      S_Coil( "DB440_MACHINE_ALARM_DECODING".ALARMS_UNIT_01.ST3_CLADDING.IS_SEOC_ALARMS )
   END_RUNG
   RUNG wire#w2
      { S7_Templates := "SrcType := UInt" } EQ_Contact(in1 := #STATION_ALARM, in2 := 4)
      S_Coil( "DB440_MACHINE_ALARM_DECODING".ALARMS_UNIT_01.ST4_CLEANING.IS_SEOC_ALARMS )
   END_RUNG
   RUNG wire#w1
      { S7_Templates := "SrcType := UInt" } EQ_Contact(in1 := #UNIT_ALARM, in2 := 2)
      wire#w3
      { S7_Templates := "SrcType := UInt" } EQ_Contact(in1 := #STATION_ALARM, in2 := 0)
      S_Coil( "DB440_MACHINE_ALARM_DECODING".ALARMS_UNIT_02.ST0_TRANSFER.IS_SEOC_ALARMS )
   END_RUNG
   RUNG wire#w3
      { S7_Templates := "SrcType := UInt" } EQ_Contact(in1 := #STATION_ALARM, in2 := 1)
      S_Coil( "DB440_MACHINE_ALARM_DECODING".ALARMS_UNIT_02.ST1_LOAD_UNLOAD.IS_SEOC_ALARMS )
   END_RUNG
   RUNG wire#w3
      { S7_Templates := "SrcType := UInt" } EQ_Contact(in1 := #STATION_ALARM, in2 := 2)
      S_Coil( "DB440_MACHINE_ALARM_DECODING".ALARMS_UNIT_02.ST2_MEASURING.IS_SEOC_ALARMS )
   END_RUNG
   RUNG wire#w3
      { S7_Templates := "SrcType := UInt" } EQ_Contact(in1 := #STATION_ALARM, in2 := 3)
      S_Coil( "DB440_MACHINE_ALARM_DECODING".ALARMS_UNIT_02.ST3_CLADDING.IS_SEOC_ALARMS )
   END_RUNG
   RUNG wire#w3
      { S7_Templates := "SrcType := UInt" } EQ_Contact(in1 := #STATION_ALARM, in2 := 4)
      S_Coil( "DB440_MACHINE_ALARM_DECODING".ALARMS_UNIT_02.ST4_CLEANING.IS_SEOC_ALARMS )
   END_RUNG
   RUNG wire#w1
      { S7_Templates := "SrcType := UInt" } EQ_Contact(in1 := #UNIT_ALARM, in2 := 3)
      S_Coil( "DB440_MACHINE_ALARM_DECODING".ALARMS_UNIT_03.IS_SEOC_ALARMS )
   END_RUNG
   RUNG wire#w1
      { S7_Templates := "SrcType := UInt" } EQ_Contact(in1 := #UNIT_ALARM, in2 := 4)
      S_Coil( "DB440_MACHINE_ALARM_DECODING".ALARMS_UNIT_04.IS_SEOC_ALARMS )
   END_RUNG
   // the same network as SCL:
   // ENO of a box is taken as its EN; it also drops when the box reports an error
   #BRAKE.IS_SEOC_ALARMS := NOT (NOT #BLOCKED_ALARM AND NOT #UNBLOCKED_ALARM AND NOT #MAINTENANCE_UNBLOCKED_ALARM);
   IF #BRAKE.IS_SEOC_ALARMS THEN
       "DB440_MACHINE_ALARM_DECODING".GLOBAL_ALARMS_MACHINE.ALARM_DECODING := #DB_NUMBER;
   END_IF;
   #_w1 := #BRAKE.IS_SEOC_ALARMS AND (#UNIT_ALARM = 1);
   IF #_w1 AND (#STATION_ALARM = 0) THEN
       "DB440_MACHINE_ALARM_DECODING".ALARMS_UNIT_01.ST0_TRANSFER.IS_SEOC_ALARMS := TRUE;
   END_IF;
   IF #_w1 AND (#STATION_ALARM = 1) THEN
       "DB440_MACHINE_ALARM_DECODING".ALARMS_UNIT_01.ST1_LOAD_UNLOAD.IS_SEOC_ALARMS := TRUE;
   END_IF;
   IF #_w1 AND (#STATION_ALARM = 2) THEN
       "DB440_MACHINE_ALARM_DECODING".ALARMS_UNIT_01.ST2_SPARE.IS_SEOC_ALARMS := TRUE;
   END_IF;
   IF #_w1 AND (#STATION_ALARM = 3) THEN
       "DB440_MACHINE_ALARM_DECODING".ALARMS_UNIT_01.ST3_CLADDING.IS_SEOC_ALARMS := TRUE;
   END_IF;
   IF #_w1 AND (#STATION_ALARM = 4) THEN
       "DB440_MACHINE_ALARM_DECODING".ALARMS_UNIT_01.ST4_CLEANING.IS_SEOC_ALARMS := TRUE;
   END_IF;
   #_w2 := #BRAKE.IS_SEOC_ALARMS AND (#UNIT_ALARM = 2);
   IF #_w2 AND (#STATION_ALARM = 0) THEN
       "DB440_MACHINE_ALARM_DECODING".ALARMS_UNIT_02.ST0_TRANSFER.IS_SEOC_ALARMS := TRUE;
   END_IF;
   IF #_w2 AND (#STATION_ALARM = 1) THEN
       "DB440_MACHINE_ALARM_DECODING".ALARMS_UNIT_02.ST1_LOAD_UNLOAD.IS_SEOC_ALARMS := TRUE;
   END_IF;
   IF #_w2 AND (#STATION_ALARM = 2) THEN
       "DB440_MACHINE_ALARM_DECODING".ALARMS_UNIT_02.ST2_MEASURING.IS_SEOC_ALARMS := TRUE;
   END_IF;
   IF #_w2 AND (#STATION_ALARM = 3) THEN
       "DB440_MACHINE_ALARM_DECODING".ALARMS_UNIT_02.ST3_CLADDING.IS_SEOC_ALARMS := TRUE;
   END_IF;
   IF #_w2 AND (#STATION_ALARM = 4) THEN
       "DB440_MACHINE_ALARM_DECODING".ALARMS_UNIT_02.ST4_CLEANING.IS_SEOC_ALARMS := TRUE;
   END_IF;
   IF #BRAKE.IS_SEOC_ALARMS AND (#UNIT_ALARM = 3) THEN
       "DB440_MACHINE_ALARM_DECODING".ALARMS_UNIT_03.IS_SEOC_ALARMS := TRUE;
   END_IF;
   IF #BRAKE.IS_SEOC_ALARMS AND (#UNIT_ALARM = 4) THEN
       "DB440_MACHINE_ALARM_DECODING".ALARMS_UNIT_04.IS_SEOC_ALARMS := TRUE;
   END_IF;
END_REGION

REGION Network 30: ANY ACTIVE ALARM
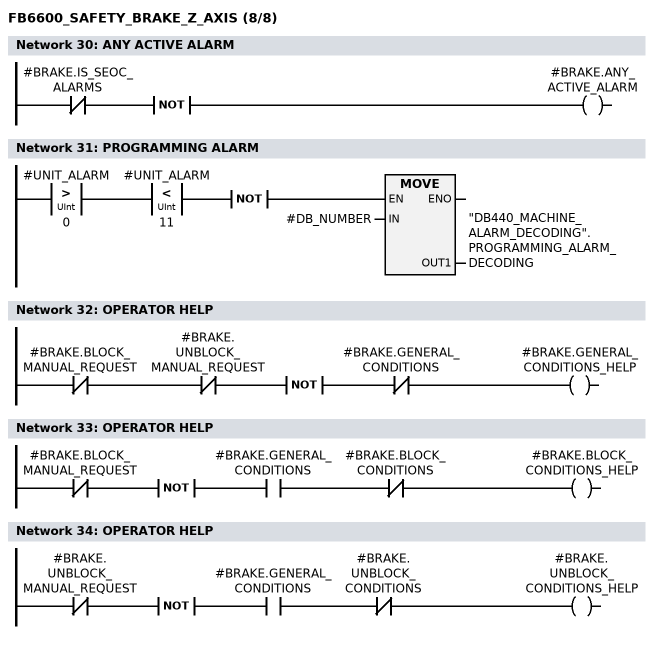
   RUNG wire#powerrail
      I_Contact( #BRAKE.IS_SEOC_ALARMS )
      Not()
      Coil( #BRAKE.ANY_ACTIVE_ALARM )
   END_RUNG
   // the same network as SCL:
   #BRAKE.ANY_ACTIVE_ALARM := NOT (NOT #BRAKE.IS_SEOC_ALARMS);
END_REGION

REGION Network 31: PROGRAMMING ALARM
   RUNG wire#powerrail
      { S7_Templates := "SrcType := UInt" } GT_Contact(in1 := #UNIT_ALARM, in2 := 0)
      { S7_Templates := "SrcType := UInt" } LT_Contact(in1 := #UNIT_ALARM, in2 := 11)
      Not()
      Move(in := #DB_NUMBER, out1 => "DB440_MACHINE_ALARM_DECODING".PROGRAMMING_ALARM_DECODING)
   END_RUNG
   // the same network as SCL:
   IF NOT ((#UNIT_ALARM > 0) AND (#UNIT_ALARM < 11)) THEN
       "DB440_MACHINE_ALARM_DECODING".PROGRAMMING_ALARM_DECODING := #DB_NUMBER;
   END_IF;
END_REGION

REGION Network 32: OPERATOR HELP
   RUNG wire#powerrail
      I_Contact( #BRAKE.BLOCK_MANUAL_REQUEST )
      I_Contact( #BRAKE.UNBLOCK_MANUAL_REQUEST )
      Not()
      I_Contact( #BRAKE.GENERAL_CONDITIONS )
      Coil( #BRAKE.GENERAL_CONDITIONS_HELP )
   END_RUNG
   // the same network as SCL:
   #BRAKE.GENERAL_CONDITIONS_HELP := NOT (NOT #BRAKE.BLOCK_MANUAL_REQUEST AND NOT #BRAKE.UNBLOCK_MANUAL_REQUEST) AND NOT #BRAKE.GENERAL_CONDITIONS;
END_REGION

REGION Network 33: OPERATOR HELP
   RUNG wire#powerrail
      I_Contact( #BRAKE.BLOCK_MANUAL_REQUEST )
      Not()
      Contact( #BRAKE.GENERAL_CONDITIONS )
      I_Contact( #BRAKE.BLOCK_CONDITIONS )
      Coil( #BRAKE.BLOCK_CONDITIONS_HELP )
   END_RUNG
   // the same network as SCL:
   #BRAKE.BLOCK_CONDITIONS_HELP := NOT (NOT #BRAKE.BLOCK_MANUAL_REQUEST) AND #BRAKE.GENERAL_CONDITIONS AND NOT #BRAKE.BLOCK_CONDITIONS;
END_REGION

REGION Network 34: OPERATOR HELP
   RUNG wire#powerrail
      I_Contact( #BRAKE.UNBLOCK_MANUAL_REQUEST )
      Not()
      Contact( #BRAKE.GENERAL_CONDITIONS )
      I_Contact( #BRAKE.UNBLOCK_CONDITIONS )
      Coil( #BRAKE.UNBLOCK_CONDITIONS_HELP )
   END_RUNG
   // the same network as SCL:
   #BRAKE.UNBLOCK_CONDITIONS_HELP := NOT (NOT #BRAKE.UNBLOCK_MANUAL_REQUEST) AND #BRAKE.GENERAL_CONDITIONS AND NOT #BRAKE.UNBLOCK_CONDITIONS;
END_REGION
END_FUNCTION_BLOCK

FUNCTION "FC7001_UNIT_01_MAIN_SAFETY_DOOR" : Void   // FC7001, LAD
{ S7_Optimized_Access := 'FALSE' }
AUTHOR : ETXETAR
VERSION : 1.0
// stored: AutoNumber false, IsIECCheckEnabled false, SetENOAutomatically false, UDAEnableTagReadback false
   VAR_INPUT
      OPTIONS_0 : Byte;   // OPTIONS 0
      CLOSED : Bool;   // CLOSED INPUT
      LOCKED : Bool;   // LOCKED INPUT
   END_VAR
   VAR_OUTPUT
      UNLOCK : Bool;   // UNLOCK OUTPUT
      RED_LIGTH : Bool;   // RED LIGTH OUTPUT
      GREEN_LIGTH : Bool;   // GREEN LIGTH OUTPUT
   END_VAR
   VAR_TEMP
      INPUTS_MASK : Byte;   // INPUTS MASK
      O_BYTE_0 : Struct   // OPTIONS BYTE 0
         IMMEDIATE_STOP : Bool;   // IMMEDIATE STOP REACTION OPTION
         SEOC_WARNING : Bool;   // SEOC WARNING REACTION OPTION
         CLOSED_SENSOR_I : Bool;   // CLOSED SENSOR INPUT OPTION
         CIRCUIT_E2 : Bool;   // CIRCUIT E2 OPTION
         PNEUMATIC_DRIVE : Bool;   // PNEUMATIC DRIVE OPTION
         CHIP_CONVEYOR : Bool;   // CHIP CONVEYOR OPTION
         SPARE_6 : Bool;   // SPARE OPTION
         SPARE_7 : Bool;   // SPARE OPTION
      END_STRUCT;
   END_VAR
   VAR CONSTANT
      FC_NUMBER : DInt := 7001;
   END_VAR
   VAR_TEMP   // added for the SCL form of the ladder/FBD networks
      _w1 : Bool;
      _w2 : Bool;
   END_VAR
BEGIN

REGION Network 1: OPTIONS
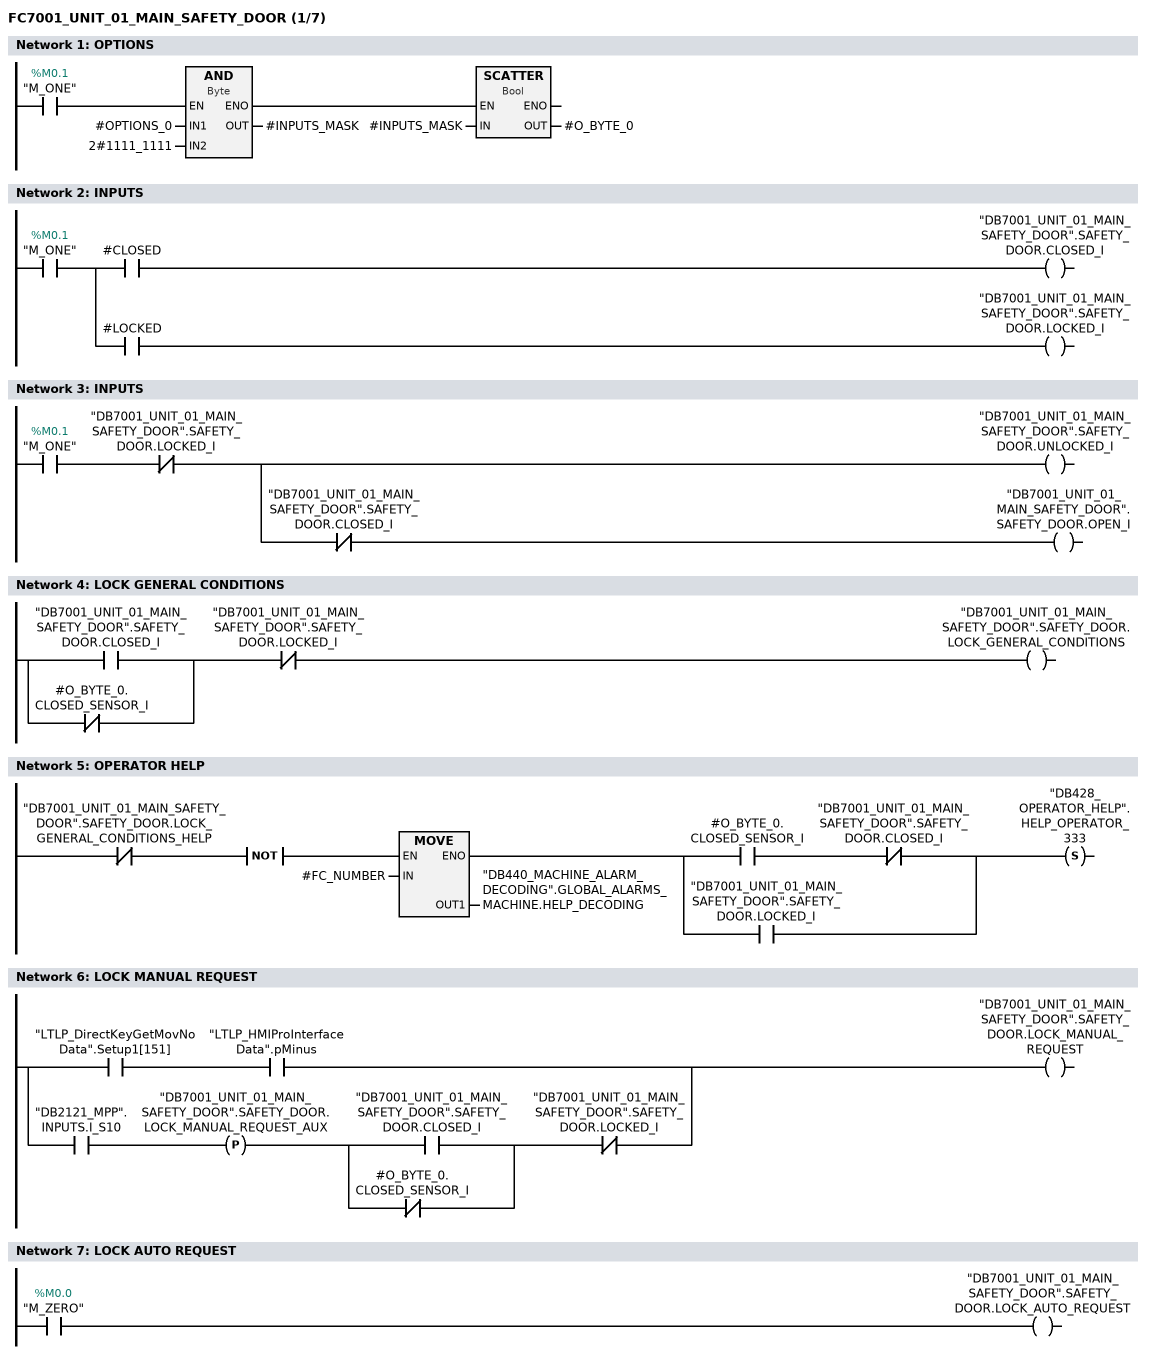
   RUNG wire#powerrail
      Contact( "M_ONE" )
      { S7_Templates := "SrcType := Byte"; S7_GenerateENO := "TRUE" } And(in1 := #OPTIONS_0, in2 := 2#1111_1111, out => #INPUTS_MASK)
      { S7_Templates := "[dest_type := Bool, src_type := Byte]" } SCATTER(IN := #INPUTS_MASK, OUT => #O_BYTE_0)
   END_RUNG
   // the same network as SCL:
   IF "M_ONE" THEN
       #INPUTS_MASK := #OPTIONS_0 AND 2#1111_1111;
       SCATTER(IN := #INPUTS_MASK, OUT => #O_BYTE_0);
   END_IF;
END_REGION

REGION Network 2: INPUTS
   RUNG wire#powerrail
      Contact( "M_ONE" )
      wire#w1
      Contact( #CLOSED )
      Coil( "DB7001_UNIT_01_MAIN_SAFETY_DOOR".SAFETY_DOOR.CLOSED_I )
   END_RUNG
   RUNG wire#w1
      Contact( #LOCKED )
      Coil( "DB7001_UNIT_01_MAIN_SAFETY_DOOR".SAFETY_DOOR.LOCKED_I )
   END_RUNG
   // the same network as SCL:
   "DB7001_UNIT_01_MAIN_SAFETY_DOOR".SAFETY_DOOR.CLOSED_I := "M_ONE" AND #CLOSED;
   "DB7001_UNIT_01_MAIN_SAFETY_DOOR".SAFETY_DOOR.LOCKED_I := "M_ONE" AND #LOCKED;
END_REGION

REGION Network 3: INPUTS
   RUNG wire#powerrail
      Contact( "M_ONE" )
      I_Contact( "DB7001_UNIT_01_MAIN_SAFETY_DOOR".SAFETY_DOOR.LOCKED_I )
      wire#w1
      Coil( "DB7001_UNIT_01_MAIN_SAFETY_DOOR".SAFETY_DOOR.UNLOCKED_I )
   END_RUNG
   RUNG wire#w1
      I_Contact( "DB7001_UNIT_01_MAIN_SAFETY_DOOR".SAFETY_DOOR.CLOSED_I )
      Coil( "DB7001_UNIT_01_MAIN_SAFETY_DOOR".SAFETY_DOOR.OPEN_I )
   END_RUNG
   // the same network as SCL:
   "DB7001_UNIT_01_MAIN_SAFETY_DOOR".SAFETY_DOOR.UNLOCKED_I := "M_ONE" AND NOT "DB7001_UNIT_01_MAIN_SAFETY_DOOR".SAFETY_DOOR.LOCKED_I;
   "DB7001_UNIT_01_MAIN_SAFETY_DOOR".SAFETY_DOOR.OPEN_I := "DB7001_UNIT_01_MAIN_SAFETY_DOOR".SAFETY_DOOR.UNLOCKED_I AND NOT "DB7001_UNIT_01_MAIN_SAFETY_DOOR".SAFETY_DOOR.CLOSED_I;
END_REGION

REGION Network 4: LOCK GENERAL CONDITIONS
   RUNG wire#powerrail
      Contact( "DB7001_UNIT_01_MAIN_SAFETY_DOOR".SAFETY_DOOR.CLOSED_I )
      wire#w1
      I_Contact( "DB7001_UNIT_01_MAIN_SAFETY_DOOR".SAFETY_DOOR.LOCKED_I )
      Coil( "DB7001_UNIT_01_MAIN_SAFETY_DOOR".SAFETY_DOOR.LOCK_GENERAL_CONDITIONS )
   END_RUNG
   RUNG wire#powerrail
      I_Contact( #O_BYTE_0.CLOSED_SENSOR_I )
   END_RUNG wire#w1
   // the same network as SCL:
   "DB7001_UNIT_01_MAIN_SAFETY_DOOR".SAFETY_DOOR.LOCK_GENERAL_CONDITIONS := ("DB7001_UNIT_01_MAIN_SAFETY_DOOR".SAFETY_DOOR.CLOSED_I OR NOT #O_BYTE_0.CLOSED_SENSOR_I) AND NOT "DB7001_UNIT_01_MAIN_SAFETY_DOOR".SAFETY_DOOR.LOCKED_I;
END_REGION

REGION Network 5: OPERATOR HELP
   RUNG wire#powerrail
      I_Contact( "DB7001_UNIT_01_MAIN_SAFETY_DOOR".SAFETY_DOOR.LOCK_GENERAL_CONDITIONS_HELP )
      Not()
      { S7_GenerateENO := "TRUE" } Move(in := #FC_NUMBER, out1 => "DB440_MACHINE_ALARM_DECODING".GLOBAL_ALARMS_MACHINE.HELP_DECODING)
      wire#w1
      Contact( #O_BYTE_0.CLOSED_SENSOR_I )
      I_Contact( "DB7001_UNIT_01_MAIN_SAFETY_DOOR".SAFETY_DOOR.CLOSED_I )
      wire#w2
      S_Coil( "DB428_OPERATOR_HELP".HELP_OPERATOR_333 )
   END_RUNG
   RUNG wire#w1
      Contact( "DB7001_UNIT_01_MAIN_SAFETY_DOOR".SAFETY_DOOR.LOCKED_I )
   END_RUNG wire#w2
   // the same network as SCL:
   // ENO of a box is taken as its EN; it also drops when the box reports an error
   #_w1 := NOT (NOT "DB7001_UNIT_01_MAIN_SAFETY_DOOR".SAFETY_DOOR.LOCK_GENERAL_CONDITIONS_HELP);
   IF #_w1 THEN "DB440_MACHINE_ALARM_DECODING".GLOBAL_ALARMS_MACHINE.HELP_DECODING := #FC_NUMBER; END_IF;
   IF #_w1 AND ((#O_BYTE_0.CLOSED_SENSOR_I AND NOT "DB7001_UNIT_01_MAIN_SAFETY_DOOR".SAFETY_DOOR.CLOSED_I) OR "DB7001_UNIT_01_MAIN_SAFETY_DOOR".SAFETY_DOOR.LOCKED_I) THEN
       "DB428_OPERATOR_HELP".HELP_OPERATOR_333 := TRUE;
   END_IF;
END_REGION

REGION Network 6: LOCK MANUAL REQUEST
   RUNG wire#powerrail
      Contact( "LTLP_DirectKeyGetMovNoData".Setup1[151] )
      Contact( "LTLP_HMIProInterfaceData".pMinus )
      wire#w1
      Coil( "DB7001_UNIT_01_MAIN_SAFETY_DOOR".SAFETY_DOOR.LOCK_MANUAL_REQUEST )
   END_RUNG
   RUNG wire#powerrail
      Contact( "DB2121_MPP".INPUTS.I_S10 )
      P_Trig( "DB7001_UNIT_01_MAIN_SAFETY_DOOR".SAFETY_DOOR.LOCK_MANUAL_REQUEST_AUX )
      wire#w2
      Contact( "DB7001_UNIT_01_MAIN_SAFETY_DOOR".SAFETY_DOOR.CLOSED_I )
      wire#w3
      I_Contact( "DB7001_UNIT_01_MAIN_SAFETY_DOOR".SAFETY_DOOR.LOCKED_I )
   END_RUNG wire#w1
   RUNG wire#w2
      I_Contact( #O_BYTE_0.CLOSED_SENSOR_I )
   END_RUNG wire#w3
   // the same network as SCL:
   #_w1 := "DB2121_MPP".INPUTS.I_S10 AND NOT "DB7001_UNIT_01_MAIN_SAFETY_DOOR".SAFETY_DOOR.LOCK_MANUAL_REQUEST_AUX;   // rising edge
   "DB7001_UNIT_01_MAIN_SAFETY_DOOR".SAFETY_DOOR.LOCK_MANUAL_REQUEST_AUX := "DB2121_MPP".INPUTS.I_S10;
   "DB7001_UNIT_01_MAIN_SAFETY_DOOR".SAFETY_DOOR.LOCK_MANUAL_REQUEST := ("LTLP_DirectKeyGetMovNoData".Setup1[151] AND "LTLP_HMIProInterfaceData".pMinus) OR (#_w1 AND ("DB7001_UNIT_01_MAIN_SAFETY_DOOR".SAFETY_DOOR.CLOSED_I OR NOT #O_BYTE_0.CLOSED_SENSOR_I) AND NOT "DB7001_UNIT_01_MAIN_SAFETY_DOOR".SAFETY_DOOR.LOCKED_I);
END_REGION

REGION Network 7: LOCK AUTO REQUEST
   RUNG wire#powerrail
      Contact( "M_ZERO" )
      Coil( "DB7001_UNIT_01_MAIN_SAFETY_DOOR".SAFETY_DOOR.LOCK_AUTO_REQUEST )
   END_RUNG
   // the same network as SCL:
   "DB7001_UNIT_01_MAIN_SAFETY_DOOR".SAFETY_DOOR.LOCK_AUTO_REQUEST := "M_ZERO";
END_REGION

REGION Network 8: LOCK GLOBAL REQUEST
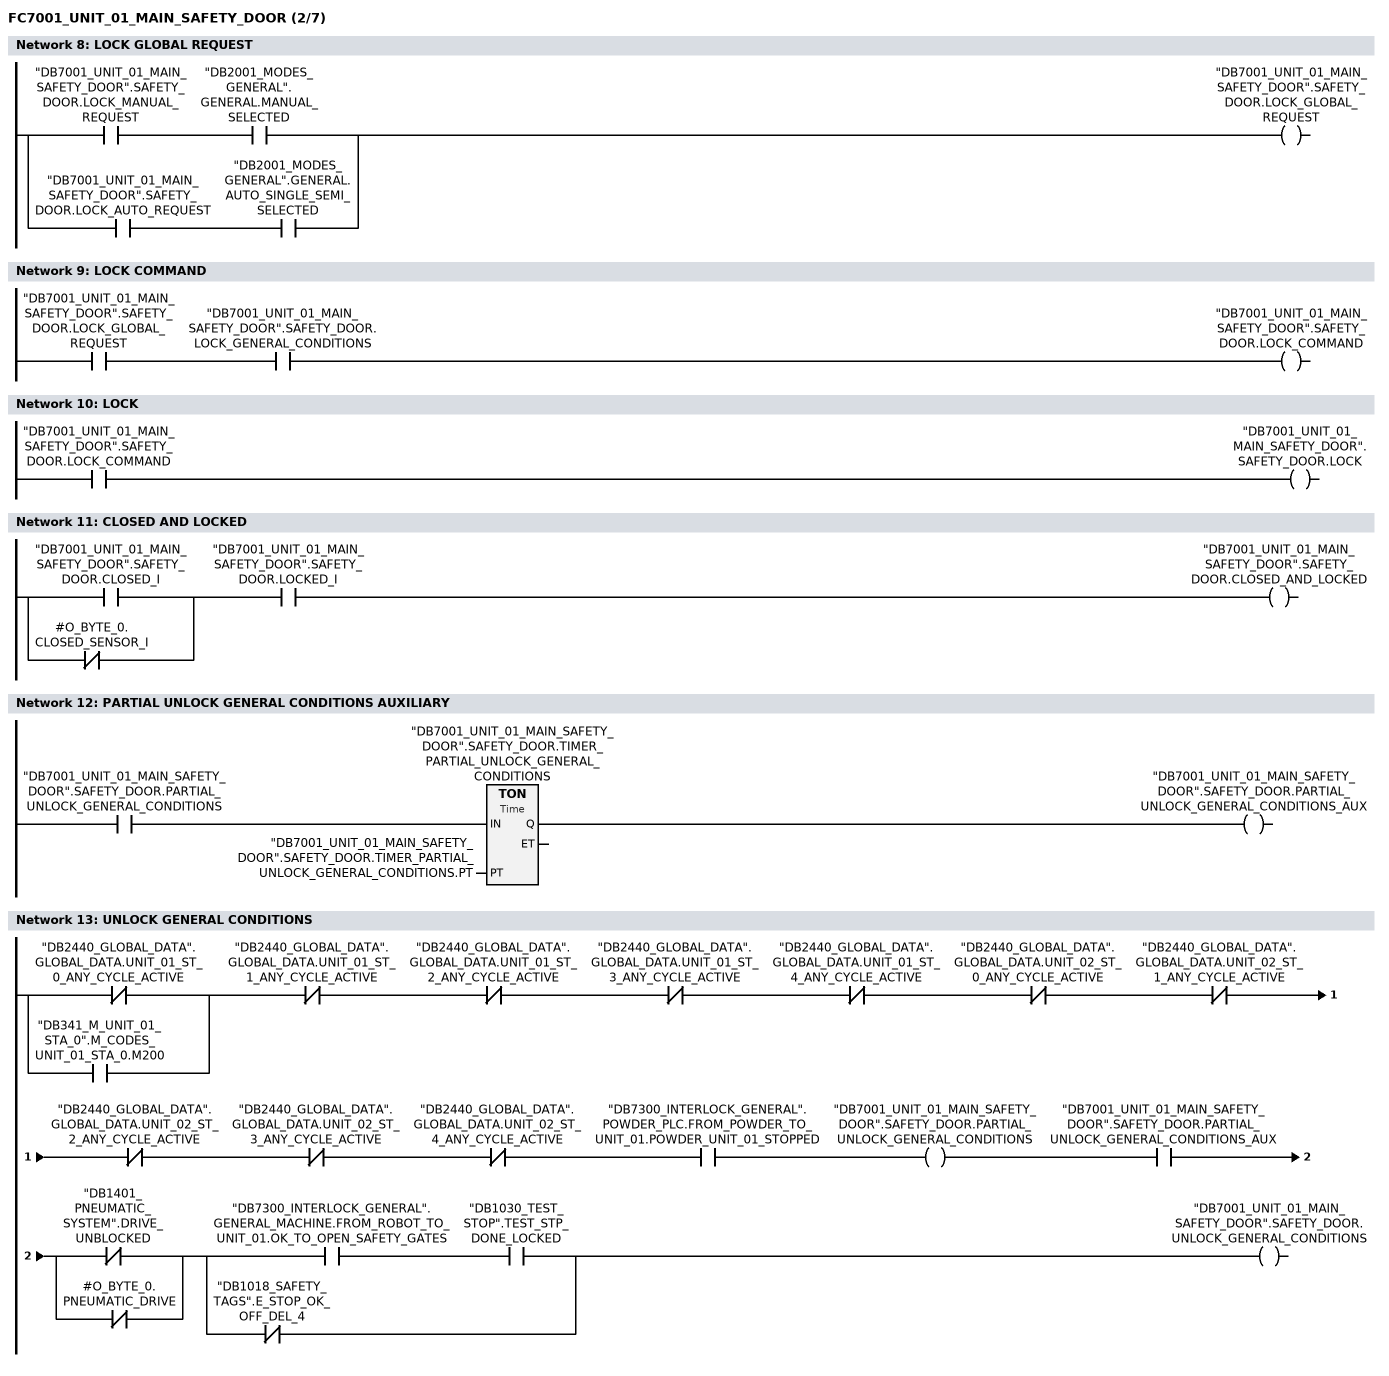
   RUNG wire#powerrail
      Contact( "DB7001_UNIT_01_MAIN_SAFETY_DOOR".SAFETY_DOOR.LOCK_MANUAL_REQUEST )
      Contact( "DB2001_MODES_GENERAL".GENERAL.MANUAL_SELECTED )
      wire#w1
      Coil( "DB7001_UNIT_01_MAIN_SAFETY_DOOR".SAFETY_DOOR.LOCK_GLOBAL_REQUEST )
   END_RUNG
   RUNG wire#powerrail
      Contact( "DB7001_UNIT_01_MAIN_SAFETY_DOOR".SAFETY_DOOR.LOCK_AUTO_REQUEST )
      Contact( "DB2001_MODES_GENERAL".GENERAL.AUTO_SINGLE_SEMI_SELECTED )
   END_RUNG wire#w1
   // the same network as SCL:
   "DB7001_UNIT_01_MAIN_SAFETY_DOOR".SAFETY_DOOR.LOCK_GLOBAL_REQUEST := ("DB7001_UNIT_01_MAIN_SAFETY_DOOR".SAFETY_DOOR.LOCK_MANUAL_REQUEST AND "DB2001_MODES_GENERAL".GENERAL.MANUAL_SELECTED) OR ("DB7001_UNIT_01_MAIN_SAFETY_DOOR".SAFETY_DOOR.LOCK_AUTO_REQUEST AND "DB2001_MODES_GENERAL".GENERAL.AUTO_SINGLE_SEMI_SELECTED);
END_REGION

REGION Network 9: LOCK COMMAND
   RUNG wire#powerrail
      Contact( "DB7001_UNIT_01_MAIN_SAFETY_DOOR".SAFETY_DOOR.LOCK_GLOBAL_REQUEST )
      Contact( "DB7001_UNIT_01_MAIN_SAFETY_DOOR".SAFETY_DOOR.LOCK_GENERAL_CONDITIONS )
      Coil( "DB7001_UNIT_01_MAIN_SAFETY_DOOR".SAFETY_DOOR.LOCK_COMMAND )
   END_RUNG
   // the same network as SCL:
   "DB7001_UNIT_01_MAIN_SAFETY_DOOR".SAFETY_DOOR.LOCK_COMMAND := "DB7001_UNIT_01_MAIN_SAFETY_DOOR".SAFETY_DOOR.LOCK_GLOBAL_REQUEST AND "DB7001_UNIT_01_MAIN_SAFETY_DOOR".SAFETY_DOOR.LOCK_GENERAL_CONDITIONS;
END_REGION

REGION Network 10: LOCK
   RUNG wire#powerrail
      Contact( "DB7001_UNIT_01_MAIN_SAFETY_DOOR".SAFETY_DOOR.LOCK_COMMAND )
      Coil( "DB7001_UNIT_01_MAIN_SAFETY_DOOR".SAFETY_DOOR.LOCK )
   END_RUNG
   // the same network as SCL:
   "DB7001_UNIT_01_MAIN_SAFETY_DOOR".SAFETY_DOOR.LOCK := "DB7001_UNIT_01_MAIN_SAFETY_DOOR".SAFETY_DOOR.LOCK_COMMAND;
END_REGION

REGION Network 11: CLOSED AND LOCKED
   RUNG wire#powerrail
      Contact( "DB7001_UNIT_01_MAIN_SAFETY_DOOR".SAFETY_DOOR.CLOSED_I )
      wire#w1
      Contact( "DB7001_UNIT_01_MAIN_SAFETY_DOOR".SAFETY_DOOR.LOCKED_I )
      Coil( "DB7001_UNIT_01_MAIN_SAFETY_DOOR".SAFETY_DOOR.CLOSED_AND_LOCKED )
   END_RUNG
   RUNG wire#powerrail
      I_Contact( #O_BYTE_0.CLOSED_SENSOR_I )
   END_RUNG wire#w1
   // the same network as SCL:
   "DB7001_UNIT_01_MAIN_SAFETY_DOOR".SAFETY_DOOR.CLOSED_AND_LOCKED := ("DB7001_UNIT_01_MAIN_SAFETY_DOOR".SAFETY_DOOR.CLOSED_I OR NOT #O_BYTE_0.CLOSED_SENSOR_I) AND "DB7001_UNIT_01_MAIN_SAFETY_DOOR".SAFETY_DOOR.LOCKED_I;
END_REGION

REGION Network 12: PARTIAL UNLOCK GENERAL CONDITIONS AUXILIARY
   RUNG wire#powerrail
      Contact( "DB7001_UNIT_01_MAIN_SAFETY_DOOR".SAFETY_DOOR.PARTIAL_UNLOCK_GENERAL_CONDITIONS )
      { S7_Templates := "time_type := Time" } "DB7001_UNIT_01_MAIN_SAFETY_DOOR".SAFETY_DOOR.TIMER_PARTIAL_UNLOCK_GENERAL_CONDITIONS.TON(pt := "DB7001_UNIT_01_MAIN_SAFETY_DOOR".SAFETY_DOOR.TIMER_PARTIAL_UNLOCK_GENERAL_CONDITIONS.PT, et =>)
      Coil( "DB7001_UNIT_01_MAIN_SAFETY_DOOR".SAFETY_DOOR.PARTIAL_UNLOCK_GENERAL_CONDITIONS_AUX )
   END_RUNG
   // the same network as SCL:
   "DB7001_UNIT_01_MAIN_SAFETY_DOOR".SAFETY_DOOR.TIMER_PARTIAL_UNLOCK_GENERAL_CONDITIONS.TON(IN := "DB7001_UNIT_01_MAIN_SAFETY_DOOR".SAFETY_DOOR.PARTIAL_UNLOCK_GENERAL_CONDITIONS,
                           PT := "DB7001_UNIT_01_MAIN_SAFETY_DOOR".SAFETY_DOOR.TIMER_PARTIAL_UNLOCK_GENERAL_CONDITIONS.PT);
   "DB7001_UNIT_01_MAIN_SAFETY_DOOR".SAFETY_DOOR.PARTIAL_UNLOCK_GENERAL_CONDITIONS_AUX := "DB7001_UNIT_01_MAIN_SAFETY_DOOR".SAFETY_DOOR.TIMER_PARTIAL_UNLOCK_GENERAL_CONDITIONS.Q;
END_REGION

REGION Network 13: UNLOCK GENERAL CONDITIONS
   RUNG wire#powerrail
      I_Contact( "DB2440_GLOBAL_DATA".GLOBAL_DATA.UNIT_01_ST_0_ANY_CYCLE_ACTIVE )
      wire#w1
      I_Contact( "DB2440_GLOBAL_DATA".GLOBAL_DATA.UNIT_01_ST_1_ANY_CYCLE_ACTIVE )
      I_Contact( "DB2440_GLOBAL_DATA".GLOBAL_DATA.UNIT_01_ST_2_ANY_CYCLE_ACTIVE )
      I_Contact( "DB2440_GLOBAL_DATA".GLOBAL_DATA.UNIT_01_ST_3_ANY_CYCLE_ACTIVE )
      I_Contact( "DB2440_GLOBAL_DATA".GLOBAL_DATA.UNIT_01_ST_4_ANY_CYCLE_ACTIVE )
      I_Contact( "DB2440_GLOBAL_DATA".GLOBAL_DATA.UNIT_02_ST_0_ANY_CYCLE_ACTIVE )
      I_Contact( "DB2440_GLOBAL_DATA".GLOBAL_DATA.UNIT_02_ST_1_ANY_CYCLE_ACTIVE )
      I_Contact( "DB2440_GLOBAL_DATA".GLOBAL_DATA.UNIT_02_ST_2_ANY_CYCLE_ACTIVE )
      I_Contact( "DB2440_GLOBAL_DATA".GLOBAL_DATA.UNIT_02_ST_3_ANY_CYCLE_ACTIVE )
      I_Contact( "DB2440_GLOBAL_DATA".GLOBAL_DATA.UNIT_02_ST_4_ANY_CYCLE_ACTIVE )
      Contact( "DB7300_INTERLOCK_GENERAL".POWDER_PLC.FROM_POWDER_TO_UNIT_01.POWDER_UNIT_01_STOPPED )
      Coil( "DB7001_UNIT_01_MAIN_SAFETY_DOOR".SAFETY_DOOR.PARTIAL_UNLOCK_GENERAL_CONDITIONS )
      Contact( "DB7001_UNIT_01_MAIN_SAFETY_DOOR".SAFETY_DOOR.PARTIAL_UNLOCK_GENERAL_CONDITIONS_AUX )
      wire#w2
      I_Contact( "DB1401_PNEUMATIC_SYSTEM".DRIVE_UNBLOCKED )
      wire#w3
      Contact( "DB7300_INTERLOCK_GENERAL".GENERAL_MACHINE.FROM_ROBOT_TO_UNIT_01.OK_TO_OPEN_SAFETY_GATES )
      Contact( "DB1030_TEST_STOP".TEST_STP_DONE_LOCKED )
      wire#w4
      Coil( "DB7001_UNIT_01_MAIN_SAFETY_DOOR".SAFETY_DOOR.UNLOCK_GENERAL_CONDITIONS )
   END_RUNG
   RUNG wire#powerrail
      Contact( "DB341_M_UNIT_01_STA_0".M_CODES_UNIT_01_STA_0.M200 )
   END_RUNG wire#w1
   RUNG wire#w2
      I_Contact( #O_BYTE_0.PNEUMATIC_DRIVE )
   END_RUNG wire#w3
   RUNG wire#w3
      I_Contact( "DB1018_SAFETY_TAGS".E_STOP_OK_OFF_DEL_4 )
   END_RUNG wire#w4
   // the same network as SCL:
   "DB7001_UNIT_01_MAIN_SAFETY_DOOR".SAFETY_DOOR.PARTIAL_UNLOCK_GENERAL_CONDITIONS := (NOT "DB2440_GLOBAL_DATA".GLOBAL_DATA.UNIT_01_ST_0_ANY_CYCLE_ACTIVE OR "DB341_M_UNIT_01_STA_0".M_CODES_UNIT_01_STA_0.M200) AND NOT "DB2440_GLOBAL_DATA".GLOBAL_DATA.UNIT_01_ST_1_ANY_CYCLE_ACTIVE AND NOT "DB2440_GLOBAL_DATA".GLOBAL_DATA.UNIT_01_ST_2_ANY_CYCLE_ACTIVE AND NOT "DB2440_GLOBAL_DATA".GLOBAL_DATA.UNIT_01_ST_3_ANY_CYCLE_ACTIVE AND NOT "DB2440_GLOBAL_DATA".GLOBAL_DATA.UNIT_01_ST_4_ANY_CYCLE_ACTIVE AND NOT "DB2440_GLOBAL_DATA".GLOBAL_DATA.UNIT_02_ST_0_ANY_CYCLE_ACTIVE AND NOT "DB2440_GLOBAL_DATA".GLOBAL_DATA.UNIT_02_ST_1_ANY_CYCLE_ACTIVE AND NOT "DB2440_GLOBAL_DATA".GLOBAL_DATA.UNIT_02_ST_2_ANY_CYCLE_ACTIVE AND NOT "DB2440_GLOBAL_DATA".GLOBAL_DATA.UNIT_02_ST_3_ANY_CYCLE_ACTIVE AND NOT "DB2440_GLOBAL_DATA".GLOBAL_DATA.UNIT_02_ST_4_ANY_CYCLE_ACTIVE AND "DB7300_INTERLOCK_GENERAL".POWDER_PLC.FROM_POWDER_TO_UNIT_01.POWDER_UNIT_01_STOPPED;
   "DB7001_UNIT_01_MAIN_SAFETY_DOOR".SAFETY_DOOR.UNLOCK_GENERAL_CONDITIONS := "DB7001_UNIT_01_MAIN_SAFETY_DOOR".SAFETY_DOOR.PARTIAL_UNLOCK_GENERAL_CONDITIONS AND "DB7001_UNIT_01_MAIN_SAFETY_DOOR".SAFETY_DOOR.PARTIAL_UNLOCK_GENERAL_CONDITIONS_AUX AND (NOT "DB1401_PNEUMATIC_SYSTEM".DRIVE_UNBLOCKED OR NOT #O_BYTE_0.PNEUMATIC_DRIVE) AND (("DB7300_INTERLOCK_GENERAL".GENERAL_MACHINE.FROM_ROBOT_TO_UNIT_01.OK_TO_OPEN_SAFETY_GATES AND "DB1030_TEST_STOP".TEST_STP_DONE_LOCKED) OR NOT "DB1018_SAFETY_TAGS".E_STOP_OK_OFF_DEL_4);
END_REGION

REGION Network 14: OPERATOR HELP
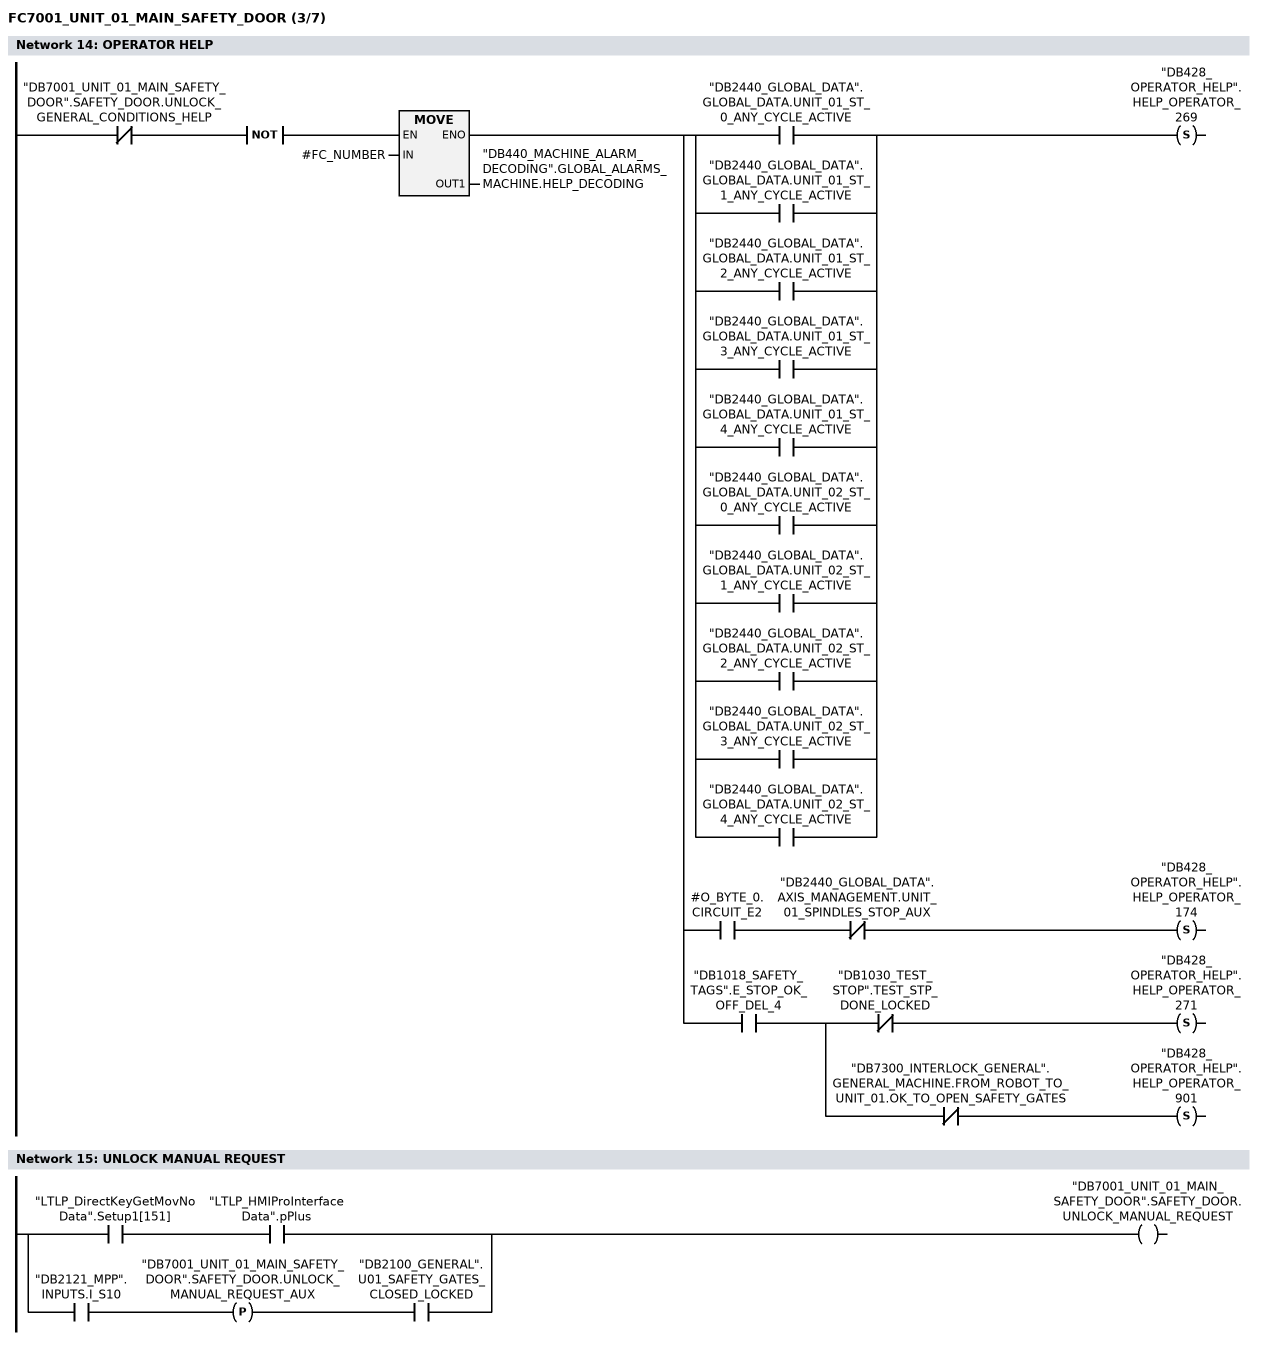
   RUNG wire#powerrail
      I_Contact( "DB7001_UNIT_01_MAIN_SAFETY_DOOR".SAFETY_DOOR.UNLOCK_GENERAL_CONDITIONS_HELP )
      Not()
      { S7_GenerateENO := "TRUE" } Move(in := #FC_NUMBER, out1 => "DB440_MACHINE_ALARM_DECODING".GLOBAL_ALARMS_MACHINE.HELP_DECODING)
      wire#w1
      Contact( "DB2440_GLOBAL_DATA".GLOBAL_DATA.UNIT_01_ST_0_ANY_CYCLE_ACTIVE )
      wire#w2
      S_Coil( "DB428_OPERATOR_HELP".HELP_OPERATOR_269 )
   END_RUNG
   RUNG wire#w1
      Contact( "DB2440_GLOBAL_DATA".GLOBAL_DATA.UNIT_01_ST_1_ANY_CYCLE_ACTIVE )
   END_RUNG wire#w2
   RUNG wire#w1
      Contact( "DB2440_GLOBAL_DATA".GLOBAL_DATA.UNIT_01_ST_2_ANY_CYCLE_ACTIVE )
   END_RUNG wire#w2
   RUNG wire#w1
      Contact( "DB2440_GLOBAL_DATA".GLOBAL_DATA.UNIT_01_ST_3_ANY_CYCLE_ACTIVE )
   END_RUNG wire#w2
   RUNG wire#w1
      Contact( "DB2440_GLOBAL_DATA".GLOBAL_DATA.UNIT_01_ST_4_ANY_CYCLE_ACTIVE )
   END_RUNG wire#w2
   RUNG wire#w1
      Contact( "DB2440_GLOBAL_DATA".GLOBAL_DATA.UNIT_02_ST_0_ANY_CYCLE_ACTIVE )
   END_RUNG wire#w2
   RUNG wire#w1
      Contact( "DB2440_GLOBAL_DATA".GLOBAL_DATA.UNIT_02_ST_1_ANY_CYCLE_ACTIVE )
   END_RUNG wire#w2
   RUNG wire#w1
      Contact( "DB2440_GLOBAL_DATA".GLOBAL_DATA.UNIT_02_ST_2_ANY_CYCLE_ACTIVE )
   END_RUNG wire#w2
   RUNG wire#w1
      Contact( "DB2440_GLOBAL_DATA".GLOBAL_DATA.UNIT_02_ST_3_ANY_CYCLE_ACTIVE )
   END_RUNG wire#w2
   RUNG wire#w1
      Contact( "DB2440_GLOBAL_DATA".GLOBAL_DATA.UNIT_02_ST_4_ANY_CYCLE_ACTIVE )
   END_RUNG wire#w2
   RUNG wire#w1
      Contact( #O_BYTE_0.CIRCUIT_E2 )
      I_Contact( "DB2440_GLOBAL_DATA".AXIS_MANAGEMENT.UNIT_01_SPINDLES_STOP_AUX )
      S_Coil( "DB428_OPERATOR_HELP".HELP_OPERATOR_174 )
   END_RUNG
   RUNG wire#w1
      Contact( "DB1018_SAFETY_TAGS".E_STOP_OK_OFF_DEL_4 )
      wire#w3
      I_Contact( "DB1030_TEST_STOP".TEST_STP_DONE_LOCKED )
      S_Coil( "DB428_OPERATOR_HELP".HELP_OPERATOR_271 )
   END_RUNG
   RUNG wire#w3
      I_Contact( "DB7300_INTERLOCK_GENERAL".GENERAL_MACHINE.FROM_ROBOT_TO_UNIT_01.OK_TO_OPEN_SAFETY_GATES )
      S_Coil( "DB428_OPERATOR_HELP".HELP_OPERATOR_901 )
   END_RUNG
   // the same network as SCL:
   // ENO of a box is taken as its EN; it also drops when the box reports an error
   #_w1 := NOT (NOT "DB7001_UNIT_01_MAIN_SAFETY_DOOR".SAFETY_DOOR.UNLOCK_GENERAL_CONDITIONS_HELP);
   IF #_w1 THEN "DB440_MACHINE_ALARM_DECODING".GLOBAL_ALARMS_MACHINE.HELP_DECODING := #FC_NUMBER; END_IF;
   IF #_w1 AND ("DB2440_GLOBAL_DATA".GLOBAL_DATA.UNIT_01_ST_0_ANY_CYCLE_ACTIVE OR "DB2440_GLOBAL_DATA".GLOBAL_DATA.UNIT_01_ST_1_ANY_CYCLE_ACTIVE OR "DB2440_GLOBAL_DATA".GLOBAL_DATA.UNIT_01_ST_2_ANY_CYCLE_ACTIVE OR "DB2440_GLOBAL_DATA".GLOBAL_DATA.UNIT_01_ST_3_ANY_CYCLE_ACTIVE OR "DB2440_GLOBAL_DATA".GLOBAL_DATA.UNIT_01_ST_4_ANY_CYCLE_ACTIVE OR "DB2440_GLOBAL_DATA".GLOBAL_DATA.UNIT_02_ST_0_ANY_CYCLE_ACTIVE OR "DB2440_GLOBAL_DATA".GLOBAL_DATA.UNIT_02_ST_1_ANY_CYCLE_ACTIVE OR "DB2440_GLOBAL_DATA".GLOBAL_DATA.UNIT_02_ST_2_ANY_CYCLE_ACTIVE OR "DB2440_GLOBAL_DATA".GLOBAL_DATA.UNIT_02_ST_3_ANY_CYCLE_ACTIVE OR "DB2440_GLOBAL_DATA".GLOBAL_DATA.UNIT_02_ST_4_ANY_CYCLE_ACTIVE) THEN
       "DB428_OPERATOR_HELP".HELP_OPERATOR_269 := TRUE;
   END_IF;
   IF #_w1 AND #O_BYTE_0.CIRCUIT_E2 AND NOT "DB2440_GLOBAL_DATA".AXIS_MANAGEMENT.UNIT_01_SPINDLES_STOP_AUX THEN
       "DB428_OPERATOR_HELP".HELP_OPERATOR_174 := TRUE;
   END_IF;
   #_w2 := #_w1 AND "DB1018_SAFETY_TAGS".E_STOP_OK_OFF_DEL_4;
   IF #_w2 AND NOT "DB1030_TEST_STOP".TEST_STP_DONE_LOCKED THEN
       "DB428_OPERATOR_HELP".HELP_OPERATOR_271 := TRUE;
   END_IF;
   IF #_w2 AND NOT "DB7300_INTERLOCK_GENERAL".GENERAL_MACHINE.FROM_ROBOT_TO_UNIT_01.OK_TO_OPEN_SAFETY_GATES THEN
       "DB428_OPERATOR_HELP".HELP_OPERATOR_901 := TRUE;
   END_IF;
END_REGION

